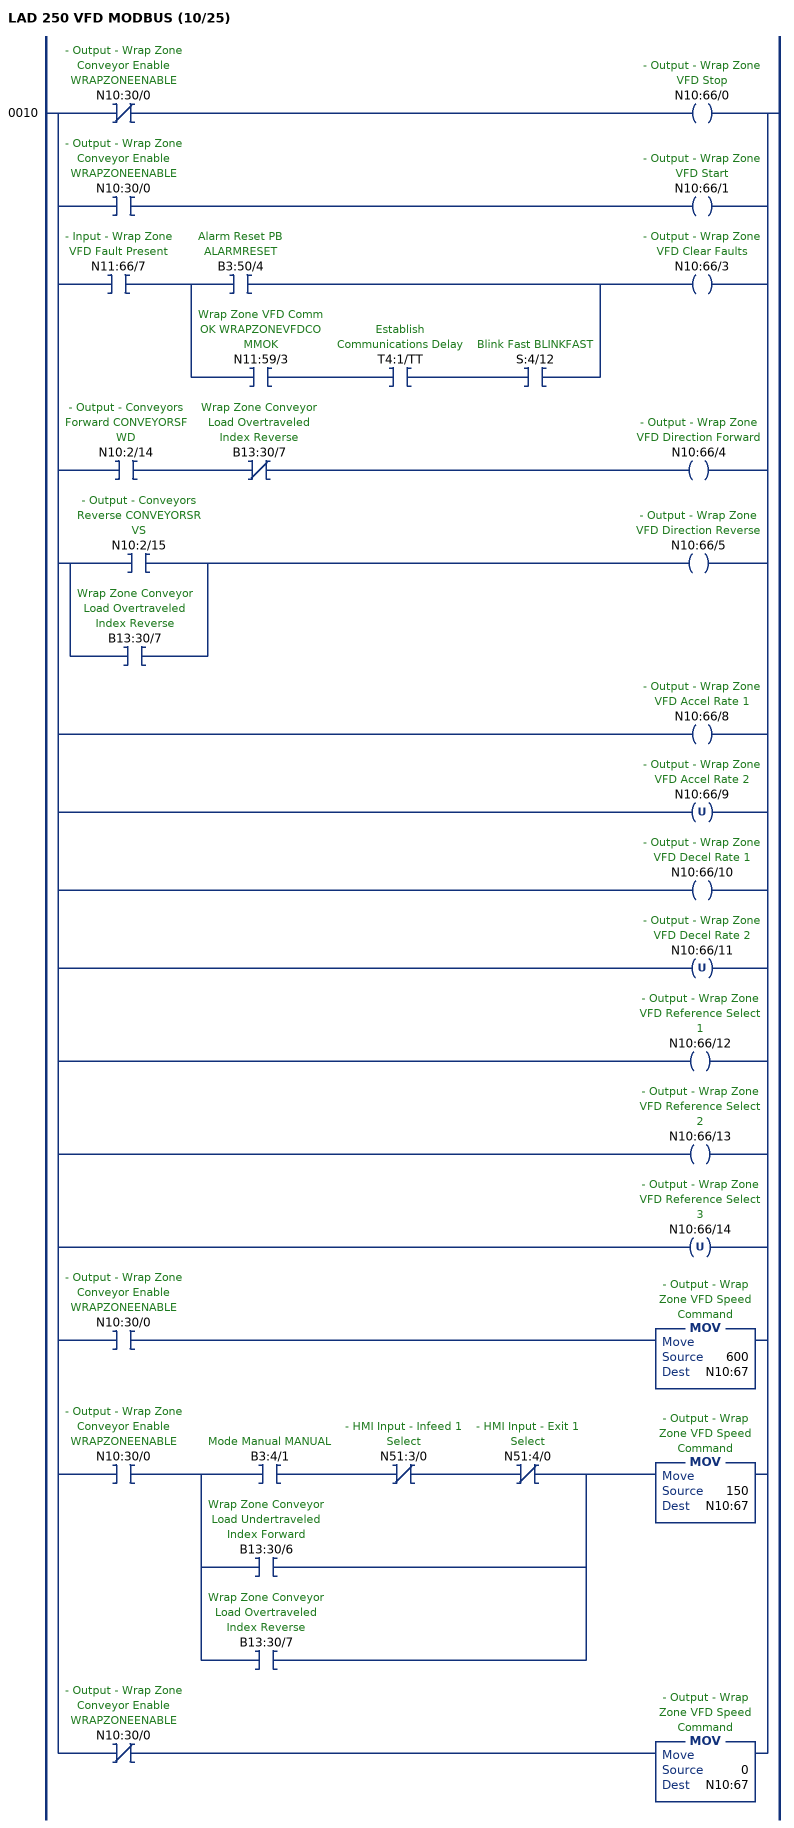
% Rung: 10 %
SOR BST XIO N10:30/0 OTE N10:66/0 NXB XIC N10:30/0 OTE N10:66/1 NXB XIC N11:66/7 BST XIC B3:50/4 NXB XIC N11:59/3 XIC T4:1/TT XIC S:4/12 BND OTE N10:66/3 NXB XIC N10:2/14 XIO B13:30/7 OTE N10:66/4 NXB BST XIC N10:2/15 NXB XIC B13:30/7 BND OTE N10:66/5 NXB OTE N10:66/8 NXB OTU N10:66/9 NXB OTE N10:66/10 NXB OTU N10:66/11 NXB OTE N10:66/12 NXB OTE N10:66/13 NXB OTU N10:66/14 NXB XIC N10:30/0 MOV 600 N10:67 NXB XIC N10:30/0 BST XIC B3:4/1 XIO N51:3/0 XIO N51:4/0 NXB XIC B13:30/6 NXB XIC B13:30/7 BND MOV 150 N10:67 NXB XIO N10:30/0 MOV 0 N10:67 BND EOR
%   N10:30/0  WRAPZONEENABLE  "- Output - Wrap Zone Conveyor Enable" %
%   N10:66/0  "- Output - Wrap Zone VFD Stop" %
%   N10:66/1  "- Output - Wrap Zone VFD Start" %
%   N11:66/7  "- Input - Wrap Zone VFD Fault Present" %
%   B3:50/4  ALARMRESET  "Alarm Reset PB" %
%   N11:59/3  WRAPZONEVFDCOMMOK  "Wrap Zone VFD Comm OK" %
%   T4:1  "Establish Communications Delay" %
%   S:4/12  BLINKFAST  "Blink Fast" %
%   N10:66/3  "- Output - Wrap Zone VFD Clear Faults" %
%   N10:2/14  CONVEYORSFWD  "- Output - Conveyors Forward" %
%   B13:30/7  "Wrap Zone Conveyor Load Overtraveled Index Reverse" %
%   N10:66/4  "- Output - Wrap Zone VFD Direction Forward" %
%   N10:2/15  CONVEYORSRVS  "- Output - Conveyors Reverse" %
%   N10:66/5  "- Output - Wrap Zone VFD Direction Reverse" %
%   N10:66/8  "- Output - Wrap Zone VFD Accel Rate 1" %
%   N10:66/9  "- Output - Wrap Zone VFD Accel Rate 2" %
%   N10:66/10  "- Output - Wrap Zone VFD Decel Rate 1" %
%   N10:66/11  "- Output - Wrap Zone VFD Decel Rate 2" %
%   N10:66/12  "- Output - Wrap Zone VFD Reference Select 1" %
%   N10:66/13  "- Output - Wrap Zone VFD Reference Select 2" %
%   N10:66/14  "- Output - Wrap Zone VFD Reference Select 3" %
%   N10:67  "- Output - Wrap Zone VFD Speed Command" %
%   B3:4/1  MANUAL  "Mode Manual" %
%   N51:3/0  "- HMI Input - Infeed 1 Select" %
%   N51:4/0  "- HMI Input - Exit 1 Select" %
%   B13:30/6  "Wrap Zone Conveyor Load Undertraveled Index Forward" %

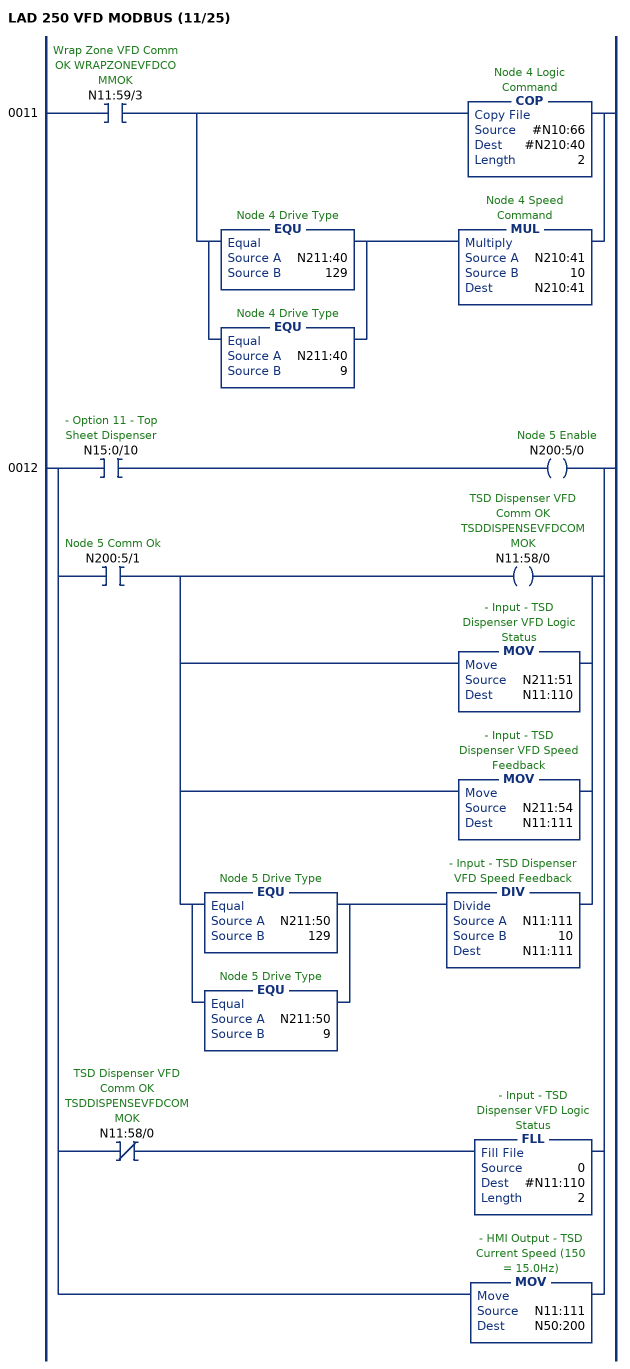
% Rung: 11 %
SOR XIC N11:59/3 BST COP #N10:66 #N210:40 2 NXB BST EQU N211:40 129 NXB EQU N211:40 9 BND MUL N210:41 10 N210:41 BND EOR
%   N11:59/3  WRAPZONEVFDCOMMOK  "Wrap Zone VFD Comm OK" %
%   N10:66  "- Output - Wrap Zone VFD Logic Command" %
%   N210:40  "Node 4 Logic Command" %
%   N211:40  "Node 4 Drive Type" %
%   N210:41  "Node 4 Speed Command" %
% Rung: 12 %
SOR BST XIC N15:0/10 OTE N200:5/0 NXB XIC N200:5/1 BST OTE N11:58/0 NXB MOV N211:51 N11:110 NXB MOV N211:54 N11:111 NXB BST EQU N211:50 129 NXB EQU N211:50 9 BND DIV N11:111 10 N11:111 BND NXB XIO N11:58/0 FLL 0 #N11:110 2 NXB MOV N11:111 N50:200 BND EOR
%   N15:0/10  "- Option 11 - Top Sheet Dispenser" %
%   N200:5/0  "Node 5 Enable" %
%   N200:5/1  "Node 5 Comm Ok" %
%   N11:58/0  TSDDISPENSEVFDCOMMOK  "TSD Dispenser VFD Comm OK" %
%   N211:51  "Node 5 Logic Status" %
%   N11:110  "- Input - TSD Dispenser VFD Logic Status" %
%   N211:54  "Node 5 Speed Feedback" %
%   N11:111  "- Input - TSD Dispenser VFD Speed Feedback" %
%   N211:50  "Node 5 Drive Type" %
%   N50:200  "- HMI Output - TSD Current Speed (150 = 15.0Hz)" %

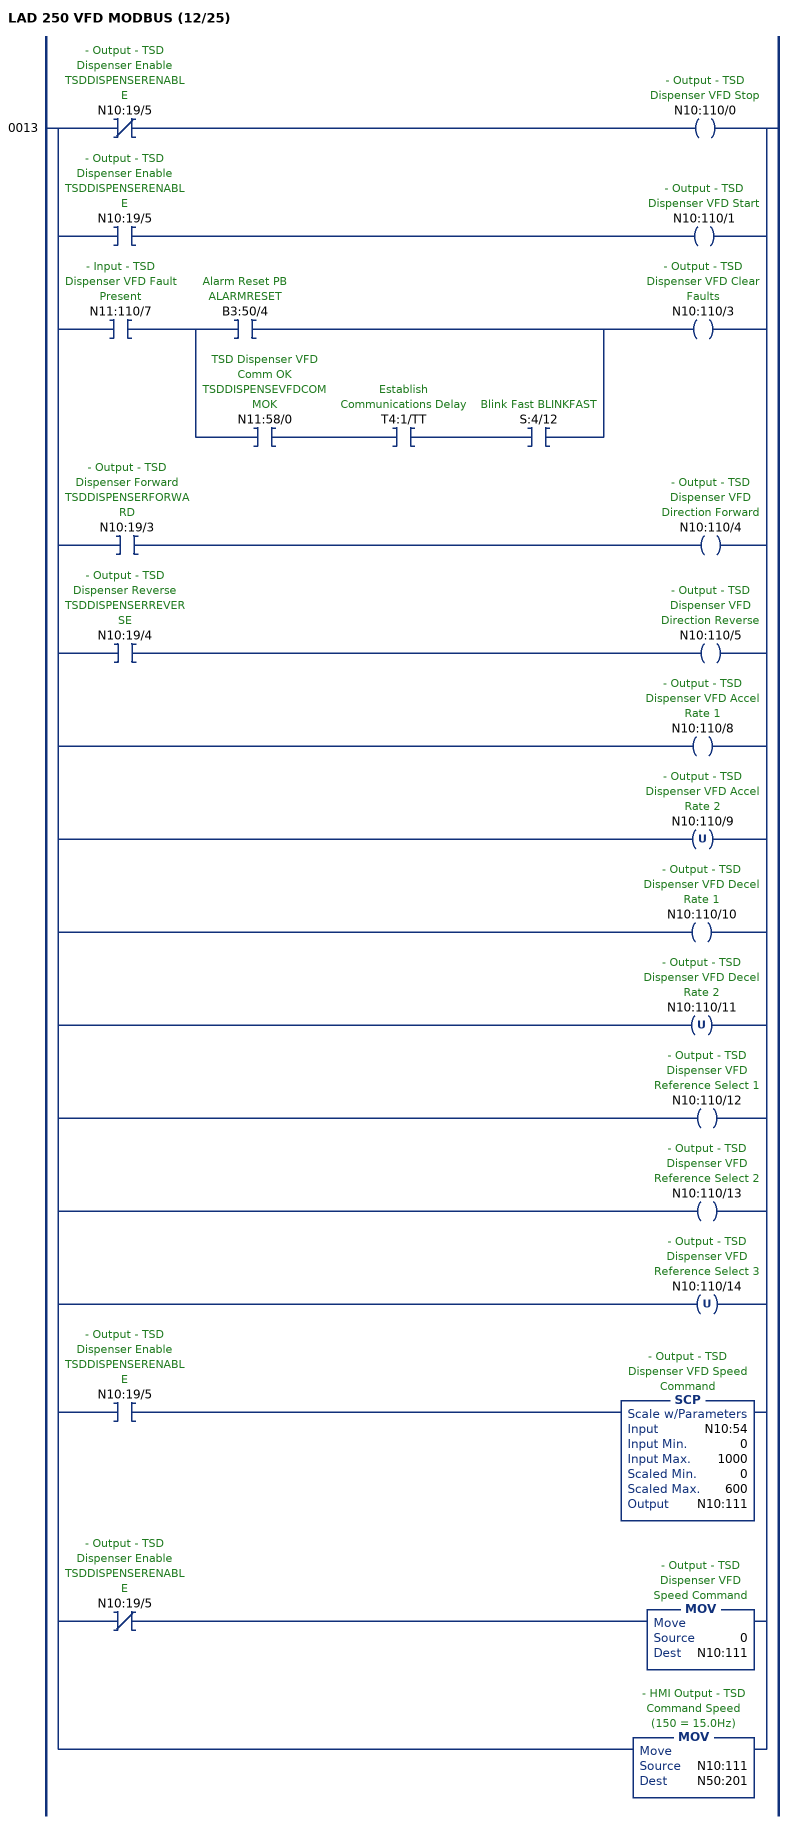
% Rung: 13 %
SOR BST XIO N10:19/5 OTE N10:110/0 NXB XIC N10:19/5 OTE N10:110/1 NXB XIC N11:110/7 BST XIC B3:50/4 NXB XIC N11:58/0 XIC T4:1/TT XIC S:4/12 BND OTE N10:110/3 NXB XIC N10:19/3 OTE N10:110/4 NXB XIC N10:19/4 OTE N10:110/5 NXB OTE N10:110/8 NXB OTU N10:110/9 NXB OTE N10:110/10 NXB OTU N10:110/11 NXB OTE N10:110/12 NXB OTE N10:110/13 NXB OTU N10:110/14 NXB XIC N10:19/5 SCP N10:54 0 1000 0 600 N10:111 NXB XIO N10:19/5 MOV 0 N10:111 NXB MOV N10:111 N50:201 BND EOR
%   N10:19/5  TSDDISPENSERENABLE  "- Output - TSD Dispenser Enable" %
%   N10:110/0  "- Output - TSD Dispenser VFD Stop" %
%   N10:110/1  "- Output - TSD Dispenser VFD Start" %
%   N11:110/7  "- Input - TSD Dispenser VFD Fault Present" %
%   B3:50/4  ALARMRESET  "Alarm Reset PB" %
%   N11:58/0  TSDDISPENSEVFDCOMMOK  "TSD Dispenser VFD Comm OK" %
%   T4:1  "Establish Communications Delay" %
%   S:4/12  BLINKFAST  "Blink Fast" %
%   N10:110/3  "- Output - TSD Dispenser VFD Clear Faults" %
%   N10:19/3  TSDDISPENSERFORWARD  "- Output - TSD Dispenser Forward" %
%   N10:110/4  "- Output - TSD Dispenser VFD Direction Forward" %
%   N10:19/4  TSDDISPENSERREVERSE  "- Output - TSD Dispenser Reverse" %
%   N10:110/5  "- Output - TSD Dispenser VFD Direction Reverse" %
%   N10:110/8  "- Output - TSD Dispenser VFD Accel Rate 1" %
%   N10:110/9  "- Output - TSD Dispenser VFD Accel Rate 2" %
%   N10:110/10  "- Output - TSD Dispenser VFD Decel Rate 1" %
%   N10:110/11  "- Output - TSD Dispenser VFD Decel Rate 2" %
%   N10:110/12  "- Output - TSD Dispenser VFD Reference Select 1" %
%   N10:110/13  "- Output - TSD Dispenser VFD Reference Select 2" %
%   N10:110/14  "- Output - TSD Dispenser VFD Reference Select 3" %
%   N10:54  TSDDISPENSECOMMAND  "- Output - TSD Dispense Speed Command (1000 = 100.0%)" %
%   N10:111  "- Output - TSD Dispenser VFD Speed Command" %
%   N50:201  "- HMI Output - TSD Command Speed (150 = 15.0Hz)" %

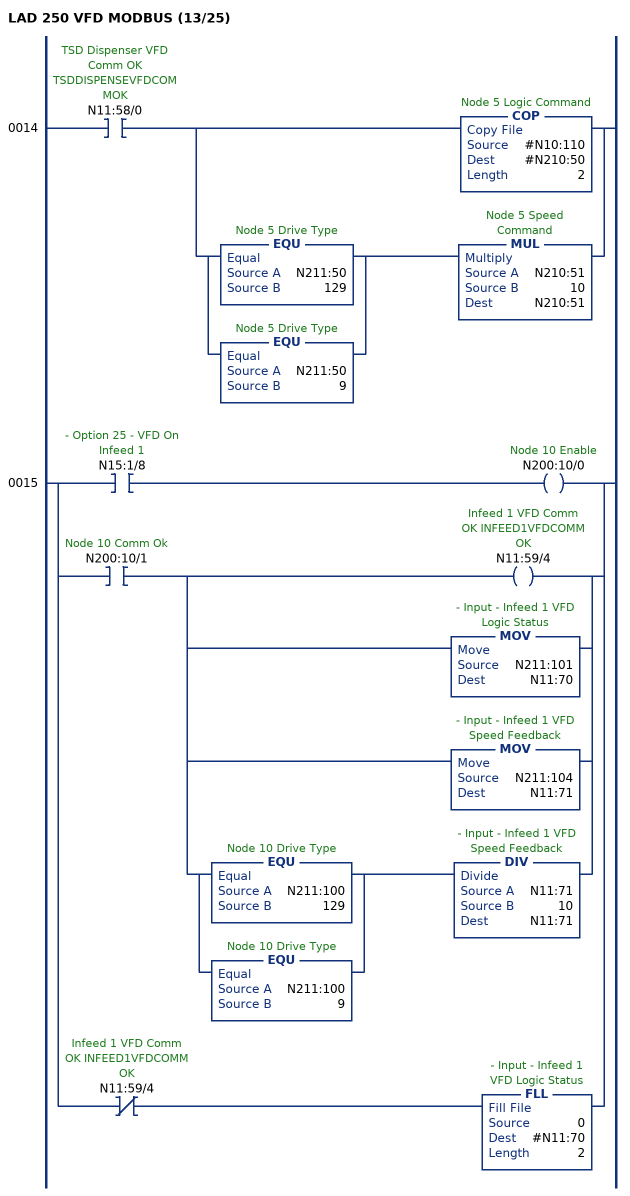
% Rung: 14 %
SOR XIC N11:58/0 BST COP #N10:110 #N210:50 2 NXB BST EQU N211:50 129 NXB EQU N211:50 9 BND MUL N210:51 10 N210:51 BND EOR
%   N11:58/0  TSDDISPENSEVFDCOMMOK  "TSD Dispenser VFD Comm OK" %
%   N10:110  "- Output - TSD Dispenser VFD Logic Command" %
%   N210:50  "Node 5 Logic Command" %
%   N211:50  "Node 5 Drive Type" %
%   N210:51  "Node 5 Speed Command" %
% Rung: 15 %
SOR BST XIC N15:1/8 OTE N200:10/0 NXB XIC N200:10/1 BST OTE N11:59/4 NXB MOV N211:101 N11:70 NXB MOV N211:104 N11:71 NXB BST EQU N211:100 129 NXB EQU N211:100 9 BND DIV N11:71 10 N11:71 BND NXB XIO N11:59/4 FLL 0 #N11:70 2 BND EOR
%   N15:1/8  "- Option 25 - VFD On Infeed 1" %
%   N200:10/0  "Node 10 Enable" %
%   N200:10/1  "Node 10 Comm Ok" %
%   N11:59/4  INFEED1VFDCOMMOK  "Infeed 1 VFD Comm OK" %
%   N211:101  "Node 10 Logic Status" %
%   N11:70  "- Input - Infeed 1 VFD Logic Status" %
%   N211:104  "Node 10 Speed Feedback" %
%   N11:71  "- Input - Infeed 1 VFD Speed Feedback" %
%   N211:100  "Node 10 Drive Type" %

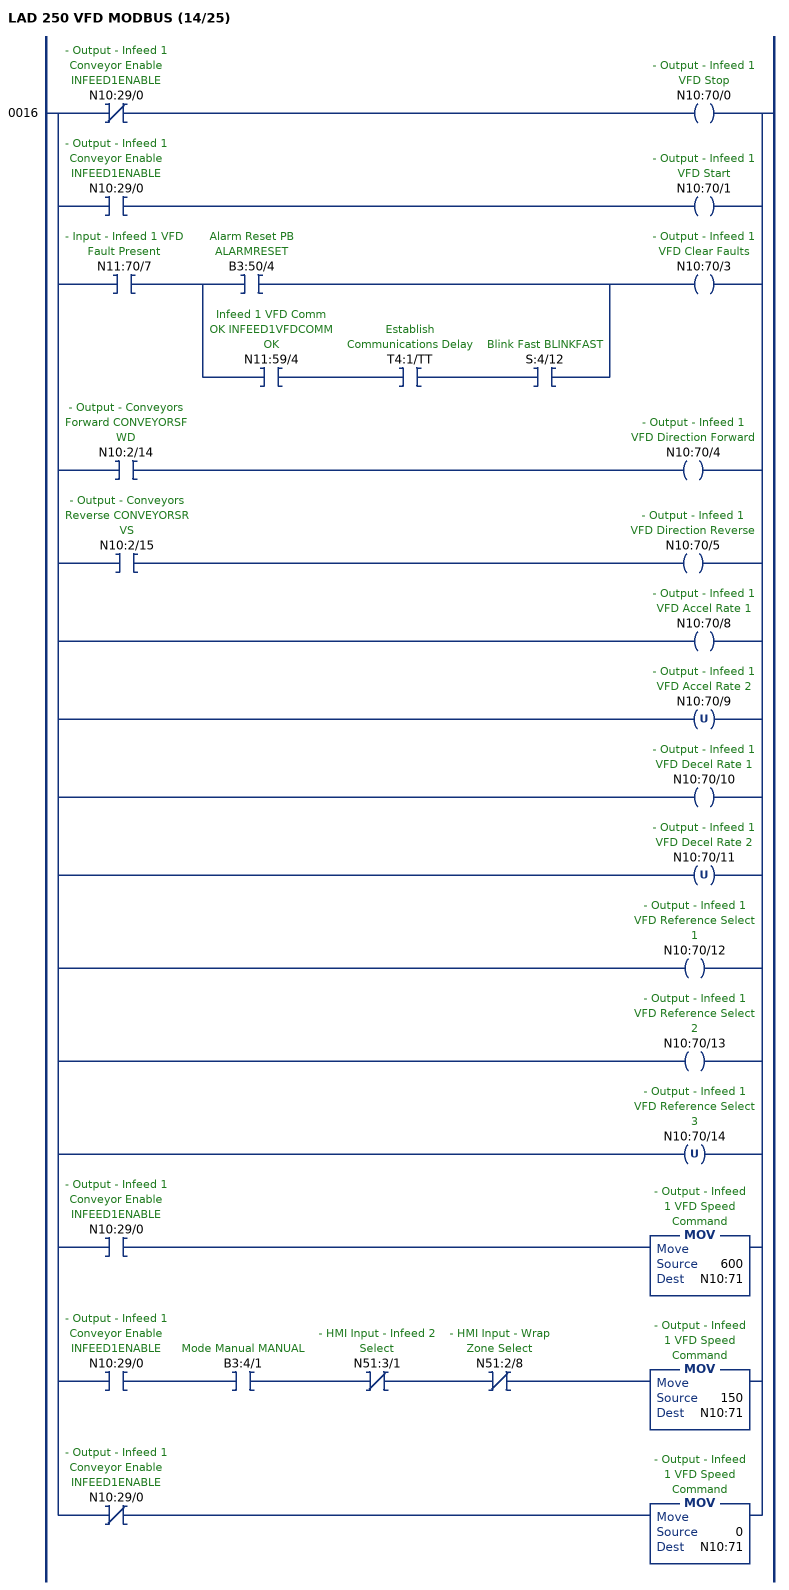
% Rung: 16 %
SOR BST XIO N10:29/0 OTE N10:70/0 NXB XIC N10:29/0 OTE N10:70/1 NXB XIC N11:70/7 BST XIC B3:50/4 NXB XIC N11:59/4 XIC T4:1/TT XIC S:4/12 BND OTE N10:70/3 NXB XIC N10:2/14 OTE N10:70/4 NXB XIC N10:2/15 OTE N10:70/5 NXB OTE N10:70/8 NXB OTU N10:70/9 NXB OTE N10:70/10 NXB OTU N10:70/11 NXB OTE N10:70/12 NXB OTE N10:70/13 NXB OTU N10:70/14 NXB XIC N10:29/0 MOV 600 N10:71 NXB XIC N10:29/0 XIC B3:4/1 XIO N51:3/1 XIO N51:2/8 MOV 150 N10:71 NXB XIO N10:29/0 MOV 0 N10:71 BND EOR
%   N10:29/0  INFEED1ENABLE  "- Output - Infeed 1 Conveyor Enable" %
%   N10:70/0  "- Output - Infeed 1 VFD Stop" %
%   N10:70/1  "- Output - Infeed 1 VFD Start" %
%   N11:70/7  "- Input - Infeed 1 VFD Fault Present" %
%   B3:50/4  ALARMRESET  "Alarm Reset PB" %
%   N11:59/4  INFEED1VFDCOMMOK  "Infeed 1 VFD Comm OK" %
%   T4:1  "Establish Communications Delay" %
%   S:4/12  BLINKFAST  "Blink Fast" %
%   N10:70/3  "- Output - Infeed 1 VFD Clear Faults" %
%   N10:2/14  CONVEYORSFWD  "- Output - Conveyors Forward" %
%   N10:70/4  "- Output - Infeed 1 VFD Direction Forward" %
%   N10:2/15  CONVEYORSRVS  "- Output - Conveyors Reverse" %
%   N10:70/5  "- Output - Infeed 1 VFD Direction Reverse" %
%   N10:70/8  "- Output - Infeed 1 VFD Accel Rate 1" %
%   N10:70/9  "- Output - Infeed 1 VFD Accel Rate 2" %
%   N10:70/10  "- Output - Infeed 1 VFD Decel Rate 1" %
%   N10:70/11  "- Output - Infeed 1 VFD Decel Rate 2" %
%   N10:70/12  "- Output - Infeed 1 VFD Reference Select 1" %
%   N10:70/13  "- Output - Infeed 1 VFD Reference Select 2" %
%   N10:70/14  "- Output - Infeed 1 VFD Reference Select 3" %
%   N10:71  "- Output - Infeed 1 VFD Speed Command" %
%   B3:4/1  MANUAL  "Mode Manual" %
%   N51:3/1  "- HMI Input - Infeed 2 Select" %
%   N51:2/8  "- HMI Input - Wrap Zone Select" %

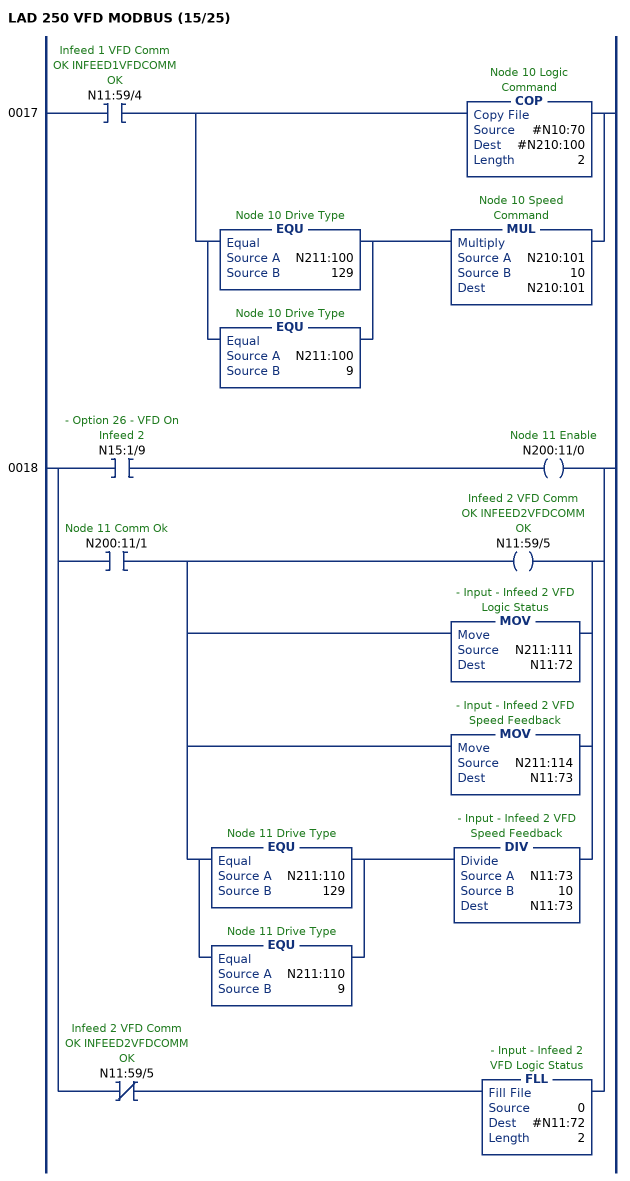
% Rung: 17 %
SOR XIC N11:59/4 BST COP #N10:70 #N210:100 2 NXB BST EQU N211:100 129 NXB EQU N211:100 9 BND MUL N210:101 10 N210:101 BND EOR
%   N11:59/4  INFEED1VFDCOMMOK  "Infeed 1 VFD Comm OK" %
%   N10:70  "- Output - Infeed 1 VFD Logic Command" %
%   N210:100  "Node 10 Logic Command" %
%   N211:100  "Node 10 Drive Type" %
%   N210:101  "Node 10 Speed Command" %
% Rung: 18 %
SOR BST XIC N15:1/9 OTE N200:11/0 NXB XIC N200:11/1 BST OTE N11:59/5 NXB MOV N211:111 N11:72 NXB MOV N211:114 N11:73 NXB BST EQU N211:110 129 NXB EQU N211:110 9 BND DIV N11:73 10 N11:73 BND NXB XIO N11:59/5 FLL 0 #N11:72 2 BND EOR
%   N15:1/9  "- Option 26 - VFD On Infeed 2" %
%   N200:11/0  "Node 11 Enable" %
%   N200:11/1  "Node 11 Comm Ok" %
%   N11:59/5  INFEED2VFDCOMMOK  "Infeed 2 VFD Comm OK" %
%   N211:111  "Node 11 Logic Status" %
%   N11:72  "- Input - Infeed 2 VFD Logic Status" %
%   N211:114  "Node 11 Speed Feedback" %
%   N11:73  "- Input - Infeed 2 VFD Speed Feedback" %
%   N211:110  "Node 11 Drive Type" %

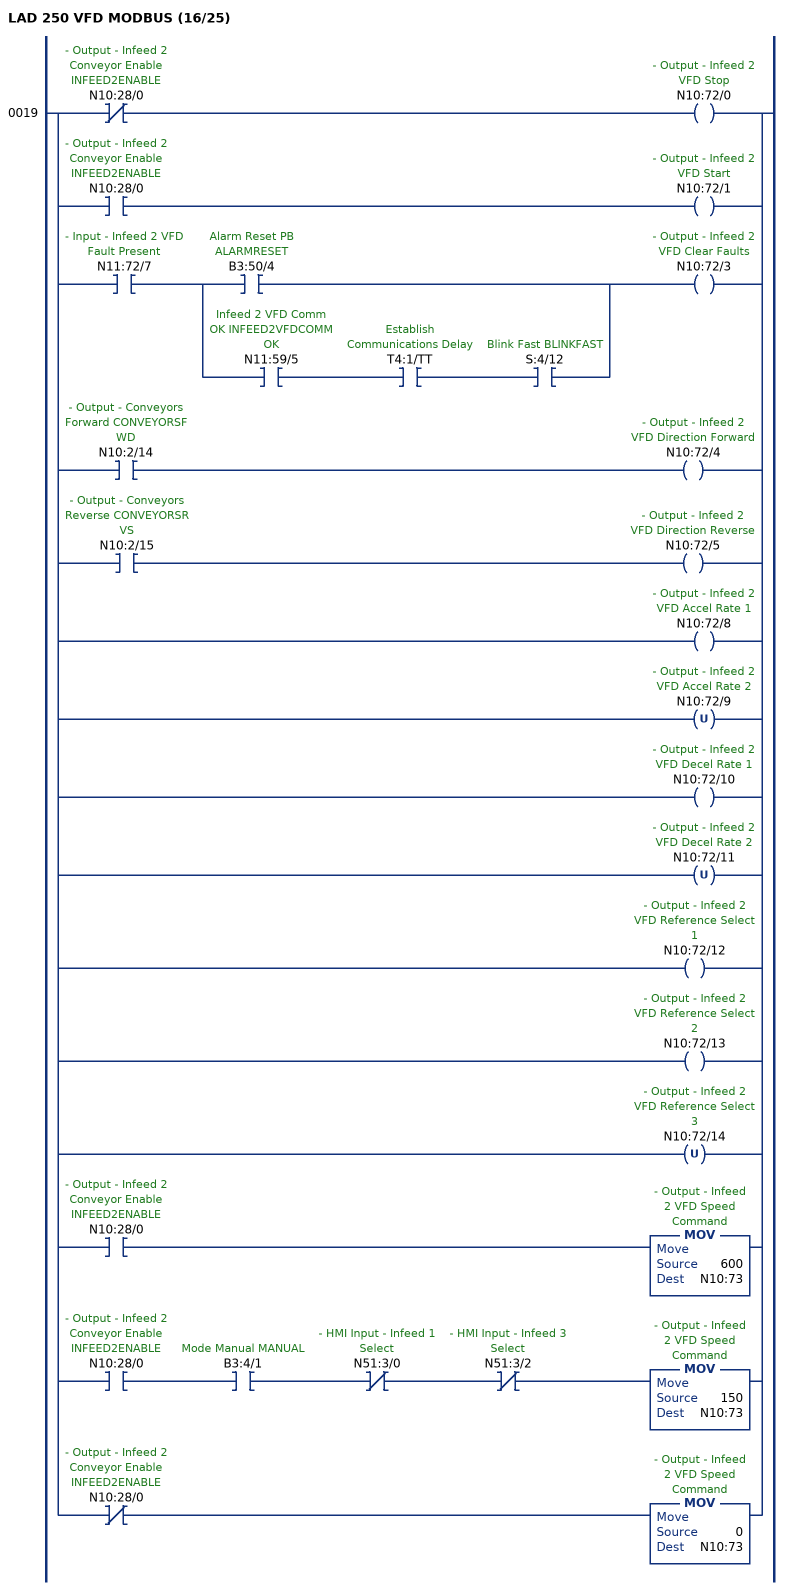
% Rung: 19 %
SOR BST XIO N10:28/0 OTE N10:72/0 NXB XIC N10:28/0 OTE N10:72/1 NXB XIC N11:72/7 BST XIC B3:50/4 NXB XIC N11:59/5 XIC T4:1/TT XIC S:4/12 BND OTE N10:72/3 NXB XIC N10:2/14 OTE N10:72/4 NXB XIC N10:2/15 OTE N10:72/5 NXB OTE N10:72/8 NXB OTU N10:72/9 NXB OTE N10:72/10 NXB OTU N10:72/11 NXB OTE N10:72/12 NXB OTE N10:72/13 NXB OTU N10:72/14 NXB XIC N10:28/0 MOV 600 N10:73 NXB XIC N10:28/0 XIC B3:4/1 XIO N51:3/0 XIO N51:3/2 MOV 150 N10:73 NXB XIO N10:28/0 MOV 0 N10:73 BND EOR
%   N10:28/0  INFEED2ENABLE  "- Output - Infeed 2 Conveyor Enable" %
%   N10:72/0  "- Output - Infeed 2 VFD Stop" %
%   N10:72/1  "- Output - Infeed 2 VFD Start" %
%   N11:72/7  "- Input - Infeed 2 VFD Fault Present" %
%   B3:50/4  ALARMRESET  "Alarm Reset PB" %
%   N11:59/5  INFEED2VFDCOMMOK  "Infeed 2 VFD Comm OK" %
%   T4:1  "Establish Communications Delay" %
%   S:4/12  BLINKFAST  "Blink Fast" %
%   N10:72/3  "- Output - Infeed 2 VFD Clear Faults" %
%   N10:2/14  CONVEYORSFWD  "- Output - Conveyors Forward" %
%   N10:72/4  "- Output - Infeed 2 VFD Direction Forward" %
%   N10:2/15  CONVEYORSRVS  "- Output - Conveyors Reverse" %
%   N10:72/5  "- Output - Infeed 2 VFD Direction Reverse" %
%   N10:72/8  "- Output - Infeed 2 VFD Accel Rate 1" %
%   N10:72/9  "- Output - Infeed 2 VFD Accel Rate 2" %
%   N10:72/10  "- Output - Infeed 2 VFD Decel Rate 1" %
%   N10:72/11  "- Output - Infeed 2 VFD Decel Rate 2" %
%   N10:72/12  "- Output - Infeed 2 VFD Reference Select 1" %
%   N10:72/13  "- Output - Infeed 2 VFD Reference Select 2" %
%   N10:72/14  "- Output - Infeed 2 VFD Reference Select 3" %
%   N10:73  "- Output - Infeed 2 VFD Speed Command" %
%   B3:4/1  MANUAL  "Mode Manual" %
%   N51:3/0  "- HMI Input - Infeed 1 Select" %
%   N51:3/2  "- HMI Input - Infeed 3 Select" %

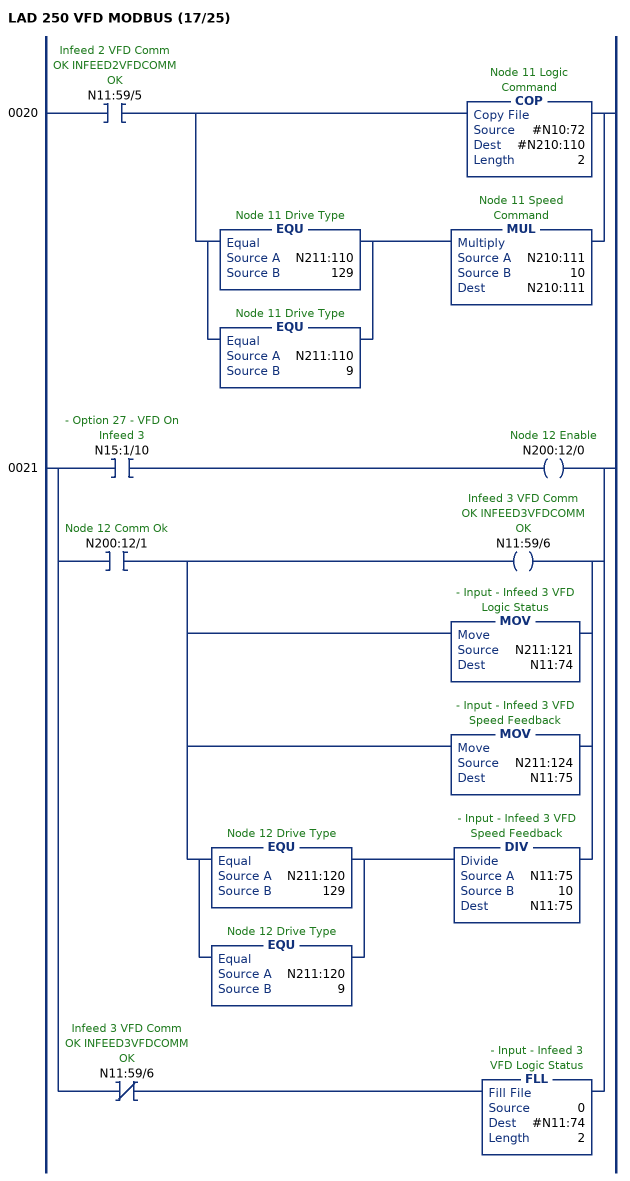
% Rung: 20 %
SOR XIC N11:59/5 BST COP #N10:72 #N210:110 2 NXB BST EQU N211:110 129 NXB EQU N211:110 9 BND MUL N210:111 10 N210:111 BND EOR
%   N11:59/5  INFEED2VFDCOMMOK  "Infeed 2 VFD Comm OK" %
%   N10:72  "- Output - Infeed 2 VFD Logic Command" %
%   N210:110  "Node 11 Logic Command" %
%   N211:110  "Node 11 Drive Type" %
%   N210:111  "Node 11 Speed Command" %
% Rung: 21 %
SOR BST XIC N15:1/10 OTE N200:12/0 NXB XIC N200:12/1 BST OTE N11:59/6 NXB MOV N211:121 N11:74 NXB MOV N211:124 N11:75 NXB BST EQU N211:120 129 NXB EQU N211:120 9 BND DIV N11:75 10 N11:75 BND NXB XIO N11:59/6 FLL 0 #N11:74 2 BND EOR
%   N15:1/10  "- Option 27 - VFD On Infeed 3" %
%   N200:12/0  "Node 12 Enable" %
%   N200:12/1  "Node 12 Comm Ok" %
%   N11:59/6  INFEED3VFDCOMMOK  "Infeed 3 VFD Comm OK" %
%   N211:121  "Node 12 Logic Status" %
%   N11:74  "- Input - Infeed 3 VFD Logic Status" %
%   N211:124  "Node 12 Speed Feedback" %
%   N11:75  "- Input - Infeed 3 VFD Speed Feedback" %
%   N211:120  "Node 12 Drive Type" %

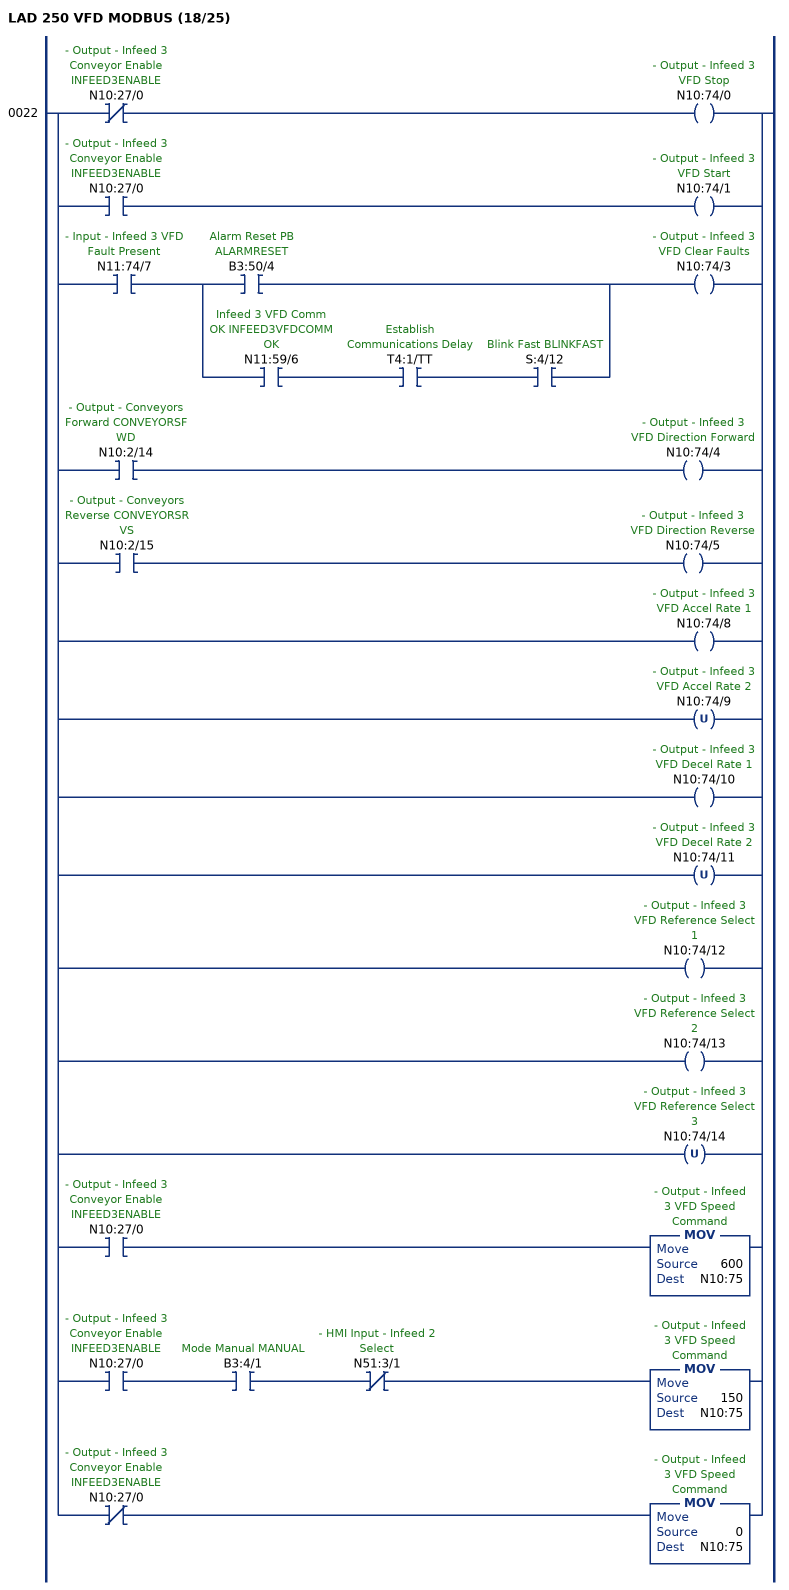
% Rung: 22 %
SOR BST XIO N10:27/0 OTE N10:74/0 NXB XIC N10:27/0 OTE N10:74/1 NXB XIC N11:74/7 BST XIC B3:50/4 NXB XIC N11:59/6 XIC T4:1/TT XIC S:4/12 BND OTE N10:74/3 NXB XIC N10:2/14 OTE N10:74/4 NXB XIC N10:2/15 OTE N10:74/5 NXB OTE N10:74/8 NXB OTU N10:74/9 NXB OTE N10:74/10 NXB OTU N10:74/11 NXB OTE N10:74/12 NXB OTE N10:74/13 NXB OTU N10:74/14 NXB XIC N10:27/0 MOV 600 N10:75 NXB XIC N10:27/0 XIC B3:4/1 XIO N51:3/1 MOV 150 N10:75 NXB XIO N10:27/0 MOV 0 N10:75 BND EOR
%   N10:27/0  INFEED3ENABLE  "- Output - Infeed 3 Conveyor Enable" %
%   N10:74/0  "- Output - Infeed 3 VFD Stop" %
%   N10:74/1  "- Output - Infeed 3 VFD Start" %
%   N11:74/7  "- Input - Infeed 3 VFD Fault Present" %
%   B3:50/4  ALARMRESET  "Alarm Reset PB" %
%   N11:59/6  INFEED3VFDCOMMOK  "Infeed 3 VFD Comm OK" %
%   T4:1  "Establish Communications Delay" %
%   S:4/12  BLINKFAST  "Blink Fast" %
%   N10:74/3  "- Output - Infeed 3 VFD Clear Faults" %
%   N10:2/14  CONVEYORSFWD  "- Output - Conveyors Forward" %
%   N10:74/4  "- Output - Infeed 3 VFD Direction Forward" %
%   N10:2/15  CONVEYORSRVS  "- Output - Conveyors Reverse" %
%   N10:74/5  "- Output - Infeed 3 VFD Direction Reverse" %
%   N10:74/8  "- Output - Infeed 3 VFD Accel Rate 1" %
%   N10:74/9  "- Output - Infeed 3 VFD Accel Rate 2" %
%   N10:74/10  "- Output - Infeed 3 VFD Decel Rate 1" %
%   N10:74/11  "- Output - Infeed 3 VFD Decel Rate 2" %
%   N10:74/12  "- Output - Infeed 3 VFD Reference Select 1" %
%   N10:74/13  "- Output - Infeed 3 VFD Reference Select 2" %
%   N10:74/14  "- Output - Infeed 3 VFD Reference Select 3" %
%   N10:75  "- Output - Infeed 3 VFD Speed Command" %
%   B3:4/1  MANUAL  "Mode Manual" %
%   N51:3/1  "- HMI Input - Infeed 2 Select" %

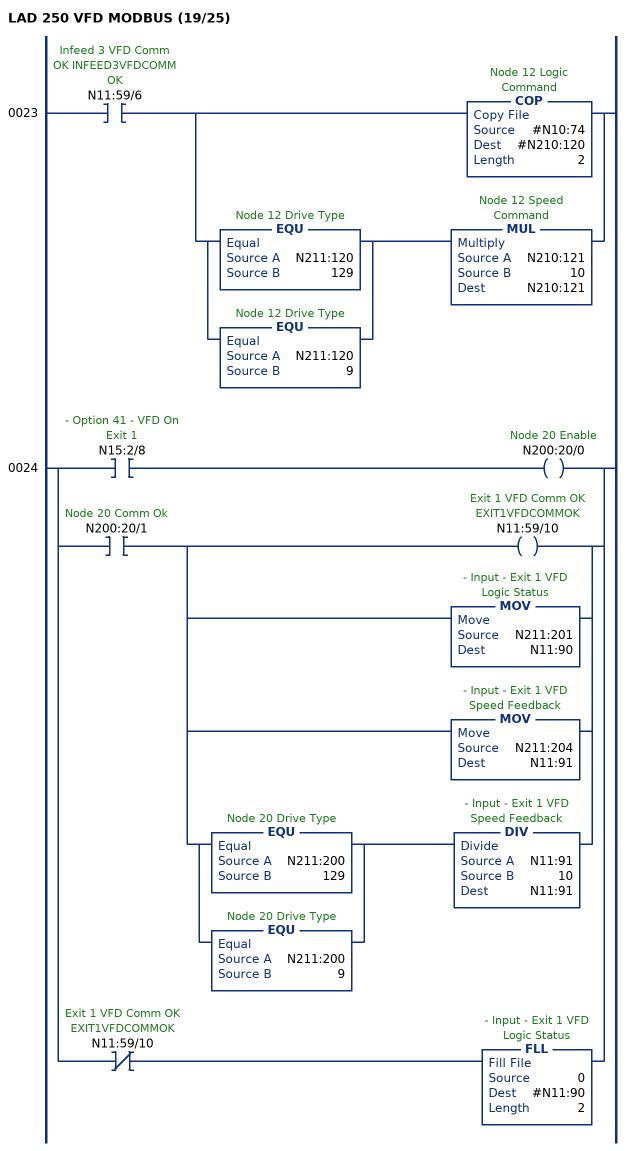
% Rung: 23 %
SOR XIC N11:59/6 BST COP #N10:74 #N210:120 2 NXB BST EQU N211:120 129 NXB EQU N211:120 9 BND MUL N210:121 10 N210:121 BND EOR
%   N11:59/6  INFEED3VFDCOMMOK  "Infeed 3 VFD Comm OK" %
%   N10:74  "- Output - Infeed 3 VFD Logic Command" %
%   N210:120  "Node 12 Logic Command" %
%   N211:120  "Node 12 Drive Type" %
%   N210:121  "Node 12 Speed Command" %
% Rung: 24 %
SOR BST XIC N15:2/8 OTE N200:20/0 NXB XIC N200:20/1 BST OTE N11:59/10 NXB MOV N211:201 N11:90 NXB MOV N211:204 N11:91 NXB BST EQU N211:200 129 NXB EQU N211:200 9 BND DIV N11:91 10 N11:91 BND NXB XIO N11:59/10 FLL 0 #N11:90 2 BND EOR
%   N15:2/8  "- Option 41 - VFD On Exit 1" %
%   N200:20/0  "Node 20 Enable" %
%   N200:20/1  "Node 20 Comm Ok" %
%   N11:59/10  EXIT1VFDCOMMOK  "Exit 1 VFD Comm OK" %
%   N211:201  "Node 20 Logic Status" %
%   N11:90  "- Input - Exit 1 VFD Logic Status" %
%   N211:204  "Node 20 Speed Feedback" %
%   N11:91  "- Input - Exit 1 VFD Speed Feedback" %
%   N211:200  "Node 20 Drive Type" %

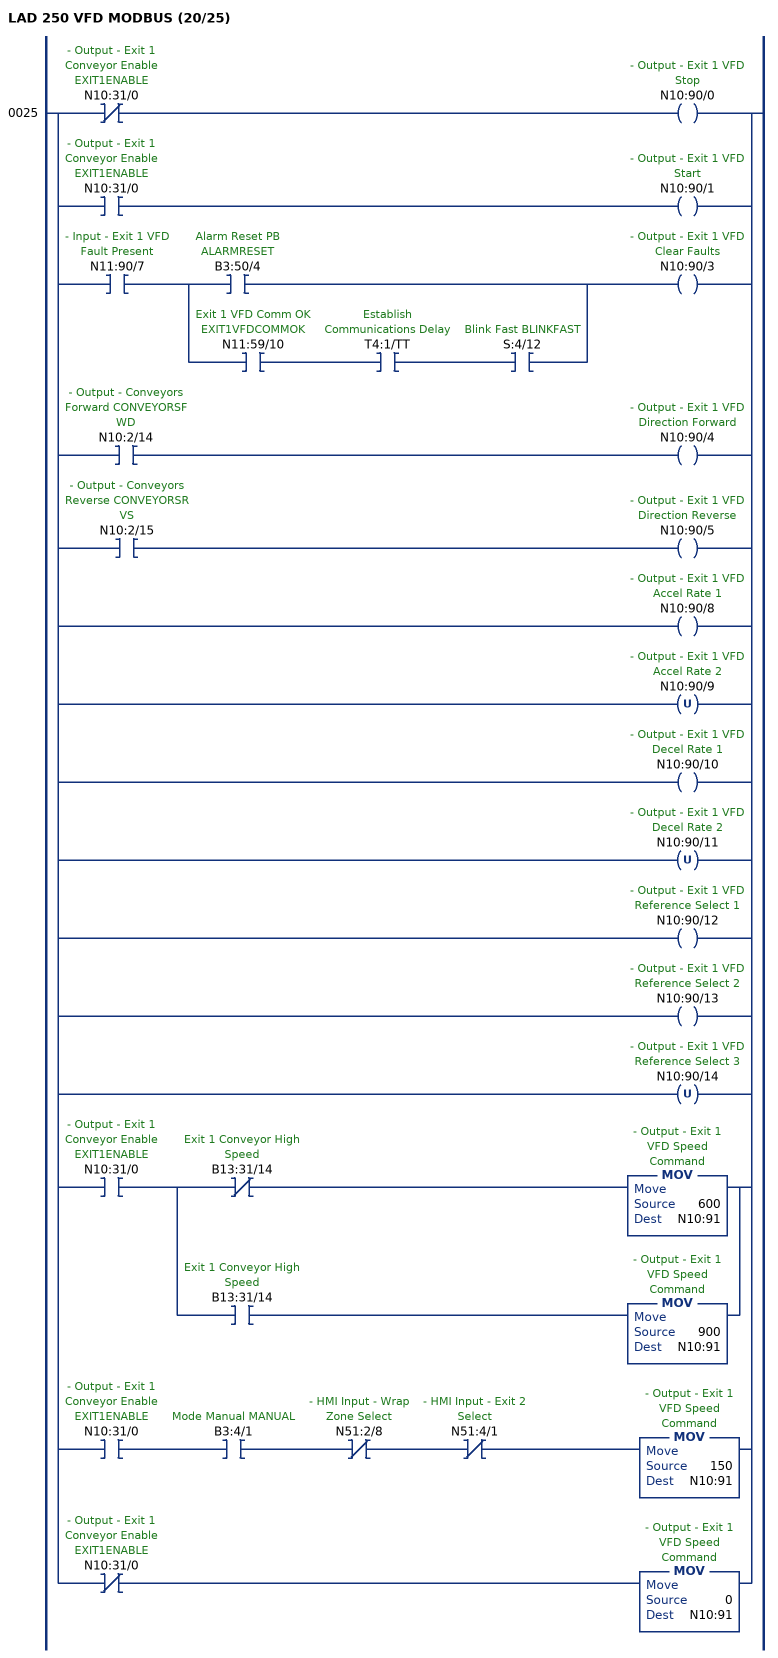
% Rung: 25 %
SOR BST XIO N10:31/0 OTE N10:90/0 NXB XIC N10:31/0 OTE N10:90/1 NXB XIC N11:90/7 BST XIC B3:50/4 NXB XIC N11:59/10 XIC T4:1/TT XIC S:4/12 BND OTE N10:90/3 NXB XIC N10:2/14 OTE N10:90/4 NXB XIC N10:2/15 OTE N10:90/5 NXB OTE N10:90/8 NXB OTU N10:90/9 NXB OTE N10:90/10 NXB OTU N10:90/11 NXB OTE N10:90/12 NXB OTE N10:90/13 NXB OTU N10:90/14 NXB XIC N10:31/0 BST XIO B13:31/14 MOV 600 N10:91 NXB XIC B13:31/14 MOV 900 N10:91 BND NXB XIC N10:31/0 XIC B3:4/1 XIO N51:2/8 XIO N51:4/1 MOV 150 N10:91 NXB XIO N10:31/0 MOV 0 N10:91 BND EOR
%   N10:31/0  EXIT1ENABLE  "- Output - Exit 1 Conveyor Enable" %
%   N10:90/0  "- Output - Exit 1 VFD Stop" %
%   N10:90/1  "- Output - Exit 1 VFD Start" %
%   N11:90/7  "- Input - Exit 1 VFD Fault Present" %
%   B3:50/4  ALARMRESET  "Alarm Reset PB" %
%   N11:59/10  EXIT1VFDCOMMOK  "Exit 1 VFD Comm OK" %
%   T4:1  "Establish Communications Delay" %
%   S:4/12  BLINKFAST  "Blink Fast" %
%   N10:90/3  "- Output - Exit 1 VFD Clear Faults" %
%   N10:2/14  CONVEYORSFWD  "- Output - Conveyors Forward" %
%   N10:90/4  "- Output - Exit 1 VFD Direction Forward" %
%   N10:2/15  CONVEYORSRVS  "- Output - Conveyors Reverse" %
%   N10:90/5  "- Output - Exit 1 VFD Direction Reverse" %
%   N10:90/8  "- Output - Exit 1 VFD Accel Rate 1" %
%   N10:90/9  "- Output - Exit 1 VFD Accel Rate 2" %
%   N10:90/10  "- Output - Exit 1 VFD Decel Rate 1" %
%   N10:90/11  "- Output - Exit 1 VFD Decel Rate 2" %
%   N10:90/12  "- Output - Exit 1 VFD Reference Select 1" %
%   N10:90/13  "- Output - Exit 1 VFD Reference Select 2" %
%   N10:90/14  "- Output - Exit 1 VFD Reference Select 3" %
%   B13:31/14  "Exit 1 Conveyor High Speed" %
%   N10:91  "- Output - Exit 1 VFD Speed Command" %
%   B3:4/1  MANUAL  "Mode Manual" %
%   N51:2/8  "- HMI Input - Wrap Zone Select" %
%   N51:4/1  "- HMI Input - Exit 2 Select" %

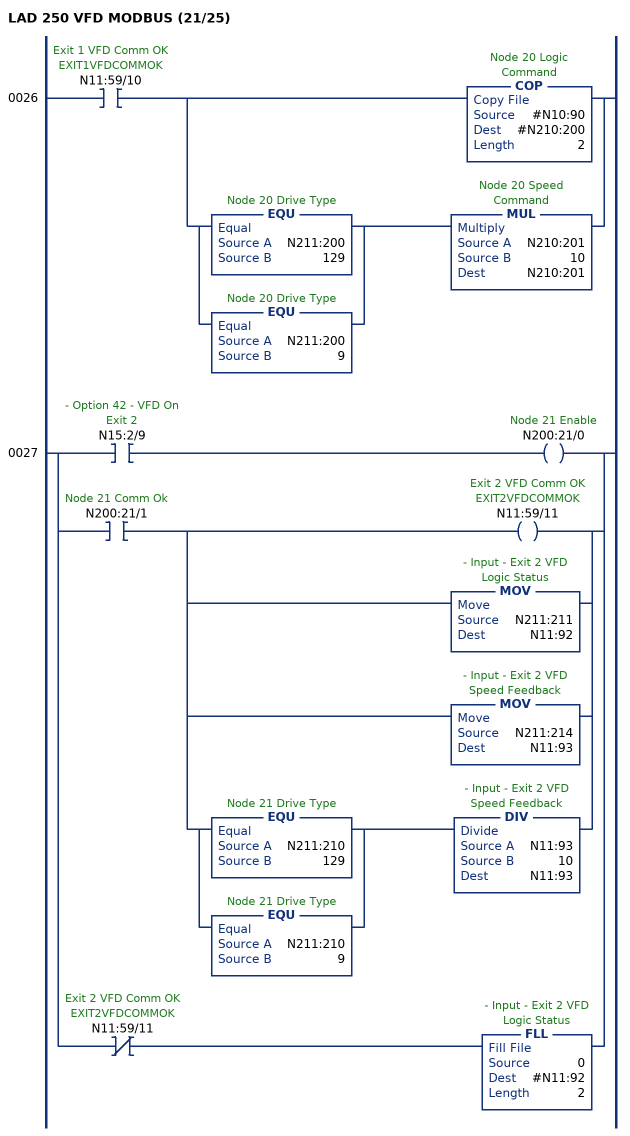
% Rung: 26 %
SOR XIC N11:59/10 BST COP #N10:90 #N210:200 2 NXB BST EQU N211:200 129 NXB EQU N211:200 9 BND MUL N210:201 10 N210:201 BND EOR
%   N11:59/10  EXIT1VFDCOMMOK  "Exit 1 VFD Comm OK" %
%   N10:90  "- Output - Exit 1 VFD Logic Command" %
%   N210:200  "Node 20 Logic Command" %
%   N211:200  "Node 20 Drive Type" %
%   N210:201  "Node 20 Speed Command" %
% Rung: 27 %
SOR BST XIC N15:2/9 OTE N200:21/0 NXB XIC N200:21/1 BST OTE N11:59/11 NXB MOV N211:211 N11:92 NXB MOV N211:214 N11:93 NXB BST EQU N211:210 129 NXB EQU N211:210 9 BND DIV N11:93 10 N11:93 BND NXB XIO N11:59/11 FLL 0 #N11:92 2 BND EOR
%   N15:2/9  "- Option 42 - VFD On Exit 2" %
%   N200:21/0  "Node 21 Enable" %
%   N200:21/1  "Node 21 Comm Ok" %
%   N11:59/11  EXIT2VFDCOMMOK  "Exit 2 VFD Comm OK" %
%   N211:211  "Node 21 Logic Status" %
%   N11:92  "- Input - Exit 2 VFD Logic Status" %
%   N211:214  "Node 21 Speed Feedback" %
%   N11:93  "- Input - Exit 2 VFD Speed Feedback" %
%   N211:210  "Node 21 Drive Type" %

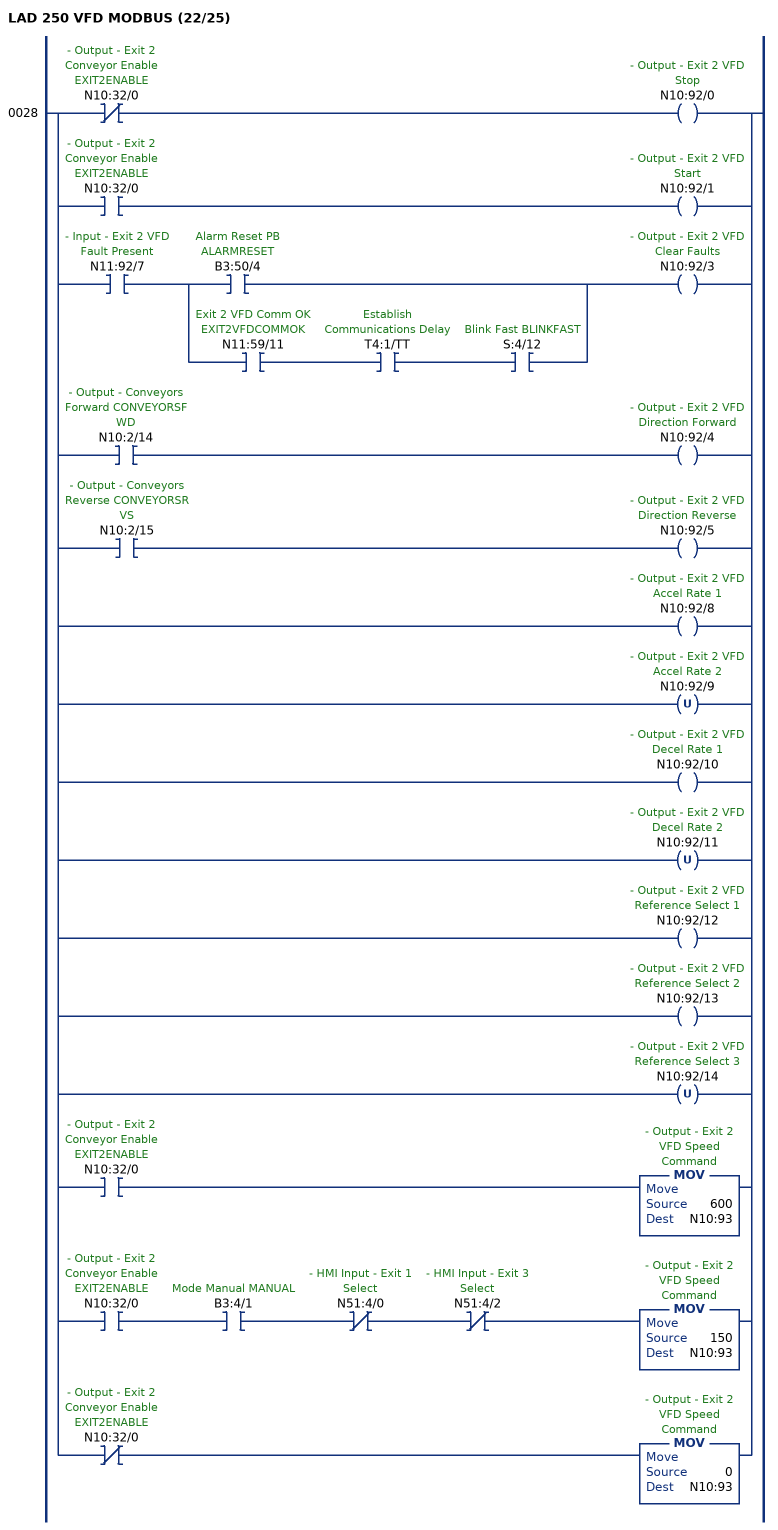
% Rung: 28 %
SOR BST XIO N10:32/0 OTE N10:92/0 NXB XIC N10:32/0 OTE N10:92/1 NXB XIC N11:92/7 BST XIC B3:50/4 NXB XIC N11:59/11 XIC T4:1/TT XIC S:4/12 BND OTE N10:92/3 NXB XIC N10:2/14 OTE N10:92/4 NXB XIC N10:2/15 OTE N10:92/5 NXB OTE N10:92/8 NXB OTU N10:92/9 NXB OTE N10:92/10 NXB OTU N10:92/11 NXB OTE N10:92/12 NXB OTE N10:92/13 NXB OTU N10:92/14 NXB XIC N10:32/0 MOV 600 N10:93 NXB XIC N10:32/0 XIC B3:4/1 XIO N51:4/0 XIO N51:4/2 MOV 150 N10:93 NXB XIO N10:32/0 MOV 0 N10:93 BND EOR
%   N10:32/0  EXIT2ENABLE  "- Output - Exit 2 Conveyor Enable" %
%   N10:92/0  "- Output - Exit 2 VFD Stop" %
%   N10:92/1  "- Output - Exit 2 VFD Start" %
%   N11:92/7  "- Input - Exit 2 VFD Fault Present" %
%   B3:50/4  ALARMRESET  "Alarm Reset PB" %
%   N11:59/11  EXIT2VFDCOMMOK  "Exit 2 VFD Comm OK" %
%   T4:1  "Establish Communications Delay" %
%   S:4/12  BLINKFAST  "Blink Fast" %
%   N10:92/3  "- Output - Exit 2 VFD Clear Faults" %
%   N10:2/14  CONVEYORSFWD  "- Output - Conveyors Forward" %
%   N10:92/4  "- Output - Exit 2 VFD Direction Forward" %
%   N10:2/15  CONVEYORSRVS  "- Output - Conveyors Reverse" %
%   N10:92/5  "- Output - Exit 2 VFD Direction Reverse" %
%   N10:92/8  "- Output - Exit 2 VFD Accel Rate 1" %
%   N10:92/9  "- Output - Exit 2 VFD Accel Rate 2" %
%   N10:92/10  "- Output - Exit 2 VFD Decel Rate 1" %
%   N10:92/11  "- Output - Exit 2 VFD Decel Rate 2" %
%   N10:92/12  "- Output - Exit 2 VFD Reference Select 1" %
%   N10:92/13  "- Output - Exit 2 VFD Reference Select 2" %
%   N10:92/14  "- Output - Exit 2 VFD Reference Select 3" %
%   N10:93  "- Output - Exit 2 VFD Speed Command" %
%   B3:4/1  MANUAL  "Mode Manual" %
%   N51:4/0  "- HMI Input - Exit 1 Select" %
%   N51:4/2  "- HMI Input - Exit 3 Select" %

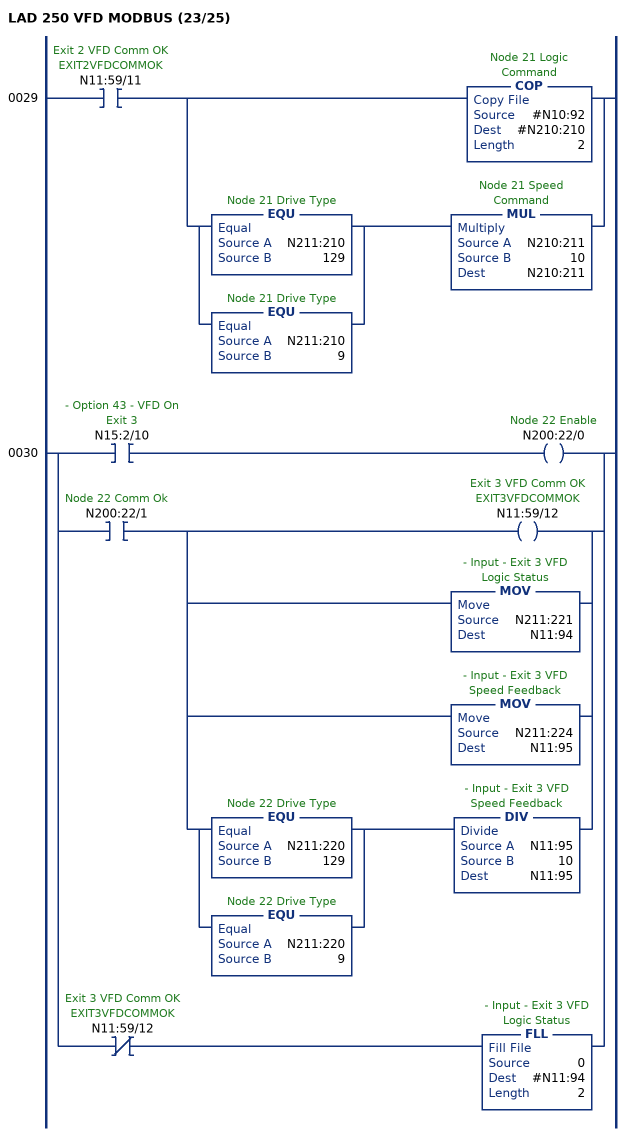
% Rung: 29 %
SOR XIC N11:59/11 BST COP #N10:92 #N210:210 2 NXB BST EQU N211:210 129 NXB EQU N211:210 9 BND MUL N210:211 10 N210:211 BND EOR
%   N11:59/11  EXIT2VFDCOMMOK  "Exit 2 VFD Comm OK" %
%   N10:92  "- Output - Exit 2 VFD Logic Command" %
%   N210:210  "Node 21 Logic Command" %
%   N211:210  "Node 21 Drive Type" %
%   N210:211  "Node 21 Speed Command" %
% Rung: 30 %
SOR BST XIC N15:2/10 OTE N200:22/0 NXB XIC N200:22/1 BST OTE N11:59/12 NXB MOV N211:221 N11:94 NXB MOV N211:224 N11:95 NXB BST EQU N211:220 129 NXB EQU N211:220 9 BND DIV N11:95 10 N11:95 BND NXB XIO N11:59/12 FLL 0 #N11:94 2 BND EOR
%   N15:2/10  "- Option 43 - VFD On Exit 3" %
%   N200:22/0  "Node 22 Enable" %
%   N200:22/1  "Node 22 Comm Ok" %
%   N11:59/12  EXIT3VFDCOMMOK  "Exit 3 VFD Comm OK" %
%   N211:221  "Node 22 Logic Status" %
%   N11:94  "- Input - Exit 3 VFD Logic Status" %
%   N211:224  "Node 22 Speed Feedback" %
%   N11:95  "- Input - Exit 3 VFD Speed Feedback" %
%   N211:220  "Node 22 Drive Type" %

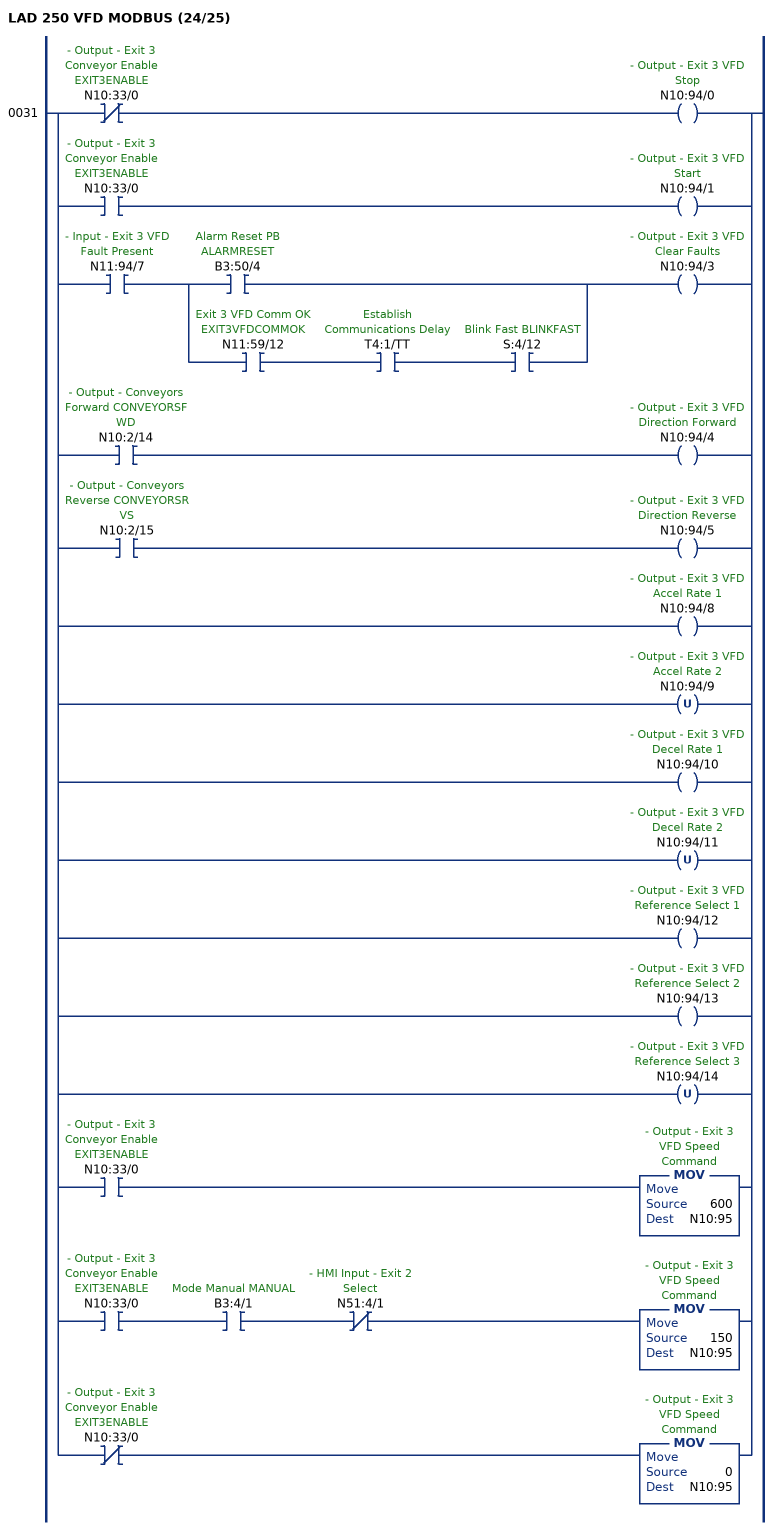
% Rung: 31 %
SOR BST XIO N10:33/0 OTE N10:94/0 NXB XIC N10:33/0 OTE N10:94/1 NXB XIC N11:94/7 BST XIC B3:50/4 NXB XIC N11:59/12 XIC T4:1/TT XIC S:4/12 BND OTE N10:94/3 NXB XIC N10:2/14 OTE N10:94/4 NXB XIC N10:2/15 OTE N10:94/5 NXB OTE N10:94/8 NXB OTU N10:94/9 NXB OTE N10:94/10 NXB OTU N10:94/11 NXB OTE N10:94/12 NXB OTE N10:94/13 NXB OTU N10:94/14 NXB XIC N10:33/0 MOV 600 N10:95 NXB XIC N10:33/0 XIC B3:4/1 XIO N51:4/1 MOV 150 N10:95 NXB XIO N10:33/0 MOV 0 N10:95 BND EOR
%   N10:33/0  EXIT3ENABLE  "- Output - Exit 3 Conveyor Enable" %
%   N10:94/0  "- Output - Exit 3 VFD Stop" %
%   N10:94/1  "- Output - Exit 3 VFD Start" %
%   N11:94/7  "- Input - Exit 3 VFD Fault Present" %
%   B3:50/4  ALARMRESET  "Alarm Reset PB" %
%   N11:59/12  EXIT3VFDCOMMOK  "Exit 3 VFD Comm OK" %
%   T4:1  "Establish Communications Delay" %
%   S:4/12  BLINKFAST  "Blink Fast" %
%   N10:94/3  "- Output - Exit 3 VFD Clear Faults" %
%   N10:2/14  CONVEYORSFWD  "- Output - Conveyors Forward" %
%   N10:94/4  "- Output - Exit 3 VFD Direction Forward" %
%   N10:2/15  CONVEYORSRVS  "- Output - Conveyors Reverse" %
%   N10:94/5  "- Output - Exit 3 VFD Direction Reverse" %
%   N10:94/8  "- Output - Exit 3 VFD Accel Rate 1" %
%   N10:94/9  "- Output - Exit 3 VFD Accel Rate 2" %
%   N10:94/10  "- Output - Exit 3 VFD Decel Rate 1" %
%   N10:94/11  "- Output - Exit 3 VFD Decel Rate 2" %
%   N10:94/12  "- Output - Exit 3 VFD Reference Select 1" %
%   N10:94/13  "- Output - Exit 3 VFD Reference Select 2" %
%   N10:94/14  "- Output - Exit 3 VFD Reference Select 3" %
%   N10:95  "- Output - Exit 3 VFD Speed Command" %
%   B3:4/1  MANUAL  "Mode Manual" %
%   N51:4/1  "- HMI Input - Exit 2 Select" %

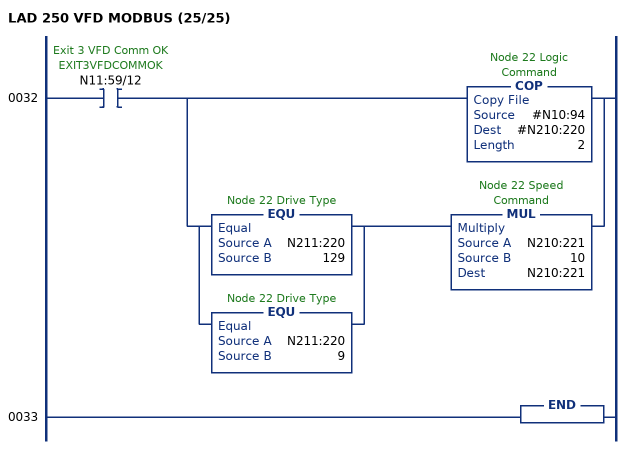
% Rung: 32 %
SOR XIC N11:59/12 BST COP #N10:94 #N210:220 2 NXB BST EQU N211:220 129 NXB EQU N211:220 9 BND MUL N210:221 10 N210:221 BND EOR
%   N11:59/12  EXIT3VFDCOMMOK  "Exit 3 VFD Comm OK" %
%   N10:94  "- Output - Exit 3 VFD Logic Command" %
%   N210:220  "Node 22 Logic Command" %
%   N211:220  "Node 22 Drive Type" %
%   N210:221  "Node 22 Speed Command" %
% Rung: 33 %
SOR END EOR

LADDER 251 "MODBUS"
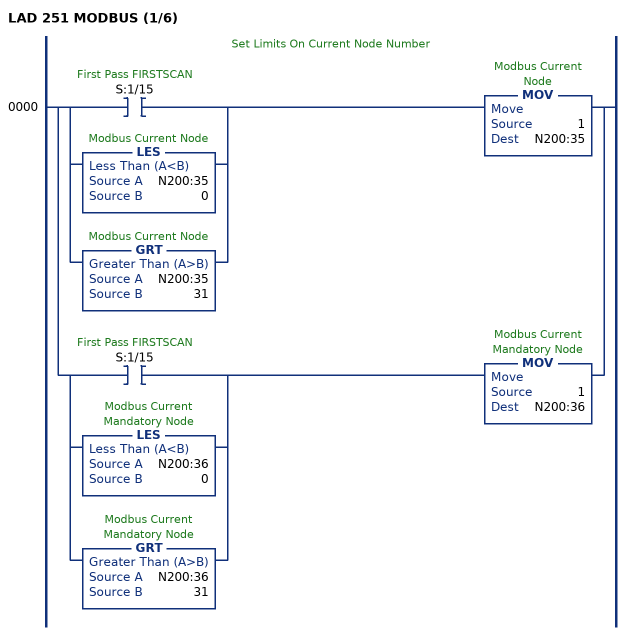
% Rung: 0 %
% Set Limits On Current Node Number %
SOR BST BST XIC S:1/15 NXB LES N200:35 0 NXB GRT N200:35 31 BND MOV 1 N200:35 NXB BST XIC S:1/15 NXB LES N200:36 0 NXB GRT N200:36 31 BND MOV 1 N200:36 BND EOR
%   S:1/15  FIRSTSCAN  "First Pass" %
%   N200:35  "Modbus Current Node" %
%   N200:36  "Modbus Current Mandatory Node" %

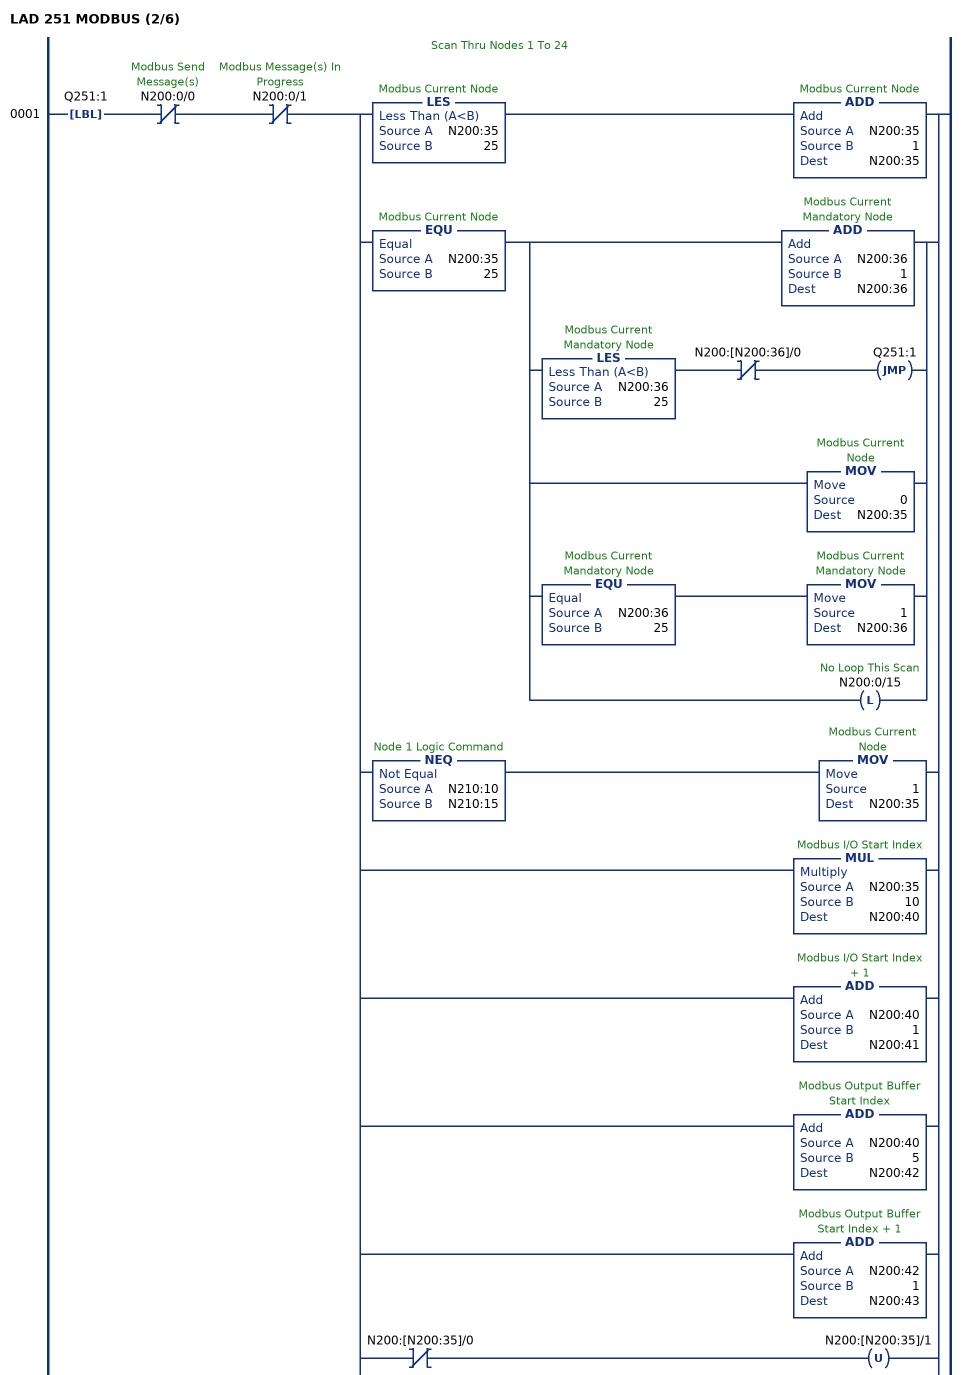

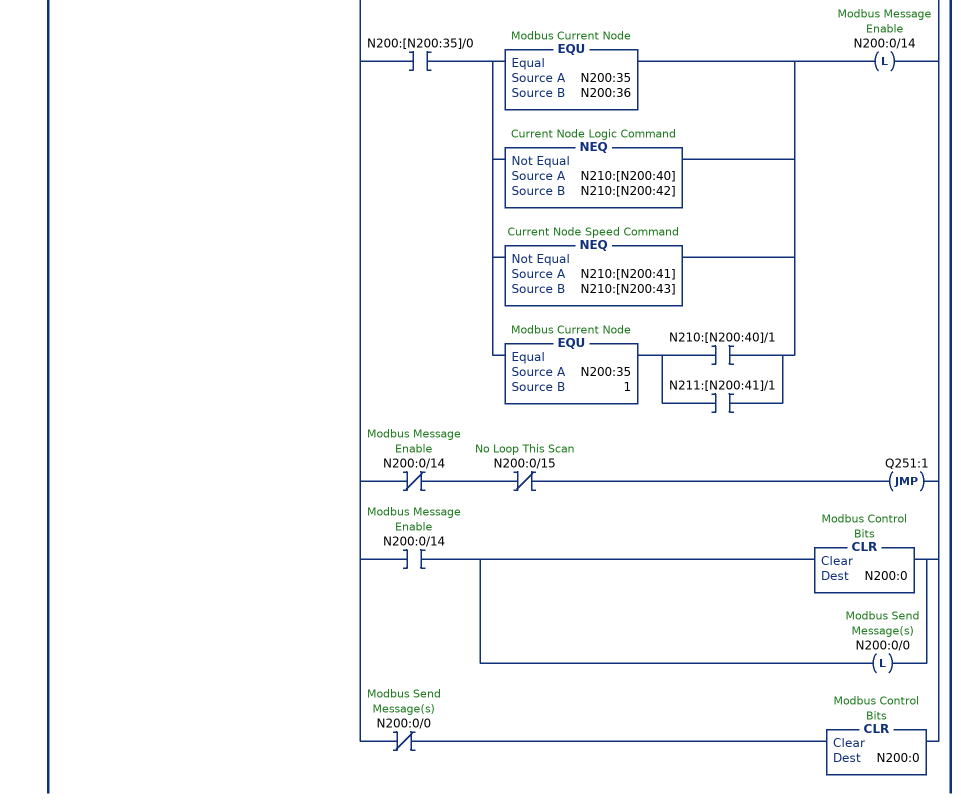
% Rung: 1 %
% Scan Thru Nodes 1 To 24 %
SOR LBL Q251:1 XIO N200:0/0 XIO N200:0/1 BST LES N200:35 25 ADD N200:35 1 N200:35 NXB EQU N200:35 25 BST ADD N200:36 1 N200:36 NXB LES N200:36 25 XIO N200:[N200:36]/0 JMP Q251:1 NXB MOV 0 N200:35 NXB EQU N200:36 25 MOV 1 N200:36 NXB OTL N200:0/15 BND NXB NEQ N210:10 N210:15 MOV 1 N200:35 NXB MUL N200:35 10 N200:40 NXB ADD N200:40 1 N200:41 NXB ADD N200:40 5 N200:42 NXB ADD N200:42 1 N200:43 NXB XIO N200:[N200:35]/0 OTU N200:[N200:35]/1 NXB XIC N200:[N200:35]/0 BST EQU N200:35 N200:36 NXB NEQ N210:[N200:40] N210:[N200:42] NXB NEQ N210:[N200:41] N210:[N200:43] NXB EQU N200:35 1 BST XIC N210:[N200:40]/1 NXB XIC N211:[N200:41]/1 BND BND OTL N200:0/14 NXB XIO N200:0/14 XIO N200:0/15 JMP Q251:1 NXB XIC N200:0/14 BST CLR N200:0 NXB OTL N200:0/0 BND NXB XIO N200:0/0 CLR N200:0 BND EOR
%   N200:0/0  "Modbus Send Message(s)" %
%   N200:0/1  "Modbus Message(s) In Progress" %
%   N200:35  "Modbus Current Node" %
%   N200:36  "Modbus Current Mandatory Node" %
%   N200:0/15  "No Loop This Scan" %
%   N210:10  "Node 1 Logic Command" %
%   N210:15  "Node 1 Spare" %
%   N200:40  "Modbus I/O Start Index" %
%   N200:41  "Modbus I/O Start Index + 1" %
%   N200:42  "Modbus Output Buffer Start Index" %
%   N200:43  "Modbus Output Buffer Start Index + 1" %
%   N210:[N200:40]  "Current Node Logic Command" %
%   N210:[N200:42]  "Current Node Logic Command" %
%   N210:[N200:41]  "Current Node Speed Command" %
%   N200:0/14  "Modbus Message Enable" %
%   N200:0  "Modbus Control Bits" %

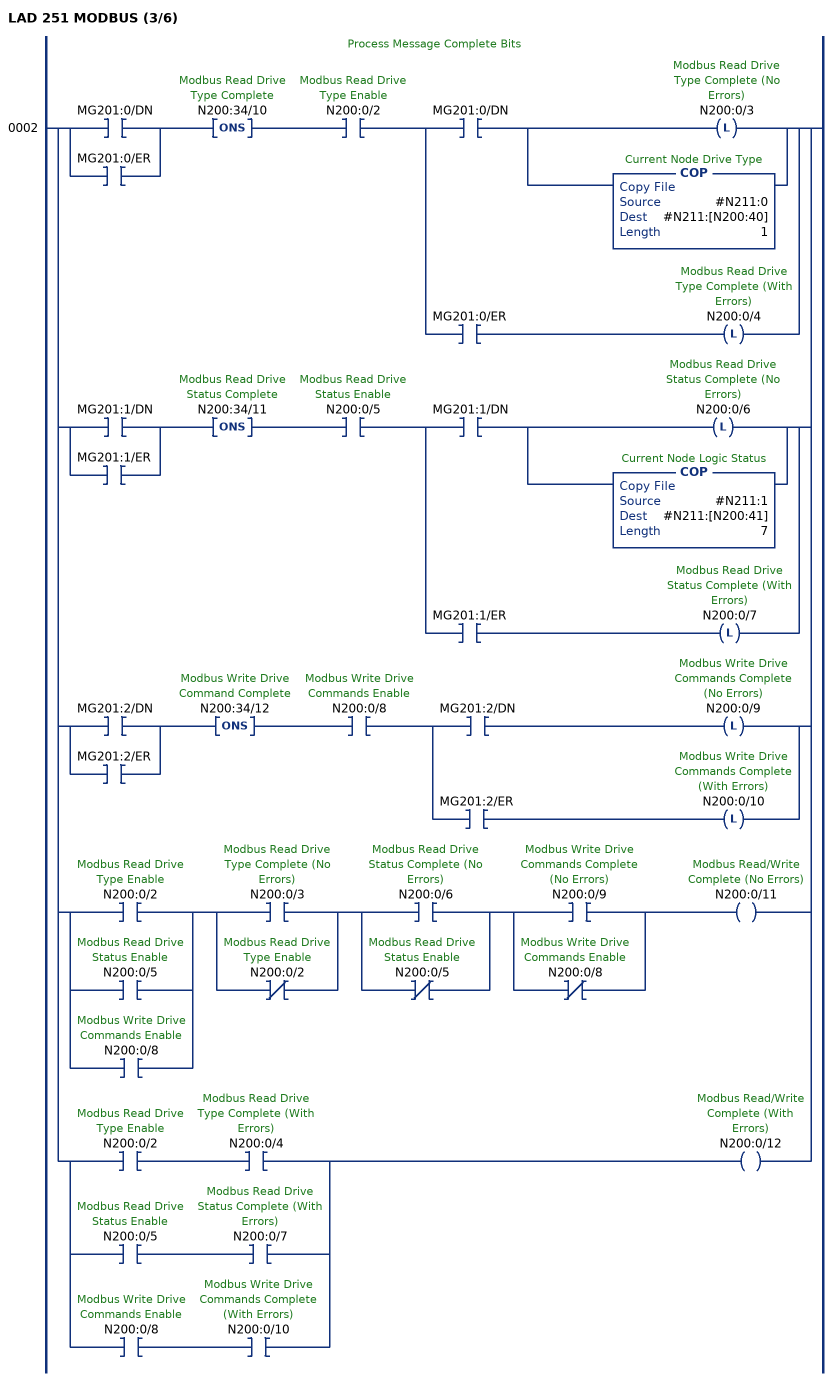
% Rung: 2 %
% Process Message Complete Bits %
SOR BST BST XIC MG201:0/DN NXB XIC MG201:0/ER BND ONS N200:34/10 XIC N200:0/2 BST XIC MG201:0/DN BST OTL N200:0/3 NXB COP #N211:0 #N211:[N200:40] 1 BND NXB XIC MG201:0/ER OTL N200:0/4 BND NXB BST XIC MG201:1/DN NXB XIC MG201:1/ER BND ONS N200:34/11 XIC N200:0/5 BST XIC MG201:1/DN BST OTL N200:0/6 NXB COP #N211:1 #N211:[N200:41] 7 BND NXB XIC MG201:1/ER OTL N200:0/7 BND NXB BST XIC MG201:2/DN NXB XIC MG201:2/ER BND ONS N200:34/12 XIC N200:0/8 BST XIC MG201:2/DN OTL N200:0/9 NXB XIC MG201:2/ER OTL N200:0/10 BND NXB BST XIC N200:0/2 NXB XIC N200:0/5 NXB XIC N200:0/8 BND BST XIC N200:0/3 NXB XIO N200:0/2 BND BST XIC N200:0/6 NXB XIO N200:0/5 BND BST XIC N200:0/9 NXB XIO N200:0/8 BND OTE N200:0/11 NXB BST XIC N200:0/2 XIC N200:0/4 NXB XIC N200:0/5 XIC N200:0/7 NXB XIC N200:0/8 XIC N200:0/10 BND OTE N200:0/12 BND EOR
%   N200:34/10  "Modbus Read Drive Type Complete" %
%   N200:0/2  "Modbus Read Drive Type Enable" %
%   N200:0/3  "Modbus Read Drive Type Complete (No Errors)" %
%   N211:0  "Current Node Drive Type" %
%   N211:[N200:40]  "Current Node Drive Type" %
%   N200:40  "Modbus I/O Start Index" %
%   N200:0/4  "Modbus Read Drive Type Complete (With Errors)" %
%   N200:34/11  "Modbus Read Drive Status Complete" %
%   N200:0/5  "Modbus Read Drive Status Enable" %
%   N200:0/6  "Modbus Read Drive Status Complete (No Errors)" %
%   N211:1  "Current Node Logic Status" %
%   N211:[N200:41]  "Current Node Logic Status" %
%   N200:41  "Modbus I/O Start Index + 1" %
%   N200:0/7  "Modbus Read Drive Status Complete (With Errors)" %
%   N200:34/12  "Modbus Write Drive Command Complete" %
%   N200:0/8  "Modbus Write Drive Commands Enable" %
%   N200:0/9  "Modbus Write Drive Commands Complete (No Errors)" %
%   N200:0/10  "Modbus Write Drive Commands Complete (With Errors)" %
%   N200:0/11  "Modbus Read/Write Complete (No Errors)" %
%   N200:0/12  "Modbus Read/Write Complete (With Errors)" %

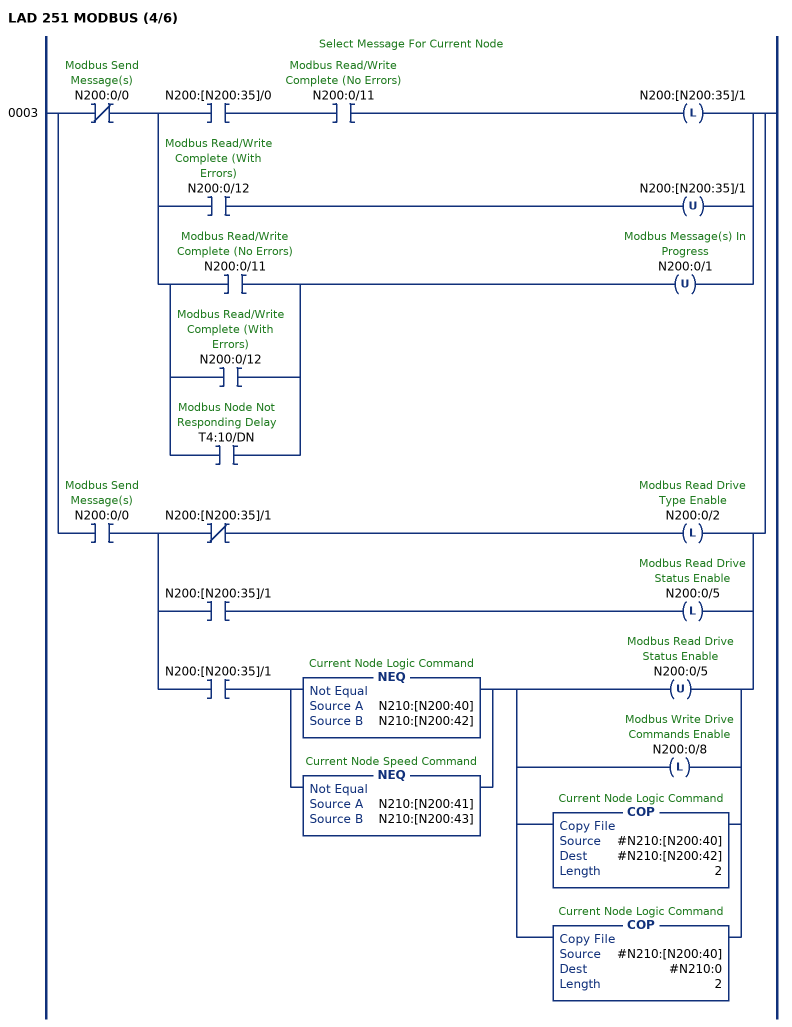
% Rung: 3 %
% Select Message For Current Node %
SOR BST XIO N200:0/0 BST XIC N200:[N200:35]/0 XIC N200:0/11 OTL N200:[N200:35]/1 NXB XIC N200:0/12 OTU N200:[N200:35]/1 NXB BST XIC N200:0/11 NXB XIC N200:0/12 NXB XIC T4:10/DN BND OTU N200:0/1 BND NXB XIC N200:0/0 BST XIO N200:[N200:35]/1 OTL N200:0/2 NXB XIC N200:[N200:35]/1 OTL N200:0/5 NXB XIC N200:[N200:35]/1 BST NEQ N210:[N200:40] N210:[N200:42] NXB NEQ N210:[N200:41] N210:[N200:43] BND BST OTU N200:0/5 NXB OTL N200:0/8 NXB COP #N210:[N200:40] #N210:[N200:42] 2 NXB COP #N210:[N200:40] #N210:0 2 BND BND BND EOR
%   N200:0/0  "Modbus Send Message(s)" %
%   N200:35  "Modbus Current Node" %
%   N200:0/11  "Modbus Read/Write Complete (No Errors)" %
%   N200:0/12  "Modbus Read/Write Complete (With Errors)" %
%   T4:10  "Modbus Node Not Responding Delay" %
%   N200:0/1  "Modbus Message(s) In Progress" %
%   N200:0/2  "Modbus Read Drive Type Enable" %
%   N200:0/5  "Modbus Read Drive Status Enable" %
%   N210:[N200:40]  "Current Node Logic Command" %
%   N200:40  "Modbus I/O Start Index" %
%   N210:[N200:42]  "Current Node Logic Command" %
%   N200:42  "Modbus Output Buffer Start Index" %
%   N210:[N200:41]  "Current Node Speed Command" %
%   N200:41  "Modbus I/O Start Index + 1" %
%   N200:43  "Modbus Output Buffer Start Index + 1" %
%   N200:0/8  "Modbus Write Drive Commands Enable" %
%   N210:0  "Current Node Logic Command" %

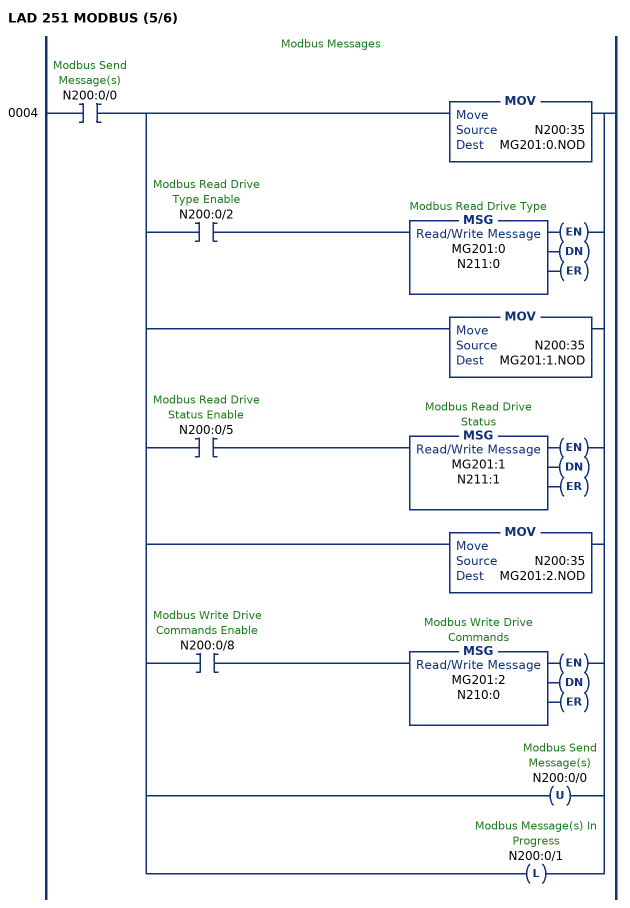
% Rung: 4 %
% Modbus Messages %
SOR XIC N200:0/0 BST MOV N200:35 MG201:0.NOD NXB XIC N200:0/2 MSG MG201:0 N211:0 NXB MOV N200:35 MG201:1.NOD NXB XIC N200:0/5 MSG MG201:1 N211:1 NXB MOV N200:35 MG201:2.NOD NXB XIC N200:0/8 MSG MG201:2 N210:0 NXB OTU N200:0/0 NXB OTL N200:0/1 BND EOR
%   N200:0/0  "Modbus Send Message(s)" %
%   N200:35  "Modbus Current Node" %
%   N200:0/2  "Modbus Read Drive Type Enable" %
%   MSG set-up: 03 Read Holding Registers (4xxxxx) | 0 | 1 | 16386 | N211:0 | 0 | 2 | 0 | CLIENT              :502 | 0 | 0 | ? %
%   MG201:0  "Modbus Read Drive Type" %
%   N211:0  "Current Node Drive Type" %
%   N200:0/5  "Modbus Read Drive Status Enable" %
%   MSG set-up: 03 Read Holding Registers (4xxxxx) | 0 | 7 | 8449 | N211:1 | 0 | 2 | 0 | CLIENT              :502 | 0 | 0 | ? %
%   MG201:1  "Modbus Read Drive Status" %
%   N211:1  "Current Node Logic Status" %
%   N200:0/8  "Modbus Write Drive Commands Enable" %
%   MSG set-up: 16 Write Multiple Registers (4xxxxx) | 0 | 2 | 8193 | N210:0 | 0 | 1 | 0 | CLIENT              :502 | 0 | 0 | ? %
%   MG201:2  "Modbus Write Drive Commands" %
%   N210:0  "Current Node Logic Command" %
%   N200:0/1  "Modbus Message(s) In Progress" %

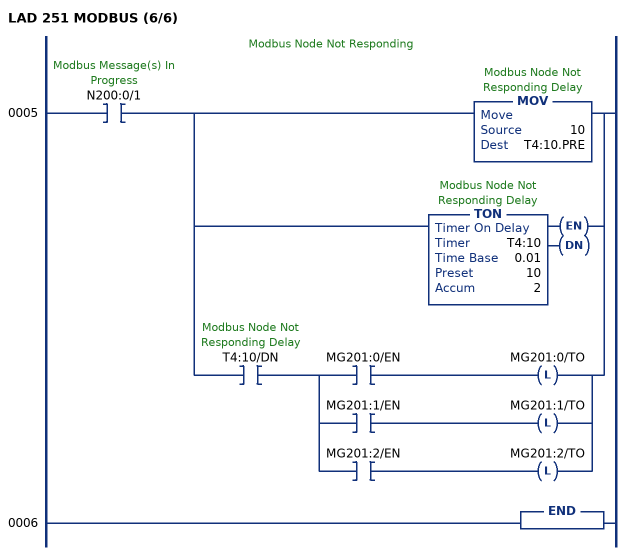
% Rung: 5 %
% Modbus Node Not Responding %
SOR XIC N200:0/1 BST MOV 10 T4:10.PRE NXB TON T4:10 0.01 10 2 NXB XIC T4:10/DN BST XIC MG201:0/EN OTL MG201:0/TO NXB XIC MG201:1/EN OTL MG201:1/TO NXB XIC MG201:2/EN OTL MG201:2/TO BND BND EOR
%   N200:0/1  "Modbus Message(s) In Progress" %
%   T4:10  "Modbus Node Not Responding Delay" %
% Rung: 6 %
SOR END EOR

LADDER 255 "HSC PFN"
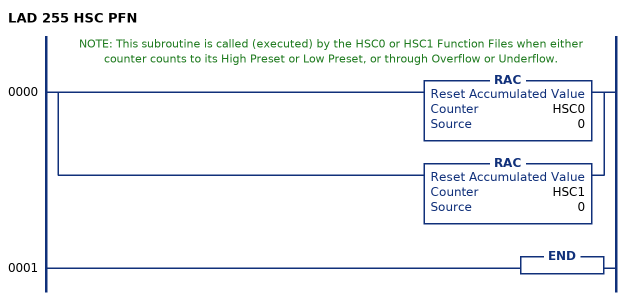
% Rung: 0 %
% NOTE: This subroutine is called (executed) by the HSC0 or HSC1 Function Files when either counter counts to its High Preset or Low Preset, or through Overflow or Underflow. %
SOR BST RAC HSC0 0 NXB RAC HSC1 0 BND EOR
% Rung: 1 %
SOR END EOR

OTHER DOCUMENTED ADDRESSES
  B3:0/0  "Lantech Ready to Accept"
  B3:0/1  "Lantech Ready to Receive Load"
  B3:0/2  WRAPPINGLOAD  "Lantech Load in Position to Wrap"
  B3:0/3  "Lantech Wrapping Load"
  B3:0/4  "Lantech Ready to Discharge"
  B3:0/5  "Lantech Wrapper OK"
  B3:4/15  "SLC09115 Specific bit"
  B3:5/8  "Load Has Blocked Exit Transition"
  B3:6/0  "CF Monitoring Turned On"
  B3:6/1  "Update CF Monitoring Toggled"
  B3:6/2  PROFILENEWONS  "Profile New Oneshot"
  B3:6/7  PROFILEUPDATEONS  "Profile Update oneshot"
  B3:6/8  PROFILESHIFTSTARTED  "Profile Delete Shift Started"
  B3:6/10  "Update Profile Edit Number"
  B3:6/11  "Profile Number Seeker Clear Oneshot"
  B3:6/12  "Update Number to Unique"
  B3:7/14  "20" Film On ONS"
  B3:7/15  "20" Film Off ONS"
  B3:8/14  "Wrap Time 2 Timer Update ONS"
  B3:8/15  WRAPRESTART  "Wrap Has Been Restarted"
  B3:9/3  "Bypass Next Load On ONS"
  B3:11/0  IOMESSAGING  "Messaging IO"
  B3:12/5  "Rotation Auto Rotate To Home"
  B3:12/6  "Rotation Auto Rotate To 90°"
  B3:13/4  "Film Carriage Auto Raise To Home Position"
  B3:13/11  CARRIAGEHOME  "Film Carriage At Home"
  B3:14/13  "Top Blink Count ONS"
  B3:14/14  "Partial Top Layer Cancel"
  B3:15/4  "Wipe Arm Stage 2 Auto Extend"
  B3:15/5  "Wipe Arm Stage 2 Auto Extend Complete"
  B3:15/6  "Wipe Arm Stage 2 Auto Retract"
  B3:15/7  "Wipe Arm Stage 2 Auto Retract Complete"
  B3:15/8  WIPERETRACTED2  "Wipe Arm Retracted"
  B3:18/10  "Load Stabilizer Auto Raise"
  B3:18/11  "Load Stabilizer Auto Raise Complete"
  B3:26/0  "Infeed 4 Conveyor Stage Load"
  B3:26/1  "Infeed 4 Conveyor Stage Load Memory"
  B3:26/2  "Infeed 4 Conveyor Advance Interjected Load"
  B3:26/3  "Infeed 4 Conveyor Advance Interjected Load Memory"
  B3:26/4  "Infeed 4 Conveyor Dischage Load"
  B3:26/5  "Infeed 4 Conveyor Dischage Load Memory"
  B3:26/6  "Infeed 4 Conveyor Clear Of Exiting Load"
  B3:26/9  "Infeed 4 Conveyor"
  B3:26/10  "Infeed 4 Conveyor Watchdog Reset ONS"
  B3:26/11  "Infeed 4 Conveyor Jog Selected"
  B3:26/12  "Infeed 4 Conveyor Select On ONS"
  B3:26/13  "Infeed 4 Conveyor Select Off ONS"
  B3:26/14  "Infeed 4 Conveyor Update Tracking ONS"
  B3:26/15  "Infeed 4 Conveyor Clear Tracking ONS"
  B3:27/4  "Infeed 3 Conveyor Dischage Load"
  B3:27/5  "Infeed 3 Conveyor Dischage Load Memory"
  B3:27/9  "Infeed 3 Conveyor"
  B3:27/10  "Infeed 3 Conveyor Watchdog Reset ONS"
  B3:27/12  "Infeed 3 Conveyor Select On ONS"
  B3:27/13  "Infeed 3 Conveyor Select Off ONS"
  B3:27/15  "Infeed 3 Conveyor Clear Tracking ONS"
  B3:28/4  "Infeed 2 Conveyor Dischage Load"
  B3:28/5  "Infeed 2 Conveyor Dischage Load Memory"
  B3:28/9  "Infeed 2 Conveyor"
  B3:28/10  "Infeed 2 Conveyor Watchdog Reset ONS"
  B3:28/12  "Infeed 2 Conveyor Select On ONS"
  B3:28/13  "Infeed 2 Conveyor Select Off ONS"
  B3:28/15  "Infeed 2 Conveyor Clear Tracking ONS"
  B3:29/4  "Infeed 1 Conveyor Dischage Load"
  B3:29/5  "Infeed 1 Conveyor Dischage Load Memory"
  B3:29/9  "Infeed 1 Conveyor"
  B3:29/10  "Infeed 1 Conveyor Watchdog Reset ONS"
  B3:29/12  "Infeed 1 Conveyor Select On ONS"
  B3:29/13  "Infeed 1 Conveyor Select Off ONS"
  B3:29/15  "Infeed 1 Conveyor Clear Tracking ONS"
  B3:30/2  "Wrap Zone Conveyor Advance Interjected Load"
  B3:30/3  "Wrap Zone Conveyor Advance Interjected Load Memory"
  B3:30/7  "Wrap Zone Conveyor Clear Of Fork Truck"
  B3:30/8  "Wrap Zone Conveyor Release Incoming Load Because Truck Was Detected While Staging"
  B3:30/11  READYTODISCHARGE  "Wrap Zone Conveyor Conveyor Load Discharging"
  B3:31/2  "Exit 1 Conveyor Advance Interjected Load"
  B3:31/3  "Exit 1 Conveyor Advance Interjected Load Memory"
  B3:31/8  "Exit 1 Conveyor Release Incoming Load Because Truck Was Detected While Staging"
  B3:31/9  "Exit 1 Conveyor"
  B3:31/11  "Exit 1 Conveyor Discharge Load Anticipation"
  B3:31/12  "Exit 1 Conveyor Discharge Load Anticipation ONS"
  B3:31/13  "Exit 1 Conveyor Discharge Load Anticipation Oneshot"
  B3:32/2  "Exit 2 Conveyor Advance Interjected Load"
  B3:32/3  "Exit 2 Conveyor Advance Interjected Load Memory"
  B3:32/8  "Exit 2 Conveyor Release Incoming Load Because Truck Was Detected While Staging"
  B3:32/9  "Exit 2 Conveyor"
  B3:32/11  "Exit 2 Conveyor Discharge Anticipation"
  B3:32/12  "Exit 2 Conveyor Discharge Load Anticipation ONS"
  B3:32/13  "Exit 2 Conveyor Discharge Load Anticipation Oneshot"
  B3:33/2  "Exit 3 Conveyor Advance Interjected Load"
  B3:33/3  "Exit 3 Conveyor Advance Interjected Load Memory"
  B3:33/8  "Exit 3 Conveyor Release Incoming Load Because Truck Was Detected While Staging"
  B3:33/9  "Exit 3 Conveyor"
  B3:33/11  "Exit 3 Conveyor Discharge Anticipation"
  B3:33/12  "Exit 3 Conveyor Discharge Load Anticipation ONS"
  B3:33/13  "Exit 3 Conveyor Discharge Load Anticipation Oneshot"
  B3:34/2  "Exit 4 Conveyor Advance Interjected Load"
  B3:34/3  "Exit 4 Conveyor Advance Interjected Load Memory"
  B3:34/4  "Exit 4 Conveyor Dischage Load"
  B3:34/5  "Exit 4 Conveyor Dischage Load Memory"
  B3:34/6  "Exit 4 Conveyor Clear Of Exiting Load"
  B3:34/7  "Exit 4 Conveyor Clear Of Fork Truck"
  B3:34/8  "Exit 4 Conveyor Release Incoming Load Because Truck Was Detected While Staging"
  B3:34/9  "Exit 4 Conveyor"
  B3:34/10  "Exit 4 Conveyor Watchdog Reset ONS"
  B3:34/11  "Exit 4 Conveyor Jog Selected"
  B3:34/12  "Exit 4 Conveyor Select On ONS"
  B3:34/13  "Exit 4 Conveyor Select Off ONS"
  B3:34/14  "Exit 4 Conveyor Update Tracking ONS"
  B3:34/15  "Exit 4 Conveyor Clear Tracking ONS"
  B3:35/0  "Wrap Zone Conveyor Conveyor Load Discharged"
  B3:45/4  "Load Lift Film Clamp Retract Reset"
  B3:45/5  "Load Lift Film Clamp Extend Reset"
  B3:50/2  MENUCLOSEBYPASSOFF  "Menu Auto Bypass Next Off Close ONS"
  B3:50/3  MENUCLOSEBYPASSON  "Menu Auto Bypass Next On Close ONS"
  B3:50/14  "End Of More Help"
  B3:50/15  "HMI More Help One Shot"
  B3:52/2  "Film Break ONS"
  B3:70/0  "Load Guardian"
  B3:99/0  INTERFACERELAY  "Project Bit SLA009179 Specific Customer Interface"
  B3:106/0  "Update Customer Number to Edit Number ONS"
  B3:106/3  "Profile Delete Index Initialize Oneshot"
  B3:106/4  "Profile Copy Deleted Plus One Oneshot"
  B3:106/10  "Regenerate Profile Edit Number HMI Input From Internal Value"
  B12:2/11  "Low Film Disable On ONS"
  B12:2/12  "Low Film Disable Off ONS"
  B12:4/6  "Mode Runout Mode Enable On ONS"
  B12:4/7  "Mode Runout Mode Enable Off ONS"
  B12:4/13  "Runout Wrap Complete"
  B12:4/15  "Runout Top Of Load Position"
  B12:9/8  WRAPSLOW  "Wrap Slow"
  B12:12/9  "Rotation Auto Tune Selected On ONS"
  B12:12/10  "Rotation Auto Tune Selected Off ONS"
  B12:13/9  "Film Carriage Auto Tune Selected On ONS"
  B12:13/10  "Film Carriage Auto Tune Selected Off ONS"
  B12:14/9  "Metered Pre-Stretch Auto Tune Selected On ONS"
  B12:14/10  "Metered Pre-Stretch Auto Tune Selected Off ONS"
  B12:15/4  WIPEARMNOWARNINGS  "Wipe Arm No Warnings"
  B12:18/0  STABILIZERNOFAULTS  "Load Stabilizer No Faults"
  B12:18/3  STABILIZERNOWARNINGS  "Load Stabilizer No Warnings"
  B12:18/4  STABILIZERHOMING  "Load Stabilizer Homing"
  B12:19/7  "TSD Dispense Indicator ONS"
  B13:2/1  "Conveyors Reverse Select"
  B13:30/15  "Wrap Zone Conveyor Load Has Blocked Exit Transition"
  C5:0  "Counter Test"
  DFILE:0  "OUTPUT"
  DFILE:1  "INPUT"
  DFILE:2  "STATUS"
  DFILE:3  "BINARY"
  DFILE:4  "TIMER"
  DFILE:5  "COUNTER"
  DFILE:6  "CONTROL"
  DFILE:7  "INTEGER"
  DFILE:8  "FLOAT"
  DFILE:9  "C FORCE"
  DFILE:10  "OUTPUT MAP"
  DFILE:11  "INPUT MAP"
  DFILE:12  "BINARY"
  DFILE:13  "BINARY"
  DFILE:14  "LG"
  DFILE:15  "OPTIONS"
  DFILE:16  "SECURITY"
  DFILE:17  "MESSAGING"
  DFILE:18  "LINC STR"
  DFILE:19  "TRACKING"
  DFILE:20  "FILM"
  DFILE:21  "PROFILES"
  DFILE:22  "PROF CALCS"
  DFILE:25  "LONG"
  DFILE:26  "ICF MAP"
  DFILE:28  "TEMP PROF Temporary Profile"
  DFILE:29  "INPUT PROF HMI Input Profile"
  DFILE:30  "DEFAULT Default Profile"
  DFILE:31  "PROFILE 1 Profile 1"
  DFILE:32  "PROFILE 2 Profile 2"
  DFILE:33  "PROFILE 3 Profile 3"
  DFILE:34  "PROFILE 4 Profile 4"
  DFILE:35  "PROFILE 5 Profile 5"
  DFILE:36  "PROFILE 6 Profile 6"
  DFILE:37  "PROFILE 7 Profile 7"
  DFILE:38  "PROFILE 8 Profile 8"
  DFILE:39  "PROFILE 9 Profile 9"
  DFILE:40  "CURRENT"
  DFILE:41  "PROFILECAL"
  DFILE:42  "PROFILENUM"
  DFILE:43  "PROFILESTR"
  DFILE:45  "PROFILES"
  DFILE:46  "PROFILES"
  DFILE:48  "PROF WARN"
  DFILE:49  "PROFWARNCH"
  DFILE:50  "HMI OUTPUT"
  DFILE:51  "HMI INPUT"
  DFILE:60  "FAULT Fault Overflow Trap"
  DFILE:80  "E_NET_IN"
  DFILE:81  "E_NET_OUT"
  DFILE:92  "WARNCOPY"
  DFILE:93  "WARN BUF WARNING BUFFER"
  DFILE:94  "WARN LIST WARNINGS LIST"
  DFILE:95  "WARNINGS WARNINGS"
  DFILE:96  "ALARMCOPY"
  DFILE:97  "ALARM BUF ALARMS BUFFER"
  DFILE:98  "ALARM ACT ALARM ACTIVE"
  DFILE:99  "ALARM LIST ALARM LIST"
  DFILE:100  "ALARMS"
  DFILE:101  "MAINT"
  DFILE:102  "MAINT1"
  DFILE:103  "MAINT2"
  DFILE:110  "CDATA Load Containment Dat a"
  DFILE:111  "CDATA1 Load Containment Dat a Array 1"
  DFILE:112  "CDATA2 Load Containment Dat a Array 2"
  DFILE:115  "PDATA Production Data Cont rol"
  DFILE:116  "PDATA1 Production Data Arra y 1"
  DFILE:117  "PDATA2 Production Data Arra y 2"
  DFILE:118  "PDATA3 Production Data Arra y 3"
  DFILE:119  "PDATALPH Production Data Load s/Breaks Per Hour"
  DFILE:120  "PDATALPR Production Data Load s Per Film Roll"
  DFILE:121  "PDATARPR Production Data Revo lutions Per Film Rol ls"
  DFILE:122  "PDATACHART Production Data Char t"
  DFILE:125  "PDATAT Production Data Time rs"
  DFILE:150  "LINC DINT"
  DFILE:151  "LINC STR"
  DFILE:200  "MODBUS"
  DFILE:201  "MODBUS MSG"
  DFILE:210  "MODBUS OUT"
  DFILE:211  "MODBUS IN"
  DFILE:255  "VERSION"
  F8:1  "Calculation Temp 2"
  F8:2  "Overlap Up During Overwrap Memory"
  F8:18  "TEST"
  F8:23  REVTIMEUP  "Revolution Time Up"
  F8:24  REVTIMEDOWN  "Revolution Time Down"
  F8:26  "Overwrap Rev Time Memory"
  F8:28  LAYERSTEMP  "Modulo For Layers (Remainder)"
  F8:35  CFINCREMENTALLAST
  F8:38  CFCALIBRATIONMUL  "Calibration Multiplier"
  F8:40  "Overwrap Partial Top"
  F22:8  "Value Used For Layers Calculations"
  F22:11  "Overwrap Minimum Based On Current Carriage Speed"
  I:0.0/5  "RESERVED (HSC:1 Count B)"
  I:0.0/6  "RESERVED (HSC:1 Z Reset)"
  I:0.0/7  "RESERVED (HSC:1 Hold)"
  I:2.0/0  "Upstream "Bypass Request""
  I:2.0/1  "Film Hoist At Retract"
  I:2.0/2  "Wrap Zone "Overtravel" Is Clear"
  I:2.0/3  "Wrap Zone "Undertravel" Is Clear"
  I:2.0/4  "Infeed Transition Is Clear"
  I:2.0/5  "Exit Transition Is Clear"
  I:2.0/6  "Short Load Is Clear"
  I:2.0/7  "Infeed Forklift Is Clear"
  I:2.0/8  "Exit Forklift Is Clear"
  I:2.0/9  "Infeed 3 Is Clear"
  I:2.0/10  "Infeed 2 Is Clear"
  I:2.0/11  "Infeed 1 Is Clear"
  I:2.0/12  "Wrap Zone Is Clear"
  I:2.0/13  "Exit 1 Is Clear"
  I:2.0/14  "Exit 2 Is Clear"
  I:2.0/15  "Exit 3 Is Clear"
  I:6.0/0  "Not Used"
  I:6.0/1  "Not Used"
  I:6.0/2  "Not Used"
  I:6.0/3  "Not Used"
  I:6.0/4  "Not Used"
  I:6.0/5  "TSD Not Used"
  I:6.0/6  "TSD Elevator Overload / Fault"
  I:6.0/7  "TSD Elevator Belt At Tension"
  I:6.0/8  "TSD Film Is Low"
  I:6.0/9  "TSD Elevator Not At Up"
  I:6.0/10  "TSD Elevator At Down"
  I:6.0/11  "TSD Cutter Wire Fault"
  I:6.0/12  "TSD Cutter Wire At Tension"
  I:6.0/13  "TSD Load Height Is Clear 1"
  I:6.0/14  "TSD Load Height Is Clear 2"
  I:6.0/15  "TSD Short Load Is Clear"
  L25:9  "Film Dispensed Per Revolution RS2 Count Memory"
  L150:0  "LINC Bools"
  L150:0/0  "LINC Comms Established"
  L150:0/1  "LINC Comm Ok"
  L150:0/2  "LINC OS Reset Request"
  L150:1  "LINCBars Signal Strength"
  L150:2  "LINC Comm Check"
  L150:3  "LINC Heartbeat"
  L150:4  "LINC RSSI"
  N7:3  "HMI Edit Number Memory"
  N7:8  "Top Wraps Adjust Memory"
  N7:9  "Bottom Wraps Adjust Memory"
  N7:20  "Wrap Profile Selected Index"
  N7:21  "Wrap Profile Edit Index"
  N7:22  "Wrap Profile Copy Source Index"
  N7:23  "Wrap Profile Copy Destination Index"
  N7:24  "Wrap Profile Edit Check"
  N7:25  "Profile Containment Force Requirement (HMI Input) Memory"
  N7:26  "Layers Whole Memory"
  N7:27  "Rotation Max Speed Memory"
  N7:28  "Rotation Up Speed Memory"
  N7:34  "Rotation Revolution Time Memory"
  N7:36  "Pallet-Grip Released Position (10 = 10 Inches)"
  N7:38  "Ladder Stagger High Priority (Every 2 Scans)"
  N7:39  "Ladder Stagger Low Priority (Every 6 Scans)"
  N7:43  "MPS Current Payout Memory (100 = 100%)"
  N7:44  "Carriage Position Memory"
  N7:45  "Film Width at Roll Memory"
  N7:46  "Overwrap FDS Speed Memory"
  N7:64  "Scan Time Added (ms)"
  N7:78  "Film Carriage Film Width With Pallet-Grip"
  N7:79  "Film Carriage Film Width Loss Due To Pallet-Grip (100 = 10.0 Inches)"
  N7:86  "Film Carriage Home Speed (25 = 2.5 IPS)"
  N7:94  OVERWRAPOFFSET  "Overwrap Offset At Current Speed"
  N7:96  "Pallet Grip Offset"
  N7:99  "Film Carriage Encoder Current Quad State"
  N7:105  "Film Thickness Difference Memory"
  N7:110  "CF Last Load Raw"
  N7:111  "CF Last Load"
  N7:113  LINE1INPUTDIFFERENCE  "Difference Between Input Wrap Force And Minimum Wrap Force For Line 1"
  N7:114  WFLINE1RANGE  "Range Of Wrap Forces On Line 1"
  N7:115  "Force To Load Check"
  N7:116  LINE2INPUTDIFFERENCE  "Difference Between Input Wrap Force And Minimum Wrap Force For Line 2"
  N7:117  WFLINE2RANGE  "Range Of Wrap Forces On Line 2"
  N7:120  "Layers Check"
  N7:121  FORCELOADMIN  "Force At Load Min Value"
  N7:122  BOTTOMWRAPS  "Bottom Wraps"
  N7:123  TOPWRAPS  "Top Wraps"
  N7:125  MINLAYERSCHECK  "Min Layers To Meet Current Containment Force Requirement Check For Half Layer"
  N7:127  "Layers Whole Truncation"
  N7:129  "CF Req Check"
  N7:130  "Min Layers To Meet Current Containment Force Requirement"
  N7:132  WRAPFORCERANGE  "Wrap Force Range"
  N7:133  TOPADJUST  "Top Wrap Count Adjustment"
  N7:134  WRAPFORCEMAX  "Maximum Wrap Force (0 = 120% Payout 15 = 90% Payout)"
  N7:135  "Layers Check (HMI Input)"
  N7:136  "Overwrap Rotation Speed (RPM)"
  N7:138  "Layers Calc Truncation"
  N7:139  "Layers Calc Truncation"
  N7:140  FDSSTOPPINGMIN  "Minimum Distance FDS Will Travel After Height Sensor Is Clear"
  N7:141  FDSSTOPPINGMAX  "Maximum Distance FDS Will Travel After Height Sensor Is Clear"
  N7:142  FDSSPEEDMAX  "FDS Speed Percentage Maximum"
  N7:143  FDSSTOPPINGRANGE  "Range Of Distance FDS Will Travel After Height Sensor Is Clear"
  N7:149  "Profile Indirect Address Temp"
  N7:150  PROFILENEWINDEX  "Add a Profile Index"
  N7:151  PROFILECOPYSOURCE  "Wrap Profile Copy Source"
  N7:152  PROFILESHIFTINDEX  "Profile Delete Shift Index"
  N7:158  "Indirect Address To Active Profile"
  N7:159/0  PROFILENEW  "Add a Profile"
  N7:159/1  PROFILEUPDATE  "Update HMI Wrap Profile Values"
  N7:160  "Top Blink Count"
  N7:162  "Wrap Time Top Wraps"
  N7:163  "Wrap Time From Last Revolution"
  N7:166  REVSFROMDOWN  "Revolutions From Down"
  N7:167  WRAPTIMEDOWN  "Wrap Time Down"
  N7:168  "Wrap Time Up"
  N7:195  "IP ADDRESS TEMP INTEGER #2"
  N7:197/0  "Temp Bit This rung may need to be filtered out due to scan time."
  N10:18/0  STABILIZERRAISE  "- Output - Stabilizer Raise"
  N10:18/1  STABILIZERLOWER  "- Output - Stabilizer Lower"
  N10:30/1  WRAPZONERVS  "- Output - Wrap Zone Conveyor Reverse"
  N10:56  "- Output - Rotation Last Command (1000 = 100.0%)"
  N10:59  "- Output - TSD Dispense Last Command (1000 = 100.0%)"
  N10:60/2  "- Output - Rotation VFD Jog"
  N10:60/6  "- Output - Rotation VFD Not Used"
  N10:60/7  "- Output - Rotation VFD Not Used"
  N10:60/15  "- Output - Rotation VFD Not Used"
  N10:62/2  "- Output - Film Carriage VFD Jog"
  N10:62/6  "- Output - Film Carriage VFD Not Used"
  N10:62/7  "- Output - Film Carriage VFD Not Used"
  N10:62/15  "- Output - Film Carriage VFD Not Used"
  N10:64/2  "- Output - MPS VFD Jog"
  N10:64/6  "- Output - MPS VFD Not Used"
  N10:64/7  "- Output - MPS VFD Not Used"
  N10:64/15  "- Output - MPS VFD Not Used"
  N10:66/2  "- Output - Wrap Zone VFD Jog"
  N10:66/6  "- Output - Wrap Zone VFD Not Used"
  N10:66/7  "- Output - Wrap Zone VFD Not Used"
  N10:66/15  "- Output - Wrap Zone VFD Not Used"
  N10:70/2  "- Output - Infeed 1 VFD Jog"
  N10:70/6  "- Output - Infeed 1 VFD Not Used"
  N10:70/7  "- Output - Infeed 1 VFD Not Used"
  N10:70/15  "- Output - Infeed 1 VFD Not Used"
  N10:72/2  "- Output - Infeed 2 VFD Jog"
  N10:72/6  "- Output - Infeed 2 VFD Not Used"
  N10:72/7  "- Output - Infeed 2 VFD Not Used"
  N10:72/15  "- Output - Infeed 2 VFD Not Used"
  N10:74/2  "- Output - Infeed 3 VFD Jog"
  N10:74/6  "- Output - Infeed 3 VFD Not Used"
  N10:74/7  "- Output - Infeed 3 VFD Not Used"
  N10:74/15  "- Output - Infeed 3 VFD Not Used"
  N10:90/2  "- Output - Exit 1 VFD Jog"
  N10:90/6  "- Output - Exit 1 VFD Not Used"
  N10:90/7  "- Output - Exit 1 VFD Not Used"
  N10:90/15  "- Output - Exit 1 VFD Not Used"
  N10:92/2  "- Output - Exit 2 VFD Jog"
  N10:92/6  "- Output - Exit 2 VFD Not Used"
  N10:92/7  "- Output - Exit 2 VFD Not Used"
  N10:92/15  "- Output - Exit 2 VFD Not Used"
  N10:94/2  "- Output - Exit 3 VFD Jog"
  N10:94/6  "- Output - Exit 3 VFD Not Used"
  N10:94/7  "- Output - Exit 3 VFD Not Used"
  N10:94/15  "- Output - Exit 3 VFD Not Used"
  N11:1/11  "- Input - Customer Gate Switch is Active"
  N11:1/12  "- Input - Customer Infeed Light Curtain OK"
  N11:1/13  "- Input - Customer Exit Light Curtain OK"
  N11:12/1  ROTATION90  "- Input - Rotation At 90°"
  N11:18/0  STABILIZERUP  "- Input - Stabilizer Up"
  N11:18/1  STABILIZERONLOAD  "- Input - Stabilizer On Load"
  N11:18/2  STABILIZERCLEAR  "- Input - Stabilizer Height Sensing Clear"
  N11:18/3  "- Input - Stabilizer Motor Overload Tripped"
  N11:27/1  INFEED3UNDERTRAVEL  "- Input - Infeed 3 Undertravel Clear"
  N11:27/2  INFEED3OVERTRAVEL  "- Input - Infeed 3 Overtravel Clear"
  N11:28/1  INFEED2UNDERTRAVEL  "- Input - Infeed 2 Undertravel Clear"
  N11:28/2  INFEED2OVERTRAVEL  "- Input - Infeed 2 Overtravel Clear"
  N11:29/1  INFEED1UNDERTRAVEL  "- Input - Infeed 1 Undertravel Clear"
  N11:29/2  INFEED1OVERTRAVEL  "- Input - Infeed 1 Overtravel Clear"
  N11:30/4  WRAPZONETRUCKCLEAR  "- Input - Wrap Zone Truck Detection Clear"
  N11:31/1  EXIT1UNDERTRAVEL  "- Input - Exit 1 Undertravel Clear"
  N11:31/2  EXIT1OVERTRAVEL  "- Input - Exit 1 Overtravel Clear"
  N11:32/1  EXIT2UNDERTRAVEL  "- Input - Exit 2 Undertravel Clear"
  N11:32/2  EXIT2OVERTRAVEL  "- Input - Exit 2 Overtravel Clear"
  N11:33/1  EXIT3UNDERTRAVEL  "- Input - Exit 3 Undertravel Clear"
  N11:33/2  EXIT3OVERTRAVEL  "- Input - Exit 3 Overtravel Clear"
  N11:41/2  "- Input - Wrap Zone Conveyor Running"
  N11:41/3  LOAD  "- Input - Load in Position to be Wrapped"
  N11:41/4  "- Input - Load In Position"
  N11:41/5  "- Input - Exit Conveyor Running"
  N11:54  TSDFEEDBACK  "Input TSD Dispense Speed Feedback (1000 = 100.0%)"
  N11:60/0  "- Input - Rotation VFD Ready"
  N11:60/2  "- Input - Rotation VFD Command Direction Forward"
  N11:60/3  "- Input - Rotation VFD Actual Direction Forward"
  N11:60/6  "- Input - Rotation VFD Alarm Present"
  N11:60/9  "- Input - Rotation VFD Main Frequency Controlled By Comm"
  N11:60/10  "- Input - Rotation VFD Operation Command Controlled By Comm"
  N11:60/11  "- Input - Rotation VFD Parameters Locked"
  N11:60/12  "- Input - Rotation VFD Digital Input 1 Status"
  N11:60/13  "- Input - Rotation VFD Digital Input 2 Status"
  N11:60/14  "- Input - Rotation VFD Digital Input 3 Status"
  N11:60/15  "- Input - Rotation VFD Digital Input 4 Status"
  N11:62/0  "- Input - Film Carriage VFD Ready"
  N11:62/2  "- Input - Film Carriage VFD Command Direction Forward"
  N11:62/3  "- Input - Film Carriage VFD Actual Direction Forward"
  N11:62/4  "- Input - Film Carriage VFD Accelerating"
  N11:62/5  "- Input - Film Carriage VFD Decelerating"
  N11:62/6  "- Input - Film Carriage VFD Alarm Present"
  N11:62/9  "- Input - Film Carriage VFD Main Frequency Controlled By Comm"
  N11:62/10  "- Input - Film Carriage VFD Operation Command Controlled By Comm"
  N11:62/11  "- Input - Film Carriage VFD Parameters Locked"
  N11:62/12  "- Input - Film Carriage VFD Digital Input 1 Status"
  N11:62/13  "- Input - Film Carriage VFD Digital Input 2 Status"
  N11:62/14  "- Input - Film Carriage VFD Digital Input 3 Status"
  N11:62/15  "- Input - Film Carriage VFD Digital Input 4 Status"
  N11:64/0  "- Input - MPS VFD Ready"
  N11:64/1  "- Input - MPS VFD Active"
  N11:64/2  "- Input - MPS VFD Command Direction Forward"
  N11:64/3  "- Input - MPS VFD Actual Direction Forward"
  N11:64/4  "- Input - MPS VFD Accelerating"
  N11:64/5  "- Input - MPS VFD Decelerating"
  N11:64/6  "- Input - MPS VFD Alarm Present"
  N11:64/8  "- Input - MPS VFD At Speed"
  N11:64/9  "- Input - MPS VFD Main Frequency Controlled By Comm"
  N11:64/10  "- Input - MPS VFD Operation Command Controlled By Comm"
  N11:64/11  "- Input - MPS VFD Parameters Locked"
  N11:64/12  "- Input - MPS VFD Digital Input 1 Status"
  N11:64/13  "- Input - MPS VFD Digital Input 2 Status"
  N11:64/14  "- Input - MPS VFD Digital Input 3 Status"
  N11:64/15  "- Input - MPS VFD Digital Input 4 Status"
  N11:66/0  "- Input - Wrap Zone VFD Ready"
  N11:66/2  "- Input - Wrap Zone VFD Command Direction Forward"
  N11:66/3  "- Input - Wrap Zone VFD Actual Direction Forward"
  N11:66/4  "- Input - Wrap Zone VFD Accelerating"
  N11:66/5  "- Input - Wrap Zone VFD Decelerating"
  N11:66/6  "- Input - Wrap Zone VFD Alarm Present"
  N11:66/8  "- Input - Wrap Zone VFD At Speed"
  N11:66/9  "- Input - Wrap Zone VFD Main Frequency Controlled By Comm"
  N11:66/10  "- Input - Wrap Zone VFD Operation Command Controlled By Comm"
  N11:66/11  "- Input - Wrap Zone VFD Parameters Locked"
  N11:66/12  "- Input - Wrap Zone VFD Digital Input 1 Status"
  N11:66/13  "- Input - Wrap Zone VFD Digital Input 2 Status"
  N11:66/14  "- Input - Wrap Zone VFD Digital Input 3 Status"
  N11:66/15  "- Input - Wrap Zone VFD Digital Input 4 Status"
  N11:70/0  "- Input - Infeed 1 VFD Ready"
  N11:70/1  "- Input - Infeed 1 VFD Active"
  N11:70/2  "- Input - Infeed 1 VFD Command Direction Forward"
  N11:70/3  "- Input - Infeed 1 VFD Actual Direction Forward"
  N11:70/4  "- Input - Infeed 1 VFD Accelerating"
  N11:70/5  "- Input - Infeed 1 VFD Decelerating"
  N11:70/6  "- Input - Infeed 1 VFD Alarm Present"
  N11:70/8  "- Input - Infeed 1 VFD At Speed"
  N11:70/9  "- Input - Infeed 1 VFD Main Frequency Controlled By Comm"
  N11:70/10  "- Input - Infeed 1 VFD Operation Command Controlled By Comm"
  N11:70/11  "- Input - Infeed 1 VFD Parameters Locked"
  N11:70/12  "- Input - Infeed 1 VFD Digital Input 1 Status"
  N11:70/13  "- Input - Infeed 1 VFD Digital Input 2 Status"
  N11:70/14  "- Input - Infeed 1 VFD Digital Input 3 Status"
  N11:70/15  "- Input - Infeed 1 VFD Digital Input 4 Status"
  N11:72/0  "- Input - Infeed 2 VFD Ready"
  N11:72/1  "- Input - Infeed 2 VFD Active"
  N11:72/2  "- Input - Infeed 2 VFD Command Direction Forward"
  N11:72/3  "- Input - Infeed 2 VFD Actual Direction Forward"
  N11:72/4  "- Input - Infeed 2 VFD Accelerating"
  N11:72/5  "- Input - Infeed 2 VFD Decelerating"
  N11:72/6  "- Input - Infeed 2 VFD Alarm Present"
  N11:72/8  "- Input - Infeed 2 VFD At Speed"
  N11:72/9  "- Input - Infeed 2 VFD Main Frequency Controlled By Comm"
  N11:72/10  "- Input - Infeed 2 VFD Operation Command Controlled By Comm"
  N11:72/11  "- Input - Infeed 2 VFD Parameters Locked"
  N11:72/12  "- Input - Infeed 2 VFD Digital Input 1 Status"
  N11:72/13  "- Input - Infeed 2 VFD Digital Input 2 Status"
  N11:72/14  "- Input - Infeed 2 VFD Digital Input 3 Status"
  N11:72/15  "- Input - Infeed 2 VFD Digital Input 4 Status"
  N11:74/0  "- Input - Infeed 3 VFD Ready"
  N11:74/1  "- Input - Infeed 3 VFD Active"
  N11:74/2  "- Input - Infeed 3 VFD Command Direction Forward"
  N11:74/3  "- Input - Infeed 3 VFD Actual Direction Forward"
  N11:74/4  "- Input - Infeed 3 VFD Accelerating"
  N11:74/5  "- Input - Infeed 3 VFD Decelerating"
  N11:74/6  "- Input - Infeed 3 VFD Alarm Present"
  N11:74/8  "- Input - Infeed 3 VFD At Speed"
  N11:74/9  "- Input - Infeed 3 VFD Main Frequency Controlled By Comm"
  N11:74/10  "- Input - Infeed 3 VFD Operation Command Controlled By Comm"
  N11:74/11  "- Input - Infeed 3 VFD Parameters Locked"
  N11:74/12  "- Input - Infeed 3 VFD Digital Input 1 Status"
  N11:74/13  "- Input - Infeed 3 VFD Digital Input 2 Status"
  N11:74/14  "- Input - Infeed 3 VFD Digital Input 3 Status"
  N11:74/15  "- Input - Infeed 3 VFD Digital Input 4 Status"
  N11:90/0  "- Input - Exit 1 VFD Ready"
  N11:90/1  "- Input - Exit 1 VFD Active"
  N11:90/2  "- Input - Exit 1 VFD Command Direction Forward"
  N11:90/3  "- Input - Exit 1 VFD Actual Direction Forward"
  N11:90/4  "- Input - Exit 1 VFD Accelerating"
  N11:90/5  "- Input - Exit 1 VFD Decelerating"
  N11:90/6  "- Input - Exit 1 VFD Alarm Present"
  N11:90/8  "- Input - Exit 1 VFD At Speed"
  N11:90/9  "- Input - Exit 1 VFD Main Frequency Controlled By Comm"
  N11:90/10  "- Input - Exit 1 VFD Operation Command Controlled By Comm"
  N11:90/11  "- Input - Exit 1 VFD Parameters Locked"
  N11:90/12  "- Input - Exit 1 VFD Digital Input 1 Status"
  N11:90/13  "- Input - Exit 1 VFD Digital Input 2 Status"
  N11:90/14  "- Input - Exit 1 VFD Digital Input 3 Status"
  N11:90/15  "- Input - Exit 1 VFD Digital Input 4 Status"
  N11:92/0  "- Input - Exit 2 VFD Ready"
  N11:92/1  "- Input - Exit 2 VFD Active"
  N11:92/2  "- Input - Exit 2 VFD Command Direction Forward"
  N11:92/3  "- Input - Exit 2 VFD Actual Direction Forward"
  N11:92/4  "- Input - Exit 2 VFD Accelerating"
  N11:92/5  "- Input - Exit 2 VFD Decelerating"
  N11:92/6  "- Input - Exit 2 VFD Alarm Present"
  N11:92/8  "- Input - Exit 2 VFD At Speed"
  N11:92/9  "- Input - Exit 2 VFD Main Frequency Controlled By Comm"
  N11:92/10  "- Input - Exit 2 VFD Operation Command Controlled By Comm"
  N11:92/11  "- Input - Exit 2 VFD Parameters Locked"
  N11:92/12  "- Input - Exit 2 VFD Digital Input 1 Status"
  N11:92/13  "- Input - Exit 2 VFD Digital Input 2 Status"
  N11:92/14  "- Input - Exit 2 VFD Digital Input 3 Status"
  N11:92/15  "- Input - Exit 2 VFD Digital Input 4 Status"
  N11:94/0  "- Input - Exit 3 VFD Ready"
  N11:94/1  "- Input - Exit 3 VFD Active"
  N11:94/2  "- Input - Exit 3 VFD Command Direction Forward"
  N11:94/3  "- Input - Exit 3 VFD Actual Direction Forward"
  N11:94/4  "- Input - Exit 3 VFD Accelerating"
  N11:94/5  "- Input - Exit 3 VFD Decelerating"
  N11:94/6  "- Input - Exit 3 VFD Alarm Present"
  N11:94/8  "- Input - Exit 3 VFD At Speed"
  N11:94/9  "- Input - Exit 3 VFD Main Frequency Controlled By Comm"
  N11:94/10  "- Input - Exit 3 VFD Operation Command Controlled By Comm"
  N11:94/11  "- Input - Exit 3 VFD Parameters Locked"
  N11:94/12  "- Input - Exit 3 VFD Digital Input 1 Status"
  N11:94/13  "- Input - Exit 3 VFD Digital Input 2 Status"
  N11:94/14  "- Input - Exit 3 VFD Digital Input 3 Status"
  N11:94/15  "- Input - Exit 3 VFD Digital Input 4 Status"
  N12:12/0  "Rotation No Faults"
  N12:12/1  "Rotation Motion Stopped"
  N12:12/2  "Rotation Ready For Auto"
  N12:13/0  "Film Carriage No Faults"
  N12:13/1  "Film Carriage Motion Stopped"
  N12:13/2  "Film Carriage Ready For Auto"
  N12:14/0  "Metered Pre-Stretch No Faults"
  N12:14/1  "Metered Pre-Stretch Motion Stopped"
  N12:14/2  "Metered Pre-Stretch Ready For Auto"
  N12:15/0  "Cutter Assembly No Faults"
  N12:15/1  "Cutter Assembly Motion Stopped"
  N12:15/2  "Cutter Assembly Ready For Auto"
  N12:16/0  "Film Clamp No Faults"
  N12:16/1  "Film Clamp Motion Stopped"
  N12:16/2  "Film Clamp Ready For Auto"
  N12:17/0  "Hot Wire No Faults"
  N12:17/1  "Hot Wire Motion Stopped"
  N12:17/2  "Hot Wire Ready For Auto"
  N12:26/0  "Infeed 4 No Faults"
  N12:27/0  "Infeed 3 No Faults"
  N12:27/1  "Infeed 3 Motion Stopped"
  N12:27/2  "Infeed 3 Ready For Auto"
  N12:28/0  "Infeed 2 No Faults"
  N12:28/1  "Infeed 2 Motion Stopped"
  N12:28/2  "Infeed 2 Ready For Auto"
  N12:29/0  "Infeed 1 No Faults"
  N12:29/1  "Infeed 1 Motion Stopped"
  N12:29/2  "Infeed 1 Ready For Auto"
  N12:30/0  "Wrap Zone No Faults"
  N12:30/1  "Wrap Zone Motion Stopped"
  N12:30/2  "Wrap Zone Ready For Auto"
  N12:31/0  "Exit 1 No Faults"
  N12:31/1  "Exit 1 Motion Stopped"
  N12:31/2  "Exit 1 Ready For Auto"
  N12:32/0  "Exit 2 No Faults"
  N12:32/1  "Exit 2 Motion Stopped"
  N12:32/2  "Exit 2 Ready For Auto"
  N12:33/0  "Exit 3 No Faults"
  N12:33/1  "Exit 3 Motion Stopped"
  N12:33/2  "Exit 3 Ready For Auto"
  N12:42/0  "Infeed Gate No Faults"
  N12:42/1  "Infeed Gate Motion Stopped"
  N12:42/2  "Infeed Gate Ready For Auto"
  N12:43/0  "Exit Gate No Faults"
  N12:43/1  "Infeed Gate Motion Stopped"
  N12:43/2  "Infeed Gate Ready For Auto"
  N12:45/0  "Load Lift No Faults"
  N12:45/1  "Load Lift Motion Stopped"
  N12:45/2  "Load Lift Ready For Auto"
  N14:60  "Profile Map HMI Input Hold Value"
  N14:61  "Customer Number Hold Value"
  N14:62  "Profile HMI Edit Input Hold Value"
  N14:63  "Select New Profile Hold Value"
  N14:64  "Sort Profiles Selection/Edit Adjustment"
  N14:100  FDSSTOPPINGDISTMIN  "FDS Stopping Distance Minimum"
  N14:101  FDSSTOPPINGDISTMAX  "FDS Stopping Distance Maximum"
  N14:102  FDSMAXSPEED  "FDS Maximum Speed"
  N15:0/7  "- Option 8 -"
  N15:0/11  "- Option 12 - Film Sealer"
  N15:1  "Options"
  N15:1/4  "- Option 21 -"
  N15:1/5  "- Option 22 -"
  N15:1/6  "- Option 23 -"
  N15:1/7  "- Option 24 -"
  N15:1/11  "- Option 28 -"
  N15:1/12  "- Option 29 -"
  N15:1/13  "- Option 30 -"
  N15:1/14  "- Option 31 -"
  N15:1/15  "- Option 32 -"
  N15:2  "Options"
  N15:2/4  "- Option 37 -"
  N15:2/5  "- Option 38 -"
  N15:2/6  "- Option 39 -"
  N15:2/7  "- Option 40 -"
  N15:2/11  "- Option 44 -"
  N15:2/12  "- Option 45 -"
  N15:2/13  "- Option 46 -"
  N15:2/14  "- Option 47 -"
  N15:2/15  "- Option 48 -"
  N15:3  "Options"
  N15:3/3  "- Option 52 -"
  N15:3/4  "- Option 53 -"
  N15:3/5  "- Option 54 -"
  N15:3/6  "- Option 55 -"
  N15:3/7  "- Option 56 -"
  N15:3/8  "- Option 57 -"
  N15:3/9  "- Option 58 -"
  N15:3/10  "- Option 59 -"
  N15:3/11  "- Option 60 -"
  N15:3/12  "- Option 61 -"
  N15:3/13  "- Option 62 -"
  N15:3/14  "- Option 63 - 90° Exit"
  N15:4  "Options"
  N15:4/3  "- Option 68 -"
  N15:4/4  "- Option 69 -"
  N15:4/5  "- Option 70 -"
  N15:4/6  "- Option 71 -"
  N15:4/7  "- Option 72 -"
  N15:4/8  "- Option 73 -"
  N15:4/9  "- Option 74 -"
  N15:4/10  "- Option 75 -"
  N15:4/11  "- Option 76 -"
  N15:4/12  "- Option 77 -"
  N15:4/13  "- Option 78 -"
  N15:5  "Options"
  N15:5/0  "- Option 1 - On One Shot"
  N15:5/1  "- Option 2 - On One Shot"
  N15:5/2  "- Option 3 - On One Shot"
  N15:5/3  "- Option 4 - On One Shot"
  N15:5/4  "- Option 5 - On One Shot"
  N15:5/5  "- Option 6 - On One Shot"
  N15:5/6  "- Option 7 - On One Shot"
  N15:5/7  "- Option 8 - On One Shot"
  N15:5/8  "- Option 9 - On One Shot"
  N15:5/9  "- Option 10 - On One Shot"
  N15:5/10  "- Option 11 - On One Shot"
  N15:5/11  "- Option 12 - On One Shot"
  N15:5/12  "- Option 13 - On One Shot"
  N15:5/13  "- Option 14 - On One Shot"
  N15:5/14  "- Option 15 - On One Shot"
  N15:5/15  "- Option 16 - On One Shot"
  N15:6  "Options"
  N15:6/0  "- Option 17 - On One Shot"
  N15:6/1  "- Option 18 - On One Shot"
  N15:6/2  "- Option 19 - On One Shot"
  N15:6/3  "- Option 20 - On One Shot"
  N15:6/4  "- Option 21 - On One Shot"
  N15:6/5  "- Option 22 - On One Shot"
  N15:6/6  "- Option 23 - On One Shot"
  N15:6/7  "- Option 24 - On One Shot"
  N15:6/8  "- Option 25 - On One Shot"
  N15:6/9  "- Option 26 - On One Shot"
  N15:6/10  "- Option 27 - On One Shot"
  N15:6/11  "- Option 28 - On One Shot"
  N15:6/12  "- Option 29 - On One Shot"
  N15:6/13  "- Option 30 - On One Shot"
  N15:6/14  "- Option 31 - On One Shot"
  N15:6/15  "- Option 32 - On One Shot"
  N15:7  "Options"
  N15:7/0  "- Option 33 - On One Shot"
  N15:7/1  "- Option 34 - On One Shot"
  N15:7/2  "- Option 35 - On One Shot"
  N15:7/3  "- Option 36 - On One Shot"
  N15:7/4  "- Option 37 - On One Shot"
  N15:7/5  "- Option 38 - On One Shot"
  N15:7/6  "- Option 39 - On One Shot"
  N15:7/7  "- Option 40 - On One Shot"
  N15:7/8  "- Option 41 - On One Shot"
  N15:7/9  "- Option 42 - On One Shot"
  N15:7/10  "- Option 43 - On One Shot"
  N15:7/11  "- Option 44 - On One Shot"
  N15:7/12  "- Option 45 - On One Shot"
  N15:7/13  "- Option 46 - On One Shot"
  N15:7/14  "- Option 47 - On One Shot"
  N15:7/15  "- Option 48 - On One Shot"
  N15:8  "Options"
  N15:8/0  "- Option 49 - On One Shot"
  N15:8/1  "- Option 50 - On One Shot"
  N15:8/2  "- Option 51 - On One Shot"
  N15:8/3  "- Option 52 - On One Shot"
  N15:8/4  "- Option 53 - On One Shot"
  N15:8/5  "- Option 54 - On One Shot"
  N15:8/6  "- Option 55 - On One Shot"
  N15:8/7  "- Option 56 - On One Shot"
  N15:8/8  "- Option 57 - On One Shot"
  N15:8/9  "- Option 58 - On One Shot"
  N15:8/10  "- Option 59 - On One Shot"
  N15:8/11  "- Option 60 - On One Shot"
  N15:8/12  "- Option 61 - On One Shot"
  N15:8/13  "- Option 62 - On One Shot"
  N15:8/14  "- Option 63 - On One Shot"
  N15:8/15  "- Option 64 - On One Shot"
  N15:9  "Options"
  N15:9/0  "- Option 65 - On One Shot"
  N15:9/1  "- Option 66 - On One Shot"
  N15:9/2  "- Option 67 - On One Shot"
  N15:9/3  "- Option 68 - On One Shot"
  N15:9/4  "- Option 69 - On One Shot"
  N15:9/5  "- Option 70 - On One Shot"
  N15:9/6  "- Option 71 - On One Shot"
  N15:9/7  "- Option 72 - On One Shot"
  N15:9/8  "- Option 73 - On One Shot"
  N15:9/9  "- Option 74 - On One Shot"
  N15:9/10  "- Option 75 - On One Shot"
  N15:9/11  "- Option 76 - On One Shot"
  N15:9/12  "- Option 77 - On One Shot"
  N15:9/13  "- Option 78 - On One Shot"
  N15:9/14  "- Option 79 - On One Shot"
  N15:9/15  "- Option 80 - On One Shot"
  N15:10  "Options"
  N15:10/0  "- Option 1 - Off One Shot"
  N15:10/1  "- Option 2 - Off One Shot"
  N15:10/2  "- Option 3 - Off One Shot"
  N15:10/3  "- Option 4 - Off One Shot"
  N15:10/4  "- Option 5 - Off One Shot"
  N15:10/5  "- Option 6 - Off One Shot"
  N15:10/6  "- Option 7 - Off One Shot"
  N15:10/7  "- Option 8 - Off One Shot"
  N15:10/8  "- Option 9 - Off One Shot"
  N15:10/9  "- Option 10 - Off One Shot"
  N15:10/10  "- Option 11 - Off One Shot"
  N15:10/11  "- Option 12 - Off One Shot"
  N15:10/12  "- Option 13 - Off One Shot"
  N15:10/13  "- Option 14 - Off One Shot"
  N15:10/14  "- Option 15 - Off One Shot"
  N15:10/15  "- Option 16 - Off One Shot"
  N15:11  "Options"
  N15:11/0  "- Option 17 - Off One Shot"
  N15:11/1  "- Option 18 - Off One Shot"
  N15:11/2  "- Option 19 - Off One Shot"
  N15:11/3  "- Option 20 - Off One Shot"
  N15:11/4  "- Option 21 - Off One Shot"
  N15:11/5  "- Option 22 - Off One Shot"
  N15:11/6  "- Option 23 - Off One Shot"
  N15:11/7  "- Option 24 - Off One Shot"
  N15:11/8  "- Option 25 - Off One Shot"
  N15:11/9  "- Option 26 - Off One Shot"
  N15:11/10  "- Option 27 - Off One Shot"
  N15:11/11  "- Option 28 - Off One Shot"
  N15:11/12  "- Option 29 - Off One Shot"
  N15:11/13  "- Option 30 - Off One Shot"
  N15:11/14  "- Option 31 - Off One Shot"
  N15:11/15  "- Option 32 - Off One Shot"
  N15:12  "Options"
  N15:12/0  "- Option 33 - Off One Shot"
  N15:12/1  "- Option 34 - Off One Shot"
  N15:12/2  "- Option 35 - Off One Shot"
  N15:12/3  "- Option 36 - Off One Shot"
  N15:12/4  "- Option 37 - Off One Shot"
  N15:12/5  "- Option 38 - Off One Shot"
  N15:12/6  "- Option 39 - Off One Shot"
  N15:12/7  "- Option 40 - Off One Shot"
  N15:12/8  "- Option 41 - Off One Shot"
  N15:12/9  "- Option 42 - Off One Shot"
  N15:12/10  "- Option 43 - Off One Shot"
  N15:12/11  "- Option 44 - Off One Shot"
  N15:12/12  "- Option 45 - Off One Shot"
  N15:12/13  "- Option 46 - Off One Shot"
  N15:12/14  "- Option 47 - Off One Shot"
  N15:12/15  "- Option 48 - Off One Shot"
  N15:13  "Options"
  N15:13/0  "- Option 49 - Off One Shot"
  N15:13/1  "- Option 50 - Off One Shot"
  N15:13/2  "- Option 51 - Off One Shot"
  N15:13/3  "- Option 52 - Off One Shot"
  N15:13/4  "- Option 53 - Off One Shot"
  N15:13/5  "- Option 54 - Off One Shot"
  N15:13/6  "- Option 55 - Off One Shot"
  N15:13/7  "- Option 56 - Off One Shot"
  N15:13/8  "- Option 57 - Off One Shot"
  N15:13/9  "- Option 58 - Off One Shot"
  N15:13/10  "- Option 59 - Off One Shot"
  N15:13/11  "- Option 60 - Off One Shot"
  N15:13/12  "- Option 61 - Off One Shot"
  N15:13/13  "- Option 62 - Off One Shot"
  N15:13/14  "- Option 63 - Off One Shot"
  N15:13/15  "- Option 64 - Off One Shot"
  N15:14  "Options"
  N15:14/0  "- Option 65 - Off One Shot"
  N15:14/1  "- Option 66 - Off One Shot"
  N15:14/2  "- Option 67 - Off One Shot"
  N15:14/3  "- Option 68 - Off One Shot"
  N15:14/4  "- Option 69 - Off One Shot"
  N15:14/5  "- Option 70 - Off One Shot"
  N15:14/6  "- Option 71 - Off One Shot"
  N15:14/7  "- Option 72 - Off One Shot"
  N15:14/8  "- Option 73 - Off One Shot"
  N15:14/9  "- Option 74 - Off One Shot"
  N15:14/10  "- Option 75 - Off One Shot"
  N15:14/11  "- Option 76 - Off One Shot"
  N15:14/12  "- Option 77 - Off One Shot"
  N15:14/13  "- Option 78 - Off One Shot"
  N15:14/14  "- Option 79 - Off One Shot"
  N15:14/15  "- Option 80 - Off One Shot"
  N17:0  "MESSAGING"
  N20:0  "Difference Between Current Film Thickness And Minimum"
  N20:1  FILMWIDTHATROLL  "Film Width At Roll"
  N20:2  "Film Width Pallet Grip Engaged"
  N20:4  LOSSFROMGRIP  "Size Of Film Width After Pallet-Grip Bunching Effect"
  N20:5  LOSSFROMSTRETCH  "Film Width Size Lost Due To Prestretch"
  N20:7  FILMWIDTHATBOTTOM  "Film Width At Bottom"
  N20:10  "Film Thickness Max"
  N20:11  "Film Thickness Min"
  N20:12  THICKNESSRANGE  "Film Thickness Range"
  N20:15  "Film Width Loss From Pallet Grip"
  N20:17  "Minimum Amount Of Film Width Lost"
  N20:18  "Maximum Amount Of Film Web Lost"
  N20:19  "Minimum Payout Percentange"
  N20:20  "Maximum Payout Percentange"
  N20:21  "Range Of Film Width Size Lost From Prestretching"
  N20:22  "Range Of Prestretch Percentages"
  N20:23  "Multiplier To Apply To Film Web Size Lost Range"
  N29:0/6  "HMI Profile Top Wraps First"
  N29:9  "HMI Input Top Overwrap (Inches)"
  N30:0/6  "Default Profile Top Wraps First"
  N30:0/8  "Default TSD New Profile (0=New, 1=Existing)"
  N30:2  "Default Number"
  N30:9  "Default Top Overwrap (Inches)"
  N30:14  "Default Projected Containment Force"
  N30:18  "Default Force At Load Min Value"
  N30:19  "Default Top Overwrap Min Value (Inches)"
  N30:32  "Default Profile Password"
  N30:48  "Default Profile TSD Leading Film"
  N30:49  "Default Profile TSD Trailing Film"
  N31:0/1  "Profile 1 Force Bottom Enable"
  N31:0/2  "Profile 1 Force Top Enable"
  N31:0/3  "Profile 1 Use Load Lift"
  N31:0/4  "Profile 1 Monitor Containment Force"
  N31:0/5  "Profile 1 Exists"
  N31:0/6  "Profile 1 Top Wraps First"
  N31:0/7  "TSD Enable"
  N31:0/8  "Profile 1 TSD New Profile (0=New, 1=Existing)"
  N31:3  "Profile 1 Rotation Up Speed (%)"
  N31:4  "Profile 1 Rotation Down Speed (%)"
  N31:5  "Profile 1 Force At Top"
  N31:6  "Profile 1 Force At Bottom"
  N31:7  "Profile 1 Force During Cut"
  N31:8  "Profile 1 Force At Load"
  N31:9  "Profile 1 Top Overwrap (Inches)"
  N31:10  "Profile 1 Number of Total Film Layers"
  N31:11  "Profile 1 Load Height"
  N31:12  "Profile 1 Short Load Height (Inches)"
  N31:13  "Profile 1 Containment Force Requirement"
  N31:14  "Profile 1 Projected Containment Force"
  N31:18  "Profile 1 Force At Load Min Value"
  N31:19  "Profile 1 Top Overwrap Min Value (Inches)"
  N31:20  "Profile 1 Band 1 Location"
  N31:21  "Profile 1 Band 1 Wraps"
  N31:22  "Profile 1 Band 1 Reference"
  N31:23  "Profile 1 Band 2 Location"
  N31:24  "Profile 1 Band 2 Wraps"
  N31:25  "Profile 1 Band 2 Reference"
  N31:26  "Profile 1 Band 3 Location"
  N31:27  "Profile 1 Band 3 Wraps"
  N31:28  "Profile 1 Band 3 Reference"
  N31:29  "Profile 1 Band 4 Location"
  N31:30  "Profile 1 Band 4 Wraps"
  N31:31  "Profile 1 Band 4 Reference"
  N31:32  "Profile 1 Password"
  N31:48  "Profile 1 TSD Leading Film"
  N31:49  "Profile 1 TSD Trailing Film"
  N32:0/1  "Profile 2 Force Bottom Enable"
  N32:0/2  "Profile 2 Force Top Enable"
  N32:0/3  "Profile 2 Use Load Lift"
  N32:0/4  "Profile 2 Monitor Containment Force"
  N32:0/5  "Profile 2 Exists"
  N32:0/8  "Profile 2 TSD New Profile (0=New, 1=Existing)"
  N32:3  "Profile 2 Rotation Up Speed (%)"
  N32:4  "Profile 2 Rotation Down Speed (%)"
  N32:5  "Profile 2 Force At Top"
  N32:6  "Profile 2 Force At Bottom"
  N32:7  "Profile 2 Force During Cut"
  N32:8  "Profile 2 Force At Load"
  N32:9  "Profile 2 Top Overwrap (Inches)"
  N32:10  "Profile 2 Number of Total Film Layers"
  N32:11  "Profile 2 Load Height"
  N32:12  "Profile 2 Short Load Height (Inches)"
  N32:13  "Profile 2 Containment Force Requirement"
  N32:14  "Profile 2 Projected Containment Force"
  N32:18  "Profile 2 Force At Load Min Value"
  N32:19  "Profile 2 Top Overwrap Min Value (Inches)"
  N32:20  "Profile 2 Band 1 Location"
  N32:21  "Profile 2 Band 1 Wraps"
  N32:22  "Profile 2 Band 1 Reference"
  N32:23  "Profile 2 Band 2 Location"
  N32:24  "Profile 2 Band 2 Wraps"
  N32:25  "Profile 2 Band 2 Reference"
  N32:26  "Profile 2 Band 3 Location"
  N32:27  "Profile 2 Band 3 Wraps"
  N32:28  "Profile 2 Band 3 Reference"
  N32:29  "Profile 2 Band 4 Location"
  N32:30  "Profile 2 Band 4 Wraps"
  N32:31  "Profile 2 Band 4 Reference"
  N32:32  "Profile 2 Password"
  N33:0/1  "Profile 3 Force Bottom Enable"
  N33:0/2  "Profile 3 Force Top Enable"
  N33:0/3  "Profile 3 Use Load Lift"
  N33:0/4  "Profile 3 Monitor Containment Force"
  N33:0/5  "Profile 3 Exists"
  N33:0/8  "Profile 3 TSD New Profile (0=New, 1=Existing)"
  N33:3  "Profile 3 Rotation Up Speed (%)"
  N33:4  "Profile 3 Rotation Down Speed (%)"
  N33:5  "Profile 3 Force At Top"
  N33:6  "Profile 3 Force At Bottom"
  N33:7  "Profile 3 Force During Cut"
  N33:8  "Profile 3 Force At Load"
  N33:9  "Profile 3 Top Overwrap (Inches)"
  N33:10  "Profile 3 Number of Total Film Layers"
  N33:11  "Profile 3 Load Height"
  N33:12  "Profile 3 Short Load Height (Inches)"
  N33:13  "Profile 3 Containment Force Requirement"
  N33:14  "Profile 3 Projected Containment Force"
  N33:18  "Profile 3 Force At Load Min Value"
  N33:19  "Profile 3 Top Overwrap Min Value (Inches)"
  N33:20  "Profile 3 Band 1 Location"
  N33:21  "Profile 3 Band 1 Wraps"
  N33:22  "Profile 3 Band 1 Reference"
  N33:23  "Profile 3 Band 2 Location"
  N33:24  "Profile 3 Band 2 Wraps"
  N33:25  "Profile 3 Band 2 Reference"
  N33:26  "Profile 3 Band 3 Location"
  N33:27  "Profile 3 Band 3 Wraps"
  N33:28  "Profile 3 Band 3 Reference"
  N33:29  "Profile 3 Band 4 Location"
  N33:30  "Profile 3 Band 4 Wraps"
  N33:31  "Profile 3 Band 4 Reference"
  N33:32  "Profile 3 Password"
  N34:0/1  "Profile 4 Force Bottom Enable"
  N34:0/2  "Profile 4 Force Top Enable"
  N34:0/3  "Profile 4 Use Load Lift"
  N34:0/4  "Profile 4 Monitor Containment Force"
  N34:0/5  "Profile 4 Exists"
  N34:0/8  "Profile 4 TSD New Profile (0=New, 1=Existing)"
  N34:3  "Profile 4 Rotation Up Speed (%)"
  N34:4  "Profile 4 Rotation Down Speed (%)"
  N34:5  "Profile 4 Force At Top"
  N34:6  "Profile 4 Force At Bottom"
  N34:7  "Profile 4 Force During Cut"
  N34:8  "Profile 4 Force At Load"
  N34:9  "Profile 4 Top Overwrap (Inches)"
  N34:10  "Profile 4 Number of Total Film Layers"
  N34:11  "Profile 4 Load Height"
  N34:12  "Profile 4 Short Load Height (Inches)"
  N34:13  "Profile 4 Containment Force Requirement"
  N34:14  "Profile 4 Projected Containment Force"
  N34:18  "Profile 4 Force At Load Min Value"
  N34:19  "Profile 4 Top Overwrap Min Value (Inches)"
  N34:20  "Profile 4 Band 1 Location"
  N34:21  "Profile 4 Band 1 Wraps"
  N34:22  "Profile 4 Band 1 Reference"
  N34:23  "Profile 4 Band 2 Location"
  N34:24  "Profile 4 Band 2 Wraps"
  N34:25  "Profile 4 Band 2 Reference"
  N34:26  "Profile 4 Band 3 Location"
  N34:27  "Profile 4 Band 3 Wraps"
  N34:28  "Profile 4 Band 3 Reference"
  N34:29  "Profile 4 Band 4 Location"
  N34:30  "Profile 4 Band 4 Wraps"
  N34:31  "Profile 4 Band 4 Reference"
  N34:32  "Profile 4 Password"
  N35:0/1  "Profile 5 Force Bottom Enable"
  N35:0/2  "Profile 5 Force Top Enable"
  N35:0/3  "Profile 5 Use Load Lift"
  N35:0/4  "Profile 5 Monitor Containment Force"
  N35:0/5  "Profile 5 Exists"
  N35:0/8  "Profile 5 TSD New Profile (0=New, 1=Existing)"
  N35:3  "Profile 5 Rotation Up Speed (%)"
  N35:4  "Profile 5 Rotation Down Speed (%)"
  N35:5  "Profile 5 Force At Top"
  N35:6  "Profile 5 Force At Bottom"
  N35:7  "Profile 5 Force During Cut"
  N35:8  "Profile 5 Force At Load"
  N35:9  "Profile 5 Top Overwrap (Inches)"
  N35:10  "Profile 5 Number of Total Film Layers"
  N35:11  "Profile 5 Load Height"
  N35:12  "Profile 5 Short Load Height (Inches)"
  N35:13  "Profile 5 Containment Force Requirement"
  N35:14  "Profile 5 Projected Containment Force"
  N35:18  "Profile 5 Force At Load Min Value"
  N35:19  "Profile 5 Top Overwrap Min Value (Inches)"
  N35:20  "Profile 5 Band 1 Location"
  N35:21  "Profile 5 Band 1 Wraps"
  N35:22  "Profile 5 Band 1 Reference"
  N35:23  "Profile 5 Band 2 Location"
  N35:24  "Profile 5 Band 2 Wraps"
  N35:25  "Profile 5 Band 2 Reference"
  N35:26  "Profile 5 Band 3 Location"
  N35:27  "Profile 5 Band 3 Wraps"
  N35:28  "Profile 5 Band 3 Reference"
  N35:29  "Profile 5 Band 4 Location"
  N35:30  "Profile 5 Band 4 Wraps"
  N35:31  "Profile 5 Band 4 Reference"
  N35:32  "Profile 5 Password"
  N36:0/1  "Profile 6 Force Bottom Enable"
  N36:0/2  "Profile 6 Force Top Enable"
  N36:0/3  "Profile 6 Use Load Lift"
  N36:0/4  "Profile 6 Monitor Containment Force"
  N36:0/5  "Profile 6 Exists"
  N36:0/8  "Profile 6 TSD New Profile (0=New, 1=Existing)"
  N36:3  "Profile 6 Rotation Up Speed (%)"
  N36:4  "Profile 6 Rotation Down Speed (%)"
  N36:5  "Profile 6 Force At Top"
  N36:6  "Profile 6 Force At Bottom"
  N36:7  "Profile 6 Force During Cut"
  N36:8  "Profile 6 Force At Load"
  N36:9  "Profile 6 Top Overwrap (Inches)"
  N36:10  "Profile 6 Number of Total Film Layers"
  N36:11  "Profile 6 Load Height"
  N36:12  "Profile 6 Short Load Height (Inches)"
  N36:13  "Profile 6 Containment Force Requirement"
  N36:14  "Profile 6 Projected Containment Force"
  N36:18  "Profile 6 Force At Load Min Value"
  N36:19  "Profile 6 Top Overwrap Min Value (Inches)"
  N36:20  "Profile 6 Band 1 Location"
  N36:21  "Profile 6 Band 1 Wraps"
  N36:22  "Profile 6 Band 1 Reference"
  N36:23  "Profile 6 Band 2 Location"
  N36:24  "Profile 6 Band 2 Wraps"
  N36:25  "Profile 6 Band 2 Reference"
  N36:26  "Profile 6 Band 3 Location"
  N36:27  "Profile 6 Band 3 Wraps"
  N36:28  "Profile 6 Band 3 Reference"
  N36:29  "Profile 6 Band 4 Location"
  N36:30  "Profile 6 Band 4 Wraps"
  N36:31  "Profile 6 Band 4 Reference"
  N36:32  "Profile 6 Password"
  N37:0/1  "Profile 7 Force Bottom Enable"
  N37:0/2  "Profile 7 Force Top Enable"
  N37:0/3  "Profile 7 Use Load Lift"
  N37:0/4  "Profile 7 Monitor Containment Force"
  N37:0/5  "Profile 7 Exists"
  N37:0/8  "Profile 7 TSD New Profile (0=New, 1=Existing)"
  N37:3  "Profile 7 Rotation Up Speed (%)"
  N37:4  "Profile 7 Rotation Down Speed (%)"
  N37:5  "Profile 7 Force At Top"
  N37:6  "Profile 7 Force At Bottom"
  N37:7  "Profile 7 Force During Cut"
  N37:8  "Profile 7 Force At Load"
  N37:9  "Profile 7 Top Overwrap (Inches)"
  N37:10  "Profile 7 Number of Total Film Layers"
  N37:11  "Profile 7 Load Height"
  N37:12  "Profile 7 Short Load Height (Inches)"
  N37:13  "Profile 7 Containment Force Requirement"
  N37:14  "Profile 7 Projected Containment Force"
  N37:18  "Profile 7 Force At Load Min Value"
  N37:19  "Profile 7 Top Overwrap Min Value (Inches)"
  N37:20  "Profile 7 Band 1 Location"
  N37:21  "Profile 7 Band 1 Wraps"
  N37:22  "Profile 7 Band 1 Reference"
  N37:23  "Profile 7 Band 2 Location"
  N37:24  "Profile 7 Band 2 Wraps"
  N37:25  "Profile 7 Band 2 Reference"
  N37:26  "Profile 7 Band 3 Location"
  N37:27  "Profile 7 Band 3 Wraps"
  N37:28  "Profile 7 Band 3 Reference"
  N37:29  "Profile 7 Band 4 Location"
  N37:30  "Profile 7 Band 4 Wraps"
  N37:31  "Profile 7 Band 4 Reference"
  N37:32  "Profile 7 Password"
  N38:0/1  "Profile 8 Force Bottom Enable"
  N38:0/2  "Profile 8 Force Top Enable"
  N38:0/3  "Profile 8 Use Load Lift"
  N38:0/4  "Profile 8 Monitor Containment Force"
  N38:0/5  "Profile 8 Exists"
  N38:0/8  "Profile 8 TSD New Profile (0=New, 1=Existing)"
  N38:3  "Profile 8 Rotation Up Speed (%)"
  N38:4  "Profile 8 Rotation Down Speed (%)"
  N38:5  "Profile 8 Force At Top"
  N38:6  "Profile 8 Force At Bottom"
  N38:7  "Profile 8 Force During Cut"
  N38:8  "Profile 8 Force At Load"
  N38:9  "Profile 8 Top Overwrap (Inches)"
  N38:10  "Profile 8 Number of Total Film Layers"
  N38:11  "Profile 8 Load Height"
  N38:12  "Profile 8 Short Load Height (Inches)"
  N38:13  "Profile 8 Containment Force Requirement"
  N38:14  "Profile 8 Projected Containment Force"
  N38:18  "Profile 8 Force At Load Min Value"
  N38:19  "Profile 8 Top Overwrap Min Value (Inches)"
  N38:20  "Profile 8 Band 1 Location"
  N38:21  "Profile 8 Band 1 Wraps"
  N38:22  "Profile 8 Band 1 Reference"
  N38:23  "Profile 8 Band 2 Location"
  N38:24  "Profile 8 Band 2 Wraps"
  N38:25  "Profile 8 Band 2 Reference"
  N38:26  "Profile 8 Band 3 Location"
  N38:27  "Profile 8 Band 3 Wraps"
  N38:28  "Profile 8 Band 3 Reference"
  N38:29  "Profile 8 Band 4 Location"
  N38:30  "Profile 8 Band 4 Wraps"
  N38:31  "Profile 8 Band 4 Reference"
  N38:32  "Profile 8 Password"
  N39:0/1  "Profile 9 Force Bottom Enable"
  N39:0/2  "Profile 9 Force Top Enable"
  N39:0/3  "Profile 9 Use Load Lift"
  N39:0/5  "Profile 9 Exists"
  N39:0/8  "Profile 9 TSD New Profile (0=New, 1=Existing)"
  N39:3  "Profile 9 Rotation Up Speed (%)"
  N39:4  "Profile 9 Rotation Down Speed (%)"
  N39:5  "Profile 9 Force At Top"
  N39:6  "Profile 9 Force At Bottom"
  N39:7  "Profile 9 Force During Cut"
  N39:8  "Profile 9 Force At Load"
  N39:9  "Profile 9 Top Overwrap (Inches)"
  N39:10  "Profile 9 Number of Total Film Layers"
  N39:11  "Profile 9 Load Height"
  N39:12  "Profile 9 Short Load Height (Inches)"
  N39:13  "Profile 9 Containment Force Requirement"
  N39:14  "Profile 9 Projected Containment Force"
  N39:18  "Profile 9 Force At Load Min Value"
  N39:19  "Profile 9 Top Overwrap Min Value (Inches)"
  N39:20  "Profile 9 Band 1 Location"
  N39:21  "Profile 9 Band 1 Wraps"
  N39:22  "Profile 9 Band 1 Reference"
  N39:23  "Profile 9 Band 2 Location"
  N39:24  "Profile 9 Band 2 Wraps"
  N39:25  "Profile 9 Band 2 Reference"
  N39:26  "Profile 9 Band 3 Location"
  N39:27  "Profile 9 Band 3 Wraps"
  N39:28  "Profile 9 Band 3 Reference"
  N39:29  "Profile 9 Band 4 Location"
  N39:30  "Profile 9 Band 4 Wraps"
  N39:31  "Profile 9 Band 4 Reference"
  N39:32  "Profile 9 Password"
  N40:0/8  "Current TSD New Profile (0=New, 1=Existing)"
  N40:2  "Profile Selected"
  N40:11  "Current Profile Load Height"
  N40:13  "Current Profile Containment Force Requirement"
  N40:14  "Current Profile Projected Containment Force"
  N40:15  "Current Profile Top Wraps Adjust"
  N40:16  "Current Profile Bottom Wraps Adjust"
  N40:18  "Current Profile Force At Load Min Value"
  N40:22  "Current Profile Band 1 Reference"
  N40:25  "Current Profile Band 2 Reference"
  N40:28  "Current Profile Band 3 Reference"
  N40:31  "Current Profile Band 4 Reference"
  N40:32  "Current Profile Password"
  N41:8  "Profile Shift Start Index"
  N41:9  "Profile Delete Index"
  N41:10  "Profile Shift Start Indirect Address"
  N41:11  "Profile Delete Index Indirect Address"
  N41:19  "Profile Copy Source"
  N41:21  "Profile Attribute Length"
  N41:27  "Infeed 1 Profile Tracking Search Index"
  N42:1  "Profile 1 Customer Number"
  N42:2  "Profile 2 Customer Number"
  N42:3  "Profile 3 Customer Number"
  N42:4  "Profile 4 Customer Number"
  N42:5  "Profile 5 Customer Number"
  N42:6  "Profile 6 Customer Number"
  N42:7  "Profile 7 Customer Number"
  N42:8  "Profile 8 Customer Number"
  N42:9  "Profile 9 Customer Number"
  N45:0  "Default Profile Top Overwrap"
  N45:1  "Default Profile Top Wraps"
  N45:2  "Default Profile Bottom Wraps"
  N45:3  "Default Profile Top Wraps First"
  N45:4  "Default Profile Overlap Up"
  N45:5  "Default Profile Overlap Down"
  N45:6  "Default Profile Rotation Up Speed"
  N45:7  "Default Profile Rotation Down Speed"
  N45:8  "Default Profile Payout Method"
  N45:9  "Default Profile Pallet Payout"
  N45:10  "Default Profile Load Payout"
  N45:11  "Default Profile Minimum Containment Force Requirement"
  N45:12  "Default Profile Spare"
  N45:13  "Default Profile Spare"
  N45:14  "Default Profile Spare"
  N45:15  "Default Profile Short Load Height"
  N45:16  "Default Profile Spare"
  N45:17  "Default Profile Spare"
  N45:18  "Default Profile Spare"
  N45:19  "Default Profile Spare"
  N45:20  "Profile 1 Top Overwrap"
  N45:21  "Profile 1 Top Wraps"
  N45:22  "Profile 1 Bottom Wraps"
  N45:23  "Profile 1 Top Wraps First"
  N45:24  "Profile 1 Overlap Up"
  N45:25  "Profile 1 Overlap Down"
  N45:26  "Profile 1 Rotation Up Speed"
  N45:27  "Profile 1 Rotation Down Speed"
  N45:28  "Profile 1 Payout Method"
  N45:29  "Profile 1 Pallet Payout"
  N45:30  "Profile 1 Load Payout"
  N45:31  "Profile 1 Minimum Containment Force Requirement"
  N45:32  "Profile 1 Spare"
  N45:33  "Profile 1 Spare"
  N45:34  "Profile 1 Spare"
  N45:35  "Profile 1 Short Load Height"
  N45:36  "Profile 1 Spare"
  N45:37  "Profile 1 Spare"
  N45:38  "Profile 1 Spare"
  N45:39  "Profile 1 Spare"
  N45:40  "Profile 2 Top Overwrap"
  N45:41  "Profile 2 Top Wraps"
  N45:42  "Profile 2 Bottom Wraps"
  N45:43  "Profile 2 Top Wraps First"
  N45:44  "Profile 2 Overlap Up"
  N45:45  "Profile 2 Overlap Down"
  N45:46  "Profile 2 Rotation Up Speed"
  N45:47  "Profile 2 Rotation Down Speed"
  N45:48  "Profile 2 Payout Method"
  N45:49  "Profile 2 Pallet Payout"
  N45:50  "Profile 2 Load Payout"
  N45:51  "Profile 2 Minimum Containment Force Requirement"
  N45:52  "Profile 2 Spare"
  N45:53  "Profile 2 Spare"
  N45:54  "Profile 2 Spare"
  N45:55  "Profile 2 Short Load Height"
  N45:56  "Profile 2 Spare"
  N45:57  "Profile 2 Spare"
  N45:58  "Profile 2 Spare"
  N45:59  "Profile 2 Spare"
  N45:60  "Profile 3 Top Overwrap"
  N45:61  "Profile 3 Top Wraps"
  N45:62  "Profile 3 Bottom Wraps"
  N45:63  "Profile 3 Top Wraps First"
  N45:64  "Profile 3 Overlap Up"
  N45:65  "Profile 3 Overlap Down"
  N45:66  "Profile 3 Rotation Up Speed"
  N45:67  "Profile 3 Rotation Down Speed"
  N45:68  "Profile 3 Payout Method"
  N45:69  "Profile 3 Pallet Payout"
  N45:70  "Profile 3 Load Payout"
  N45:71  "Profile 3 Minimum Containment Force Requirement"
  N45:72  "Profile 3 Spare"
  N45:73  "Profile 3 Spare"
  N45:74  "Profile 3 Spare"
  N45:75  "Profile 3 Short Load Height"
  N45:76  "Profile 3 Spare"
  N45:77  "Profile 3 Spare"
  N45:78  "Profile 3 Spare"
  N45:79  "Profile 3 Spare"
  N45:80  "Profile 4 Top Overwrap"
  N45:81  "Profile 4 Top Wraps"
  N45:82  "Profile 4 Bottom Wraps"
  N45:83  "Profile 4 Top Wraps First"
  N45:84  "Profile 4 Overlap Up"
  N45:85  "Profile 4 Overlap Down"
  N45:86  "Profile 4 Rotation Up Speed"
  N45:87  "Profile 4 Rotation Down Speed"
  N45:88  "Profile 4 Payout Method"
  N45:89  "Profile 4 Pallet Payout"
  N45:90  "Profile 4 Load Payout"
  N45:91  "Profile 4 Minimum Containment Force Requirement"
  N45:92  "Profile 4 Spare"
  N45:93  "Profile 4 Spare"
  N45:94  "Profile 4 Spare"
  N45:95  "Profile 4 Short Load Height"
  N45:96  "Profile 4 Spare"
  N45:97  "Profile 4 Spare"
  N45:98  "Profile 4 Spare"
  N45:99  "Profile 4 Spare"
  N45:100  "Profile 5 Top Overwrap"
  N45:101  "Profile 5 Top Wraps"
  N45:102  "Profile 5 Bottom Wraps"
  N45:103  "Profile 5 Top Wraps First"
  N45:104  "Profile 5 Overlap Up"
  N45:105  "Profile 5 Overlap Down"
  N45:106  "Profile 5 Rotation Up Speed"
  N45:107  "Profile 5 Rotation Down Speed"
  N45:108  "Profile 5 Payout Method"
  N45:109  "Profile 5 Pallet Payout"
  N45:110  "Profile 5 Load Payout"
  N45:111  "Profile 5 Minimum Containment Force Requirement"
  N45:112  "Profile 5 Spare"
  N45:113  "Profile 5 Spare"
  N45:114  "Profile 5 Spare"
  N45:115  "Profile 5 Short Load Height"
  N45:116  "Profile 5 Spare"
  N45:117  "Profile 5 Spare"
  N45:118  "Profile 5 Spare"
  N45:119  "Profile 5 Spare"
  N45:120  "Profile 6 Top Overwrap"
  N45:121  "Profile 6 Top Wraps"
  N45:122  "Profile 6 Bottom Wraps"
  N45:123  "Profile 6 Top Wraps First"
  N45:124  "Profile 6 Overlap Up"
  N45:125  "Profile 6 Overlap Down"
  N45:126  "Profile 6 Rotation Up Speed"
  N45:127  "Profile 6 Rotation Down Speed"
  N45:128  "Profile 6 Payout Method"
  N45:129  "Profile 6 Pallet Payout"
  N45:130  "Profile 6 Load Payout"
  N45:131  "Profile 6 Minimum Containment Force Requirement"
  N45:132  "Profile 6 Spare"
  N45:133  "Profile 6 Spare"
  N45:134  "Profile 6 Spare"
  N45:135  "Profile 6 Short Load Height"
  N45:136  "Profile 6 Spare"
  N45:137  "Profile 6 Spare"
  N45:138  "Profile 6 Spare"
  N45:139  "Profile 6 Spare"
  N45:140  "Profile 7 Top Overwrap"
  N45:141  "Profile 7 Top Wraps"
  N45:142  "Profile 7 Bottom Wraps"
  N45:143  "Profile 7 Top Wraps First"
  N45:144  "Profile 7 Overlap Up"
  N45:145  "Profile 7 Overlap Down"
  N45:146  "Profile 7 Rotation Up Speed"
  N45:147  "Profile 7 Rotation Down Speed"
  N45:148  "Profile 7 Payout Method"
  N45:149  "Profile 7 Pallet Payout"
  N45:150  "Profile 7 Load Payout"
  N45:151  "Profile 7 Minimum Containment Force Requirement"
  N45:152  "Profile 7 Spare"
  N45:153  "Profile 7 Spare"
  N45:154  "Profile 7 Spare"
  N45:155  "Profile 7 Short Load Height"
  N45:156  "Profile 7 Spare"
  N45:157  "Profile 7 Spare"
  N45:158  "Profile 7 Spare"
  N45:159  "Profile 7 Spare"
  N45:160  "Profile 8 Top Overwrap"
  N45:161  "Profile 8 Top Wraps"
  N45:162  "Profile 8 Bottom Wraps"
  N45:163  "Profile 8 Top Wraps First"
  N45:164  "Profile 8 Overlap Up"
  N45:165  "Profile 8 Overlap Down"
  N45:166  "Profile 8 Rotation Up Speed"
  N45:167  "Profile 8 Rotation Down Speed"
  N45:168  "Profile 8 Payout Method"
  N45:169  "Profile 8 Pallet Payout"
  N45:170  "Profile 8 Load Payout"
  N45:171  "Profile 8 Minimum Containment Force Requirement"
  N45:172  "Profile 8 Spare"
  N45:173  "Profile 8 Spare"
  N45:174  "Profile 8 Spare"
  N45:175  "Profile 8 Short Load Height"
  N45:176  "Profile 8 Spare"
  N45:177  "Profile 8 Spare"
  N45:178  "Profile 8 Spare"
  N45:179  "Profile 8 Spare"
  N45:180  "Profile 9 Top Overwrap"
  N45:181  "Profile 9 Top Wraps"
  N45:182  "Profile 9 Bottom Wraps"
  N45:183  "Profile 9 Top Wraps First"
  N45:184  "Profile 9 Overlap Up"
  N45:185  "Profile 9 Overlap Down"
  N45:186  "Profile 9 Rotation Up Speed"
  N45:187  "Profile 9 Rotation Down Speed"
  N45:188  "Profile 9 Payout Method"
  N45:189  "Profile 9 Pallet Payout"
  N45:190  "Profile 9 Load Payout"
  N45:191  "Profile 9 Minimum Containment Force Requirement"
  N45:192  "Profile 9 Spare"
  N45:193  "Profile 9 Spare"
  N45:194  "Profile 9 Spare"
  N45:195  "Profile 9 Short Load Height"
  N45:196  "Profile 9 Spare"
  N45:197  "Profile 9 Spare"
  N45:198  "Profile 9 Spare"
  N45:199  "Profile 9 Spare"
  N50:0  "- HMI Output - System Bits"
  N50:0/14  "- HMI Output - PLC Initialize Complete"
  N50:1  "- HMI Output - Manual Bits"
  N50:2  "- HMI Output - Conveyor Bits"
  N50:2/12  "- HMI Output - Wrap Zone At 90°"
  N50:3  "- HMI Output - Conveyor Bits"
  N50:4  "- HMI Output - Conveyor Bits"
  N50:7  "- HMI Output - System Bits"
  N50:7/0  "- HMI Output - Rotation Auto Tune Selected"
  N50:7/1  "- HMI Output - Film Carriage Auto Tune Selected"
  N50:7/2  "- HMI Output - Metered Pre-Stretch Auto Tune Selected"
  N50:7/8  "- HMI Output - Low Film Disabled"
  N50:8  "- HMI Output - Wrap Setup Bits"
  N50:8/1  N50
  N50:8/3  "- HMI Output - 20" Film Used On 30" Carriage"
  N50:8/10  "- HMI Output - Wrap In Progress"
  N50:8/12  "- HMI Output - Profile Copy Enable"
  N50:9  "- HMI Output - Goto Screen Bits"
  N50:9/0  "- HMI Output - Display Goto "Wrap Setup" Screen"
  N50:9/2  "- HMI Output - Display Goto "Profile Copy" Screen"
  N50:9/3  "- HMI Output - Display Goto "Edit Presets" Screen"
  N50:9/4  "- HMI Output - Display Goto "Edit Profiles" Screen"
  N50:9/14  "- HMI Output - Display Goto "Machine Controls" Screen"
  N50:9/15  "- HMI Output - Display Goto "Conv Controls" Screen"
  N50:12  "- HMI Output - Manual Input Warnings"
  N50:13/0  "- HMI Input - No Profiles Enabled"
  N50:16  "- HMI Output - Wrap Progress Indicator"
  N50:27  "- HMI Output - Help"
  N50:39  "- HMI Output - Rotation Status"
  N50:57  "- HMI Output - TSD Elevator Indicator"
  N50:71  "- HMI Output - Interface Status"
  N50:100/0  "- HMI Output - - Option 1 -"
  N50:100/1  "- HMI Output - - Option 2 -"
  N50:100/2  "- HMI Output - - Option 3 -"
  N50:100/3  "- HMI Output - - Option 4 -"
  N50:100/4  "- HMI Output - - Option 5 -"
  N50:100/5  "- HMI Output - - Option 6 -"
  N50:100/6  "- HMI Output - - Option 7 -"
  N50:100/7  "- HMI Output - - Option 8 -"
  N50:100/8  "- HMI Output - - Option 9 -"
  N50:100/9  "- HMI Output - - Option 10 -"
  N50:100/10  "- HMI Output - - Option 11 -"
  N50:100/11  "- HMI Output - - Option 12 -"
  N50:100/12  "- HMI Output - - Option 13 -"
  N50:100/13  "- HMI Output - - Option 14 -"
  N50:100/14  "- HMI Output - - Option 15 -"
  N50:100/15  "- HMI Output - - Option 16 -"
  N50:101/0  "- HMI Output - - Option 17 -"
  N50:101/1  "- HMI Output - - Option 18 -"
  N50:101/2  "- HMI Output - - Option 19 -"
  N50:101/3  "- HMI Output - - Option 20 -"
  N50:101/4  "- HMI Output - - Option 21 -"
  N50:101/5  "- HMI Output - - Option 22 -"
  N50:101/6  "- HMI Output - - Option 23 -"
  N50:101/7  "- HMI Output - - Option 24 -"
  N50:101/8  "- HMI Output - - Option 25 -"
  N50:101/9  "- HMI Output - - Option 26 -"
  N50:101/10  "- HMI Output - - Option 27 -"
  N50:101/11  "- HMI Output - - Option 28 -"
  N50:101/12  "- HMI Output - - Option 29 -"
  N50:101/13  "- HMI Output - - Option 30 -"
  N50:101/14  "- HMI Output - - Option 31 -"
  N50:101/15  "- HMI Output - - Option 32 -"
  N50:102/0  "- HMI Output - - Option 33 -"
  N50:102/1  "- HMI Output - - Option 34 -"
  N50:102/2  "- HMI Output - - Option 35 -"
  N50:102/3  "- HMI Output - - Option 36 -"
  N50:102/4  "- HMI Output - - Option 37 -"
  N50:102/5  "- HMI Output - - Option 38 -"
  N50:102/6  "- HMI Output - - Option 39 -"
  N50:102/7  "- HMI Output - - Option 40 -"
  N50:102/8  "- HMI Output - - Option 41 -"
  N50:102/9  "- HMI Output - - Option 42 -"
  N50:102/10  "- HMI Output - - Option 43 -"
  N50:102/11  "- HMI Output - - Option 44 -"
  N50:102/12  "- HMI Output - - Option 45 -"
  N50:102/13  "- HMI Output - - Option 46 -"
  N50:102/14  "- HMI Output - - Option 47 -"
  N50:102/15  "- HMI Output - - Option 48 -"
  N50:103/0  "- HMI Output - - Option 49 -"
  N50:103/1  "- HMI Output - - Option 50 -"
  N50:103/2  "- HMI Output - - Option 51 -"
  N50:103/3  "- HMI Output - - Option 52 -"
  N50:103/4  "- HMI Output - - Option 53 -"
  N50:103/5  "- HMI Output - - Option 54 -"
  N50:103/6  "- HMI Output - - Option 55 -"
  N50:103/7  "- HMI Output - - Option 56 -"
  N50:103/8  "- HMI Output - - Option 57 -"
  N50:103/9  "- HMI Output - - Option 58 -"
  N50:103/10  "- HMI Output - - Option 59 -"
  N50:103/11  "- HMI Output - - Option 60 -"
  N50:103/12  "- HMI Output - - Option 61 -"
  N50:103/13  "- HMI Output - - Option 62 -"
  N50:103/14  "- HMI Output - - Option 63 -"
  N50:103/15  "- HMI Output - - Option 64 -"
  N50:104/0  "- HMI Output - - Option 65 -"
  N50:104/1  "- HMI Output - - Option 66 -"
  N50:104/2  "- HMI Output - - Option 67 -"
  N50:104/3  "- HMI Output - - Option 68 -"
  N50:104/4  "- HMI Output - - Option 69 -"
  N50:104/5  "- HMI Output - - Option 70 -"
  N50:104/6  "- HMI Output - - Option 71 -"
  N50:104/7  "- HMI Output - - Option 72 -"
  N50:104/8  "- HMI Output - - Option 73 -"
  N50:104/9  "- HMI Output - - Option 74 -"
  N50:104/10  "- HMI Output - - Option 75 -"
  N50:104/11  "- HMI Output - - Option 76 -"
  N50:104/12  "- HMI Output - - Option 77 -"
  N50:104/13  "- HMI Output - - Option 78 -"
  N50:104/14  "- HMI Output - - Option 79 -"
  N50:104/15  "- HMI Output - - Option 80 -"
  N50:111  "- HMI Output - Chart 1"
  N50:112  "- HMI Output - Chart 2"
  N50:113  "- HMI Output - Chart 3"
  N50:114  "- HMI Output - Chart 4"
  N50:115  "- HMI Output - Chart 5"
  N50:116  "- HMI Output - Chart 6"
  N50:117  "- HMI Output - Chart 7"
  N50:118  "- HMI Output - Chart 8"
  N50:119  "- HMI Output - Chart 9"
  N50:120  "- HMI Output - Chart 10"
  N50:121  "- HMI Output - Chart 11"
  N50:122  "- HMI Output - Chart 12"
  N50:123  "- HMI Output - Chart 13"
  N50:124  "- HMI Output - Chart 14"
  N50:125  "- HMI Output - Chart 15"
  N50:126  "- HMI Output - Chart 16"
  N50:127  "- HMI Output - Chart 17"
  N50:128  "- HMI Output - Chart 18"
  N50:129  "- HMI Output - Chart 19"
  N50:130  "- HMI Output - Chart 20"
  N50:131  "- HMI Output - Chart 21"
  N50:132  "- HMI Output - Chart 22"
  N50:133  "- HMI Output - Chart 23"
  N50:134  "- HMI Output - Chart 24"
  N50:135  "- HMI Output - Chart 25"
  N50:136  "- HMI Output - Chart 26"
  N50:137  "- HMI Output - Chart 27"
  N50:138  "- HMI Output - Chart 28"
  N50:139  "- HMI Output - Chart 29"
  N50:140  "- HMI Output - Chart 30"
  N50:141  "- HMI Output - Chart 31"
  N50:170  "- HMI Output - I/O Screen Page Index"
  N50:213/3  "- HMI Output - Top Sheet Overload / Fault"
  N50:213/4  "- HMI Output - Top Sheet Belt At Tension"
  N50:213/5  "- HMI Output - Top Sheet Film Is Low"
  N50:213/6  "- HMI Output - Top Sheet Elevator Up"
  N50:213/7  "- HMI Output - Top Sheet Elevator Down"
  N50:213/8  "- HMI Output - Top Sheet Cutter Wire Fault"
  N50:213/9  "- HMI Output - Top Sheet Cutter Wire Is Tensioned"
  N50:213/10  "- HMI Output - Top Sheet Load Height Is Clear 1"
  N50:213/12  "- HMI Output - Top Sheet Short Load Is Clear"
  N50:214/0  "- HMI Output - Top Sheet Cut Film PB Visible"
  N51:0/10  "- HMI Input - Runout Mode PB"
  N51:0/11  "- HMI Input - Runout Repeat PB"
  N51:0/12  "- HMI Input - Runout No Film Enable PB"
  N51:0/14  "- HMI Input - Initialize PLC PB"
  N51:1/10  "- HMI Input -"
  N51:1/11  "- HMI Input -"
  N51:1/15  "- HMI Input - Stabilizer Raise PB"
  N51:2/0  "- HMI Input - Conveyor Jog PB"
  N51:2/4  "- HMI Input - Conveyors Select None"
  N51:2/9  "- HMI Input - Wrap Zone Tracking Update PB"
  N51:2/10  "- HMI Input - Rotation Jog Jog 90° PB"
  N51:3  "- HMI Input - Conveyor PBs"
  N51:3/8  "- HMI Input - Infeed 1 Tracking Update PB"
  N51:3/9  "- HMI Input - Infeed 2 Tracking Update PB"
  N51:3/10  "- HMI Input - Infeed 3 Tracking Update PB"
  N51:4  "- HMI Input - Conveyor PBs"
  N51:4/8  "- HMI Input - Exit 1 Tracking Update PB"
  N51:4/9  "- HMI Input - Exit 2 Tracking Update PB"
  N51:4/10  "- HMI Input - Exit 3 Tracking Update PB"
  N51:5/0  "- HMI Input - Goto Setup Screen"
  N51:5/1  "- HMI Input - Goto Profile Names Screen"
  N51:5/2  "- HMI Input - Goto Profile Copy Screen"
  N51:5/3  "- HMI Input - Goto Edit Presets Screen"
  N51:5/4  "- HMI Input - Goto Edit Profiles Screen"
  N51:5/14  "- HMI Input - Goto Machine Controls"
  N51:5/15  "- HMI Input - Goto Conveyor Controls"
  N51:7  "- HMI Input - System PBs"
  N51:7/7  "- HMI Input - Menu Is Open"
  N51:8  "- HMI Input - Wrap Setup PBs"
  N51:8/1  "- HMI Input - Wrap Profile Copy PB"
  N51:8/3  "- HMI Input - 20 Inch Film PB"
  N51:8/4  "- HMI Input - 30 Inch Film PB"
  N51:8/9  "- HMI Input - Profile Edit Menu"
  N51:8/12  "- HMI Input - Profile Import PB"
  N51:9  "- HMI Input - System PBs (Maintained)"
  N51:11/0  "- HMI Input - Default User "Wrap Setup" Access PB"
  N51:11/2  "- HMI Input - Default User "Profile Copy" Access"
  N51:11/3  "- HMI Input - Default User "Edit Presets" Access"
  N51:11/4  "- HMI Input - Default User "Edit Profiles" Access"
  N51:11/5  "- HMI Input - Level 1 User "Wrap Setup" Access PB"
  N51:11/7  "- HMI Input - User Level 1 "Profile Copy" Access"
  N51:11/8  "- HMI Input - User Level 1 "Edit Presets" Access"
  N51:11/9  "- HMI Input - User Level 1 "Edit Profiles" Access"
  N51:11/10  "- HMI Input - Level 2 User "Wrap Setup" Access PB"
  N51:11/12  "- HMI Input - User Level 2 "Profile Copy" Access"
  N51:11/13  "- HMI Input - User Level 2 "Edit Presets" Access"
  N51:11/14  "- HMI Input - User Level 2 "Edit Profiles" Access"
  N51:20  "- HMI Input - Year"
  N51:21  "- HMI Input - Month"
  N51:26  "- HMI Input - RESERVED"
  N51:41  "- HMI Input - Wrap Profile Edit"
  N51:42  "- HMI Input - Wrap Profile Edit Request"
  N51:44  "- HMI Input - Wrap Profile Copy Destination"
  N51:52  "- HMI Input - Wrap Profile Import Index"
  N51:53  "- HMI Input - Wrap Profile Import Value"
  N51:54  "- HMI Input - Wrap Profile Import New Value"
  N51:62  "- HMI Input - Starting Girth"
  N51:68  "- HMI Input - Conveyor Upstream Speed"
  N51:69  "- HMI Input - Conveyor Downstream Speed"
  N51:74  "- HMI Input - Preset Spare"
  N51:75  "- HMI Input - Load Stabilizer Off Load Delay"
  N51:76  "- HMI Input - Load Stabilizer On Load Delay"
  N51:80  "- HMI Input - Preset Starved Speed"
  N51:80/0  "TSD Dispense Trailing Film"
  N51:81  "- HMI Input - Preset Reserved"
  N51:82  "- HMI Input - Preset Reserved"
  N51:85  "- HMI Input - Preset Reserved"
  N51:87  "- HMI Input - Preset Spare"
  N51:88  "- HMI Input - Preset Wipe Arm Retract Delay"
  N51:89  "- HMI Input - Preset Wipe Retract"
  N51:90  "- HMI Input - Wrap Profile Number"
  N51:100/7  "- HMI Input - - Option 8 -"
  N51:100/9  "- HMI Input - - Option 10 - Load Stabilizer"
  N51:100/11  "- HMI Input - - Option 12 - Film Sealer"
  N51:101  "- HMI Input - Options"
  N51:101/4  "- HMI Input - - Option 21 -"
  N51:101/5  "- HMI Input - - Option 22 -"
  N51:101/6  "- HMI Input - - Option 23 -"
  N51:101/7  "- HMI Input - - Option 24 -"
  N51:101/11  "- HMI Input - - Option 28 -"
  N51:101/12  "- HMI Input - - Option 29 -"
  N51:101/13  "- HMI Input - - Option 30 -"
  N51:101/14  "- HMI Input - - Option 31 -"
